REGION Network 14: data move
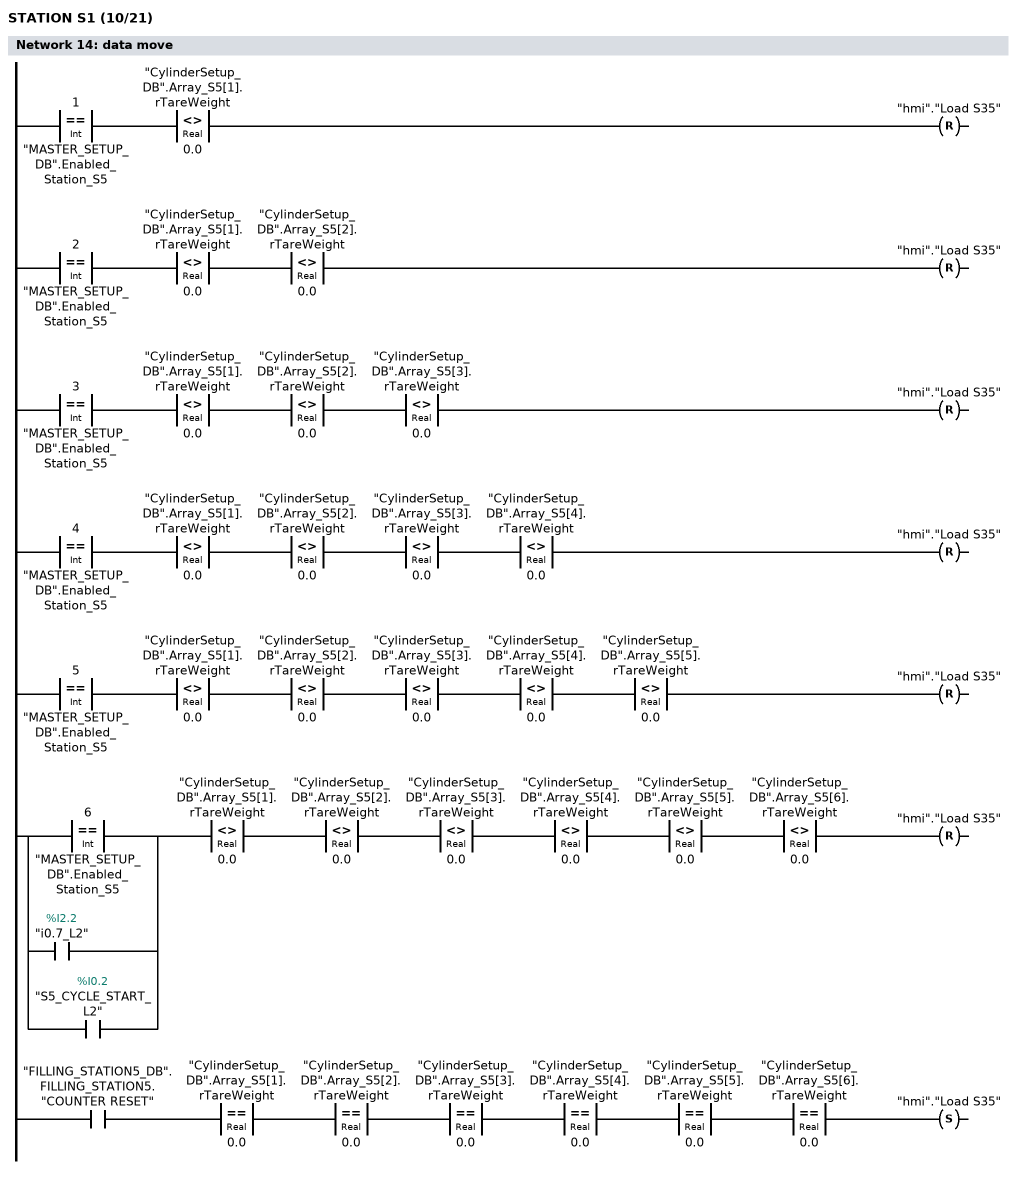
   RUNG wire#powerrail
      { S7_Templates := "SrcType := Int" } EQ_Contact(in1 := 1, in2 := "MASTER_SETUP_DB".Enabled_Station_S5)
      { S7_Templates := "SrcType := Real" } NE_Contact(in1 := "CylinderSetup_DB".Array_S5[1].rTareWeight, in2 := 0.0)
      R_Coil( "hmi"."Load S35" )
   END_RUNG
   RUNG wire#powerrail
      { S7_Templates := "SrcType := Int" } EQ_Contact(in1 := 2, in2 := "MASTER_SETUP_DB".Enabled_Station_S5)
      { S7_Templates := "SrcType := Real" } NE_Contact(in1 := "CylinderSetup_DB".Array_S5[1].rTareWeight, in2 := 0.0)
      { S7_Templates := "SrcType := Real" } NE_Contact(in1 := "CylinderSetup_DB".Array_S5[2].rTareWeight, in2 := 0.0)
      R_Coil( "hmi"."Load S35" )
   END_RUNG
   RUNG wire#powerrail
      { S7_Templates := "SrcType := Int" } EQ_Contact(in1 := 3, in2 := "MASTER_SETUP_DB".Enabled_Station_S5)
      { S7_Templates := "SrcType := Real" } NE_Contact(in1 := "CylinderSetup_DB".Array_S5[1].rTareWeight, in2 := 0.0)
      { S7_Templates := "SrcType := Real" } NE_Contact(in1 := "CylinderSetup_DB".Array_S5[2].rTareWeight, in2 := 0.0)
      { S7_Templates := "SrcType := Real" } NE_Contact(in1 := "CylinderSetup_DB".Array_S5[3].rTareWeight, in2 := 0.0)
      R_Coil( "hmi"."Load S35" )
   END_RUNG
   RUNG wire#powerrail
      { S7_Templates := "SrcType := Int" } EQ_Contact(in1 := 4, in2 := "MASTER_SETUP_DB".Enabled_Station_S5)
      { S7_Templates := "SrcType := Real" } NE_Contact(in1 := "CylinderSetup_DB".Array_S5[1].rTareWeight, in2 := 0.0)
      { S7_Templates := "SrcType := Real" } NE_Contact(in1 := "CylinderSetup_DB".Array_S5[2].rTareWeight, in2 := 0.0)
      { S7_Templates := "SrcType := Real" } NE_Contact(in1 := "CylinderSetup_DB".Array_S5[3].rTareWeight, in2 := 0.0)
      { S7_Templates := "SrcType := Real" } NE_Contact(in1 := "CylinderSetup_DB".Array_S5[4].rTareWeight, in2 := 0.0)
      R_Coil( "hmi"."Load S35" )
   END_RUNG
   RUNG wire#powerrail
      { S7_Templates := "SrcType := Int" } EQ_Contact(in1 := 5, in2 := "MASTER_SETUP_DB".Enabled_Station_S5)
      { S7_Templates := "SrcType := Real" } NE_Contact(in1 := "CylinderSetup_DB".Array_S5[1].rTareWeight, in2 := 0.0)
      { S7_Templates := "SrcType := Real" } NE_Contact(in1 := "CylinderSetup_DB".Array_S5[2].rTareWeight, in2 := 0.0)
      { S7_Templates := "SrcType := Real" } NE_Contact(in1 := "CylinderSetup_DB".Array_S5[3].rTareWeight, in2 := 0.0)
      { S7_Templates := "SrcType := Real" } NE_Contact(in1 := "CylinderSetup_DB".Array_S5[4].rTareWeight, in2 := 0.0)
      { S7_Templates := "SrcType := Real" } NE_Contact(in1 := "CylinderSetup_DB".Array_S5[5].rTareWeight, in2 := 0.0)
      R_Coil( "hmi"."Load S35" )
   END_RUNG
   RUNG wire#powerrail
      { S7_Templates := "SrcType := Int" } EQ_Contact(in1 := 6, in2 := "MASTER_SETUP_DB".Enabled_Station_S5)
      wire#w1
      { S7_Templates := "SrcType := Real" } NE_Contact(in1 := "CylinderSetup_DB".Array_S5[1].rTareWeight, in2 := 0.0)
      { S7_Templates := "SrcType := Real" } NE_Contact(in1 := "CylinderSetup_DB".Array_S5[2].rTareWeight, in2 := 0.0)
      { S7_Templates := "SrcType := Real" } NE_Contact(in1 := "CylinderSetup_DB".Array_S5[3].rTareWeight, in2 := 0.0)
      { S7_Templates := "SrcType := Real" } NE_Contact(in1 := "CylinderSetup_DB".Array_S5[4].rTareWeight, in2 := 0.0)
      { S7_Templates := "SrcType := Real" } NE_Contact(in1 := "CylinderSetup_DB".Array_S5[5].rTareWeight, in2 := 0.0)
      { S7_Templates := "SrcType := Real" } NE_Contact(in1 := "CylinderSetup_DB".Array_S5[6].rTareWeight, in2 := 0.0)
      R_Coil( "hmi"."Load S35" )
   END_RUNG
   RUNG wire#powerrail
      Contact( "i0.7_L2" )
   END_RUNG wire#w1
   RUNG wire#powerrail
      Contact( "S5_CYCLE_START_L2" )
   END_RUNG wire#w1
   RUNG wire#powerrail
      Contact( "FILLING_STATION5_DB".FILLING_STATION5."COUNTER RESET" )
      { S7_Templates := "SrcType := Real" } EQ_Contact(in1 := "CylinderSetup_DB".Array_S5[1].rTareWeight, in2 := 0.0)
      { S7_Templates := "SrcType := Real" } EQ_Contact(in1 := "CylinderSetup_DB".Array_S5[2].rTareWeight, in2 := 0.0)
      { S7_Templates := "SrcType := Real" } EQ_Contact(in1 := "CylinderSetup_DB".Array_S5[3].rTareWeight, in2 := 0.0)
      { S7_Templates := "SrcType := Real" } EQ_Contact(in1 := "CylinderSetup_DB".Array_S5[4].rTareWeight, in2 := 0.0)
      { S7_Templates := "SrcType := Real" } EQ_Contact(in1 := "CylinderSetup_DB".Array_S5[5].rTareWeight, in2 := 0.0)
      { S7_Templates := "SrcType := Real" } EQ_Contact(in1 := "CylinderSetup_DB".Array_S5[6].rTareWeight, in2 := 0.0)
      S_Coil( "hmi"."Load S35" )
   END_RUNG
   // the same network as SCL:
   IF (1 = "MASTER_SETUP_DB".Enabled_Station_S5) AND ("CylinderSetup_DB".Array_S5[1].rTareWeight <> 0.0) THEN
       "hmi"."Load S35" := FALSE;
   END_IF;
   IF (2 = "MASTER_SETUP_DB".Enabled_Station_S5) AND ("CylinderSetup_DB".Array_S5[1].rTareWeight <> 0.0) AND ("CylinderSetup_DB".Array_S5[2].rTareWeight <> 0.0) THEN
       "hmi"."Load S35" := FALSE;
   END_IF;
   IF (3 = "MASTER_SETUP_DB".Enabled_Station_S5) AND ("CylinderSetup_DB".Array_S5[1].rTareWeight <> 0.0) AND ("CylinderSetup_DB".Array_S5[2].rTareWeight <> 0.0) AND ("CylinderSetup_DB".Array_S5[3].rTareWeight <> 0.0) THEN
       "hmi"."Load S35" := FALSE;
   END_IF;
   IF (4 = "MASTER_SETUP_DB".Enabled_Station_S5) AND ("CylinderSetup_DB".Array_S5[1].rTareWeight <> 0.0) AND ("CylinderSetup_DB".Array_S5[2].rTareWeight <> 0.0) AND ("CylinderSetup_DB".Array_S5[3].rTareWeight <> 0.0) AND ("CylinderSetup_DB".Array_S5[4].rTareWeight <> 0.0) THEN
       "hmi"."Load S35" := FALSE;
   END_IF;
   IF (5 = "MASTER_SETUP_DB".Enabled_Station_S5) AND ("CylinderSetup_DB".Array_S5[1].rTareWeight <> 0.0) AND ("CylinderSetup_DB".Array_S5[2].rTareWeight <> 0.0) AND ("CylinderSetup_DB".Array_S5[3].rTareWeight <> 0.0) AND ("CylinderSetup_DB".Array_S5[4].rTareWeight <> 0.0) AND ("CylinderSetup_DB".Array_S5[5].rTareWeight <> 0.0) THEN
       "hmi"."Load S35" := FALSE;
   END_IF;
   IF ((6 = "MASTER_SETUP_DB".Enabled_Station_S5) OR "i0.7_L2" OR "S5_CYCLE_START_L2") AND ("CylinderSetup_DB".Array_S5[1].rTareWeight <> 0.0) AND ("CylinderSetup_DB".Array_S5[2].rTareWeight <> 0.0) AND ("CylinderSetup_DB".Array_S5[3].rTareWeight <> 0.0) AND ("CylinderSetup_DB".Array_S5[4].rTareWeight <> 0.0) AND ("CylinderSetup_DB".Array_S5[5].rTareWeight <> 0.0) AND ("CylinderSetup_DB".Array_S5[6].rTareWeight <> 0.0) THEN
       "hmi"."Load S35" := FALSE;
   END_IF;
   IF "FILLING_STATION5_DB".FILLING_STATION5."COUNTER RESET" AND ("CylinderSetup_DB".Array_S5[1].rTareWeight = 0.0) AND ("CylinderSetup_DB".Array_S5[2].rTareWeight = 0.0) AND ("CylinderSetup_DB".Array_S5[3].rTareWeight = 0.0) AND ("CylinderSetup_DB".Array_S5[4].rTareWeight = 0.0) AND ("CylinderSetup_DB".Array_S5[5].rTareWeight = 0.0) AND ("CylinderSetup_DB".Array_S5[6].rTareWeight = 0.0) THEN
       "hmi"."Load S35" := TRUE;
   END_IF;
END_REGION

REGION Network 15: S5_TO_S7 exit
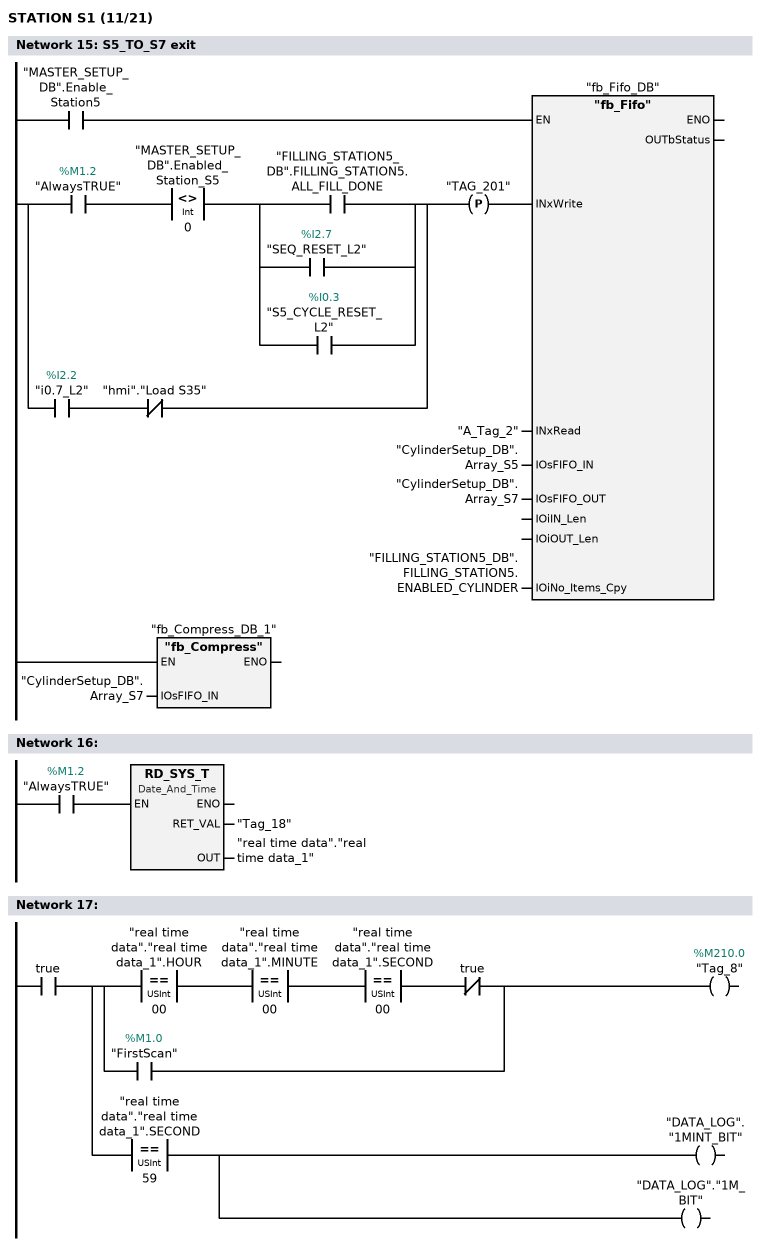
   RUNG wire#powerrail
      Contact( "MASTER_SETUP_DB".Enable_Station5 )
      "fb_Fifo_DB"(INxWrite := wire#w3, INxRead := "A_Tag_2", IOsFIFO_IN := "CylinderSetup_DB".Array_S5, IOsFIFO_OUT := "CylinderSetup_DB".Array_S7, IOiIN_Len :=, IOiOUT_Len :=, IOiNo_Items_Cpy := "FILLING_STATION5_DB".FILLING_STATION5.ENABLED_CYLINDER, OUTbStatus =>)
   END_RUNG
   RUNG wire#powerrail
      Contact( "AlwaysTRUE" )
      { S7_Templates := "SrcType := Int" } NE_Contact(in1 := "MASTER_SETUP_DB".Enabled_Station_S5, in2 := 0)
      wire#w1
      Contact( "FILLING_STATION5_DB".FILLING_STATION5.ALL_FILL_DONE )
      wire#w2
      P_Trig( "TAG_201" )
   END_RUNG wire#w3
   RUNG wire#w1
      Contact( "SEQ_RESET_L2" )
   END_RUNG wire#w2
   RUNG wire#w1
      Contact( "S5_CYCLE_RESET_L2" )
   END_RUNG wire#w2
   RUNG wire#powerrail
      Contact( "i0.7_L2" )
      I_Contact( "hmi"."Load S35" )
   END_RUNG wire#w2
   RUNG wire#powerrail
      "fb_Compress_DB_1"(IOsFIFO_IN := "CylinderSetup_DB".Array_S7)
   END_RUNG
   // the same network as SCL:
   #_w1 := ("AlwaysTRUE" AND ("MASTER_SETUP_DB".Enabled_Station_S5 <> 0) AND ("FILLING_STATION5_DB".FILLING_STATION5.ALL_FILL_DONE OR "SEQ_RESET_L2" OR "S5_CYCLE_RESET_L2")) OR ("i0.7_L2" AND NOT "hmi"."Load S35");
   #_w2 := #_w1 AND NOT "TAG_201";   // rising edge
   "TAG_201" := #_w1;
   IF "MASTER_SETUP_DB".Enable_Station5 THEN
       "fb_Fifo_DB"(INxWrite := #_w2,   // "fb_Fifo"
                    INxRead := "A_Tag_2",
                    IOsFIFO_IN := "CylinderSetup_DB".Array_S5,
                    IOsFIFO_OUT := "CylinderSetup_DB".Array_S7,
                    IOiNo_Items_Cpy := "FILLING_STATION5_DB".FILLING_STATION5.ENABLED_CYLINDER);
   END_IF;
   "fb_Compress_DB_1"(IOsFIFO_IN := "CylinderSetup_DB".Array_S7);   // "fb_Compress"
END_REGION

REGION Network 16
   RUNG wire#powerrail
      Contact( "AlwaysTRUE" )
      { S7_Templates := "date_type := Date_And_Time" } RD_SYS_T(RET_VAL => "Tag_18", OUT => "real time data"."real time data_1")
   END_RUNG
   // the same network as SCL:
   IF "AlwaysTRUE" THEN "Tag_18" := RD_SYS_T(OUT => "real time data"."real time data_1"); END_IF;
END_REGION

REGION Network 17
   RUNG wire#powerrail
      Contact( true )
      wire#w1
      { S7_Templates := "SrcType := USInt" } EQ_Contact(in1 := "real time data"."real time data_1".HOUR, in2 := 00)
      { S7_Templates := "SrcType := USInt" } EQ_Contact(in1 := "real time data"."real time data_1".MINUTE, in2 := 00)
      { S7_Templates := "SrcType := USInt" } EQ_Contact(in1 := "real time data"."real time data_1".SECOND, in2 := 00)
      I_Contact( true )
      wire#w2
      Coil( "Tag_8" )
   END_RUNG
   RUNG wire#w1
      Contact( "FirstScan" )
   END_RUNG wire#w2
   RUNG wire#w1
      { S7_Templates := "SrcType := USInt" } EQ_Contact(in1 := "real time data"."real time data_1".SECOND, in2 := 59)
      wire#w3
      Coil( "DATA_LOG"."1MINT_BIT" )
   END_RUNG
   RUNG wire#w3
      Coil( "DATA_LOG"."1M_BIT" )
   END_RUNG
   // the same network as SCL:
   "Tag_8" := true AND ((("real time data"."real time data_1".HOUR = 00) AND ("real time data"."real time data_1".MINUTE = 00) AND ("real time data"."real time data_1".SECOND = 00) AND NOT true) OR "FirstScan");
   "DATA_LOG"."1MINT_BIT" := true AND ("real time data"."real time data_1".SECOND = 59);
   "DATA_LOG"."1M_BIT" := "DATA_LOG"."1MINT_BIT";
END_REGION

REGION Network 18 (SCL): S4 S6 FIFO DATA SKIP
   #idx2 := 0;
   #idx3 := 0;

   IF "AlwaysTRUE" THEN
       FOR #idx2 := 1 TO "MASTER_SETUP_DB".S4_Total_Station DO

           IF "MASTER_SETUP_DB".S4_Enabled_Station[#idx2]  THEN
               #idx3 := #idx3 + 1;
               "hmi_dummy_array".S4_PrefillingDummyData[#idx2] := "CylinderSetup_DB".Array_S6[#idx3];

             ELSIF
                #idx2 > "MASTER_SETUP_DB".S4_Total_Station OR #idx3 >"MASTER_SETUP_DB".S4_Total_Station THEN
                   EXIT;
               END_IF;
           END_FOR;


   END_IF;
END_REGION

REGION Network 19 (SCL)
   #idx4 := 0;
   #idx6 := 0;

   IF "AlwaysTRUE" THEN
       FOR #idx4 := 1 TO "MASTER_SETUP_DB".S5_Total_Station DO

           IF "MASTER_SETUP_DB".S5_Enabled_Station[#idx4] THEN
               #idx6 := #idx6 + 1;
               "hmi_dummy_array".S5_PrefillingdummyData[#idx4] := "CylinderSetup_DB".Array_S5[#idx6];

           ELSIF
               #idx4 > "MASTER_SETUP_DB".S5_Total_Station OR #idx6 > "MASTER_SETUP_DB".S5_Total_Station THEN
               EXIT;
           END_IF;
       END_FOR;


   END_IF;
END_REGION

REGION Network 20
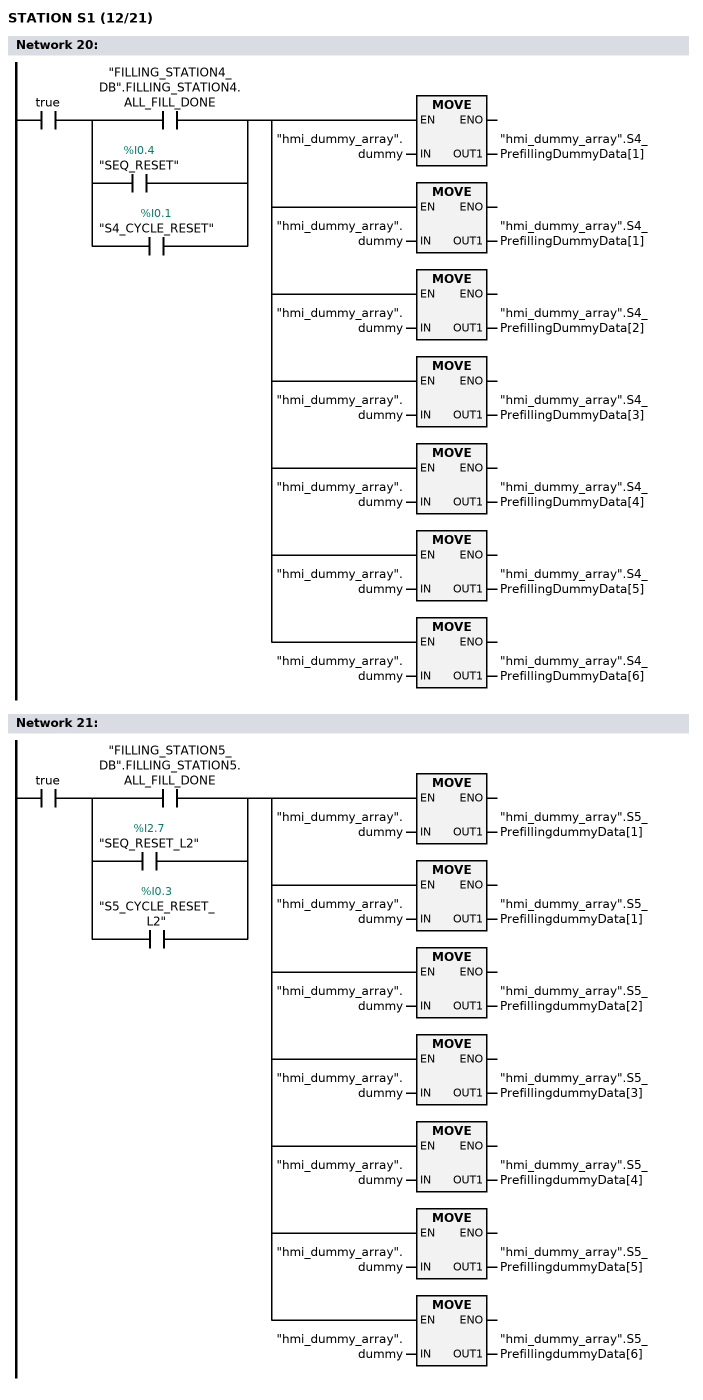
   RUNG wire#powerrail
      Contact( true )
      wire#w1
      Contact( "FILLING_STATION4_DB".FILLING_STATION4.ALL_FILL_DONE )
      wire#w2
      Move(in := "hmi_dummy_array".dummy, out1 => "hmi_dummy_array".S4_PrefillingDummyData[1])
   END_RUNG
   RUNG wire#w1
      Contact( "SEQ_RESET" )
   END_RUNG wire#w2
   RUNG wire#w1
      Contact( "S4_CYCLE_RESET" )
   END_RUNG wire#w2
   RUNG wire#w2
      Move(in := "hmi_dummy_array".dummy, out1 => "hmi_dummy_array".S4_PrefillingDummyData[1])
   END_RUNG
   RUNG wire#w2
      Move(in := "hmi_dummy_array".dummy, out1 => "hmi_dummy_array".S4_PrefillingDummyData[2])
   END_RUNG
   RUNG wire#w2
      Move(in := "hmi_dummy_array".dummy, out1 => "hmi_dummy_array".S4_PrefillingDummyData[3])
   END_RUNG
   RUNG wire#w2
      Move(in := "hmi_dummy_array".dummy, out1 => "hmi_dummy_array".S4_PrefillingDummyData[4])
   END_RUNG
   RUNG wire#w2
      Move(in := "hmi_dummy_array".dummy, out1 => "hmi_dummy_array".S4_PrefillingDummyData[5])
   END_RUNG
   RUNG wire#w2
      Move(in := "hmi_dummy_array".dummy, out1 => "hmi_dummy_array".S4_PrefillingDummyData[6])
   END_RUNG
   // the same network as SCL:
   IF true AND ("FILLING_STATION4_DB".FILLING_STATION4.ALL_FILL_DONE OR "SEQ_RESET" OR "S4_CYCLE_RESET") THEN
       "hmi_dummy_array".S4_PrefillingDummyData[1] := "hmi_dummy_array".dummy;
       "hmi_dummy_array".S4_PrefillingDummyData[1] := "hmi_dummy_array".dummy;
       "hmi_dummy_array".S4_PrefillingDummyData[2] := "hmi_dummy_array".dummy;
       "hmi_dummy_array".S4_PrefillingDummyData[3] := "hmi_dummy_array".dummy;
       "hmi_dummy_array".S4_PrefillingDummyData[4] := "hmi_dummy_array".dummy;
       "hmi_dummy_array".S4_PrefillingDummyData[5] := "hmi_dummy_array".dummy;
       "hmi_dummy_array".S4_PrefillingDummyData[6] := "hmi_dummy_array".dummy;
   END_IF;
END_REGION

REGION Network 21
   RUNG wire#powerrail
      Contact( true )
      wire#w1
      Contact( "FILLING_STATION5_DB".FILLING_STATION5.ALL_FILL_DONE )
      wire#w2
      Move(in := "hmi_dummy_array".dummy, out1 => "hmi_dummy_array".S5_PrefillingdummyData[1])
   END_RUNG
   RUNG wire#w1
      Contact( "SEQ_RESET_L2" )
   END_RUNG wire#w2
   RUNG wire#w1
      Contact( "S5_CYCLE_RESET_L2" )
   END_RUNG wire#w2
   RUNG wire#w2
      Move(in := "hmi_dummy_array".dummy, out1 => "hmi_dummy_array".S5_PrefillingdummyData[1])
   END_RUNG
   RUNG wire#w2
      Move(in := "hmi_dummy_array".dummy, out1 => "hmi_dummy_array".S5_PrefillingdummyData[2])
   END_RUNG
   RUNG wire#w2
      Move(in := "hmi_dummy_array".dummy, out1 => "hmi_dummy_array".S5_PrefillingdummyData[3])
   END_RUNG
   RUNG wire#w2
      Move(in := "hmi_dummy_array".dummy, out1 => "hmi_dummy_array".S5_PrefillingdummyData[4])
   END_RUNG
   RUNG wire#w2
      Move(in := "hmi_dummy_array".dummy, out1 => "hmi_dummy_array".S5_PrefillingdummyData[5])
   END_RUNG
   RUNG wire#w2
      Move(in := "hmi_dummy_array".dummy, out1 => "hmi_dummy_array".S5_PrefillingdummyData[6])
   END_RUNG
   // the same network as SCL:
   IF true AND ("FILLING_STATION5_DB".FILLING_STATION5.ALL_FILL_DONE OR "SEQ_RESET_L2" OR "S5_CYCLE_RESET_L2") THEN
       "hmi_dummy_array".S5_PrefillingdummyData[1] := "hmi_dummy_array".dummy;
       "hmi_dummy_array".S5_PrefillingdummyData[1] := "hmi_dummy_array".dummy;
       "hmi_dummy_array".S5_PrefillingdummyData[2] := "hmi_dummy_array".dummy;
       "hmi_dummy_array".S5_PrefillingdummyData[3] := "hmi_dummy_array".dummy;
       "hmi_dummy_array".S5_PrefillingdummyData[4] := "hmi_dummy_array".dummy;
       "hmi_dummy_array".S5_PrefillingdummyData[5] := "hmi_dummy_array".dummy;
       "hmi_dummy_array".S5_PrefillingdummyData[6] := "hmi_dummy_array".dummy;
   END_IF;
END_REGION

REGION Network 22
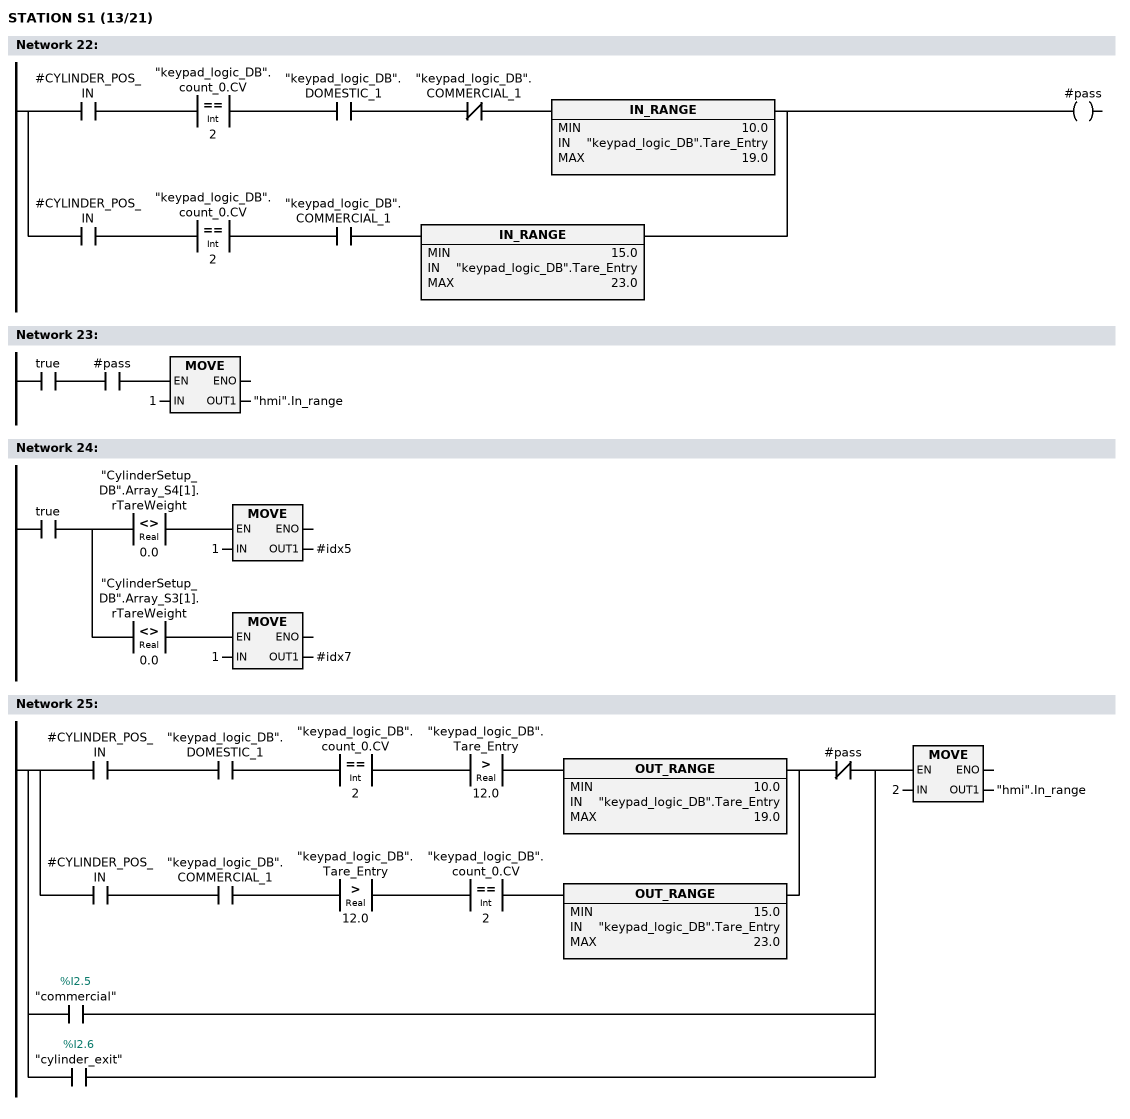
   RUNG wire#powerrail
      Contact( #CYLINDER_POS_IN )
      { S7_Templates := "SrcType := Int" } EQ_Contact(in1 := "keypad_logic_DB".count_0.CV, in2 := 2)
      Contact( "keypad_logic_DB".DOMESTIC_1 )
      I_Contact( "keypad_logic_DB".COMMERCIAL_1 )
      { S7_Templates := "SrcType := Real" } InRange(min := 10.0, in := "keypad_logic_DB".Tare_Entry, max := 19.0)
      wire#w1
      Coil( #pass )
   END_RUNG
   RUNG wire#powerrail
      Contact( #CYLINDER_POS_IN )
      { S7_Templates := "SrcType := Int" } EQ_Contact(in1 := "keypad_logic_DB".count_0.CV, in2 := 2)
      Contact( "keypad_logic_DB".COMMERCIAL_1 )
      { S7_Templates := "SrcType := Real" } InRange(min := 15.0, in := "keypad_logic_DB".Tare_Entry, max := 23.0)
   END_RUNG wire#w1
   // the same network as SCL:
   #pass := (#CYLINDER_POS_IN AND ("keypad_logic_DB".count_0.CV = 2) AND "keypad_logic_DB".DOMESTIC_1 AND NOT "keypad_logic_DB".COMMERCIAL_1 AND (10.0 <= "keypad_logic_DB".Tare_Entry) AND ("keypad_logic_DB".Tare_Entry <= 19.0)) OR (#CYLINDER_POS_IN AND ("keypad_logic_DB".count_0.CV = 2) AND "keypad_logic_DB".COMMERCIAL_1 AND (15.0 <= "keypad_logic_DB".Tare_Entry) AND ("keypad_logic_DB".Tare_Entry <= 23.0));
END_REGION

REGION Network 23
   RUNG wire#powerrail
      Contact( true )
      Contact( #pass )
      Move(in := 1, out1 => "hmi".In_range)
   END_RUNG
   // the same network as SCL:
   IF true AND #pass THEN "hmi".In_range := 1; END_IF;
END_REGION

REGION Network 24
   RUNG wire#powerrail
      Contact( true )
      wire#w1
      { S7_Templates := "SrcType := Real" } NE_Contact(in1 := "CylinderSetup_DB".Array_S4[1].rTareWeight, in2 := 0.0)
      Move(in := 1, out1 => #idx5)
   END_RUNG
   RUNG wire#w1
      { S7_Templates := "SrcType := Real" } NE_Contact(in1 := "CylinderSetup_DB".Array_S3[1].rTareWeight, in2 := 0.0)
      Move(in := 1, out1 => #idx7)
   END_RUNG
   // the same network as SCL:
   IF true AND ("CylinderSetup_DB".Array_S4[1].rTareWeight <> 0.0) THEN #idx5 := 1; END_IF;
   IF true AND ("CylinderSetup_DB".Array_S3[1].rTareWeight <> 0.0) THEN #idx7 := 1; END_IF;
END_REGION

REGION Network 25
   IF (((#CYLINDER_POS_IN AND "keypad_logic_DB".DOMESTIC_1 AND ("keypad_logic_DB".count_0.CV = 2) AND ("keypad_logic_DB".Tare_Entry > 12.0) AND (("keypad_logic_DB".Tare_Entry < 10.0) OR ("keypad_logic_DB".Tare_Entry > 19.0))) OR (#CYLINDER_POS_IN AND "keypad_logic_DB".COMMERCIAL_1 AND ("keypad_logic_DB".Tare_Entry > 12.0) AND ("keypad_logic_DB".count_0.CV = 2) AND (("keypad_logic_DB".Tare_Entry < 15.0) OR ("keypad_logic_DB".Tare_Entry > 23.0)))) AND NOT #pass) OR "commercial" OR "cylinder_exit" THEN
       "hmi".In_range := 2;
   END_IF;
END_REGION

REGION Network 26
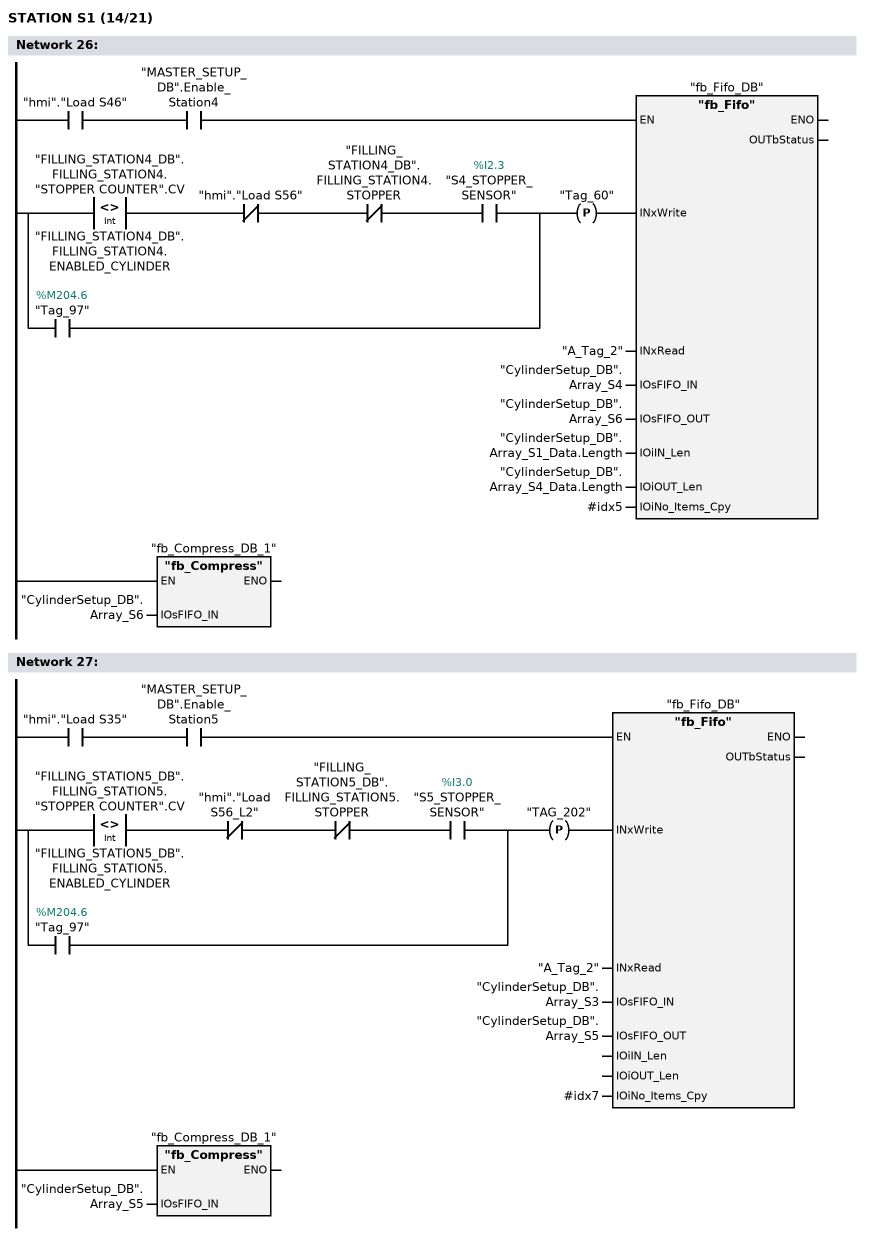
   RUNG wire#powerrail
      Contact( "hmi"."Load S46" )
      Contact( "MASTER_SETUP_DB".Enable_Station4 )
      "fb_Fifo_DB"(INxWrite := wire#w2, INxRead := "A_Tag_2", IOsFIFO_IN := "CylinderSetup_DB".Array_S4, IOsFIFO_OUT := "CylinderSetup_DB".Array_S6, IOiIN_Len := "CylinderSetup_DB".Array_S1_Data.Length, IOiOUT_Len := "CylinderSetup_DB".Array_S4_Data.Length, IOiNo_Items_Cpy := #idx5, OUTbStatus =>)
   END_RUNG
   RUNG wire#powerrail
      { S7_Templates := "SrcType := Int" } NE_Contact(in1 := "FILLING_STATION4_DB".FILLING_STATION4."STOPPER COUNTER".CV, in2 := "FILLING_STATION4_DB".FILLING_STATION4.ENABLED_CYLINDER)
      I_Contact( "hmi"."Load S56" )
      I_Contact( "FILLING_STATION4_DB".FILLING_STATION4.STOPPER )
      Contact( "S4_STOPPER_SENSOR" )
      wire#w1
      P_Trig( "Tag_60" )
   END_RUNG wire#w2
   RUNG wire#powerrail
      Contact( "Tag_97" )
   END_RUNG wire#w1
   RUNG wire#powerrail
      "fb_Compress_DB_1"(IOsFIFO_IN := "CylinderSetup_DB".Array_S6)
   END_RUNG
   // the same network as SCL:
   #_w1 := (("FILLING_STATION4_DB".FILLING_STATION4."STOPPER COUNTER".CV <> "FILLING_STATION4_DB".FILLING_STATION4.ENABLED_CYLINDER) AND NOT "hmi"."Load S56" AND NOT "FILLING_STATION4_DB".FILLING_STATION4.STOPPER AND "S4_STOPPER_SENSOR") OR "Tag_97";
   #_w2 := #_w1 AND NOT "Tag_60";   // rising edge
   "Tag_60" := #_w1;
   IF "hmi"."Load S46" AND "MASTER_SETUP_DB".Enable_Station4 THEN
       "fb_Fifo_DB"(INxWrite := #_w2,   // "fb_Fifo"
                    INxRead := "A_Tag_2",
                    IOsFIFO_IN := "CylinderSetup_DB".Array_S4,
                    IOsFIFO_OUT := "CylinderSetup_DB".Array_S6,
                    IOiIN_Len := "CylinderSetup_DB".Array_S1_Data.Length,
                    IOiOUT_Len := "CylinderSetup_DB".Array_S4_Data.Length,
                    IOiNo_Items_Cpy := #idx5);
   END_IF;
   "fb_Compress_DB_1"(IOsFIFO_IN := "CylinderSetup_DB".Array_S6);   // "fb_Compress"
END_REGION

REGION Network 27
   RUNG wire#powerrail
      Contact( "hmi"."Load S35" )
      Contact( "MASTER_SETUP_DB".Enable_Station5 )
      "fb_Fifo_DB"(INxWrite := wire#w2, INxRead := "A_Tag_2", IOsFIFO_IN := "CylinderSetup_DB".Array_S3, IOsFIFO_OUT := "CylinderSetup_DB".Array_S5, IOiIN_Len :=, IOiOUT_Len :=, IOiNo_Items_Cpy := #idx7, OUTbStatus =>)
   END_RUNG
   RUNG wire#powerrail
      { S7_Templates := "SrcType := Int" } NE_Contact(in1 := "FILLING_STATION5_DB".FILLING_STATION5."STOPPER COUNTER".CV, in2 := "FILLING_STATION5_DB".FILLING_STATION5.ENABLED_CYLINDER)
      I_Contact( "hmi"."Load S56_L2" )
      I_Contact( "FILLING_STATION5_DB".FILLING_STATION5.STOPPER )
      Contact( "S5_STOPPER_SENSOR" )
      wire#w1
      P_Trig( "TAG_202" )
   END_RUNG wire#w2
   RUNG wire#powerrail
      Contact( "Tag_97" )
   END_RUNG wire#w1
   RUNG wire#powerrail
      "fb_Compress_DB_1"(IOsFIFO_IN := "CylinderSetup_DB".Array_S5)
   END_RUNG
   // the same network as SCL:
   #_w1 := (("FILLING_STATION5_DB".FILLING_STATION5."STOPPER COUNTER".CV <> "FILLING_STATION5_DB".FILLING_STATION5.ENABLED_CYLINDER) AND NOT "hmi"."Load S56_L2" AND NOT "FILLING_STATION5_DB".FILLING_STATION5.STOPPER AND "S5_STOPPER_SENSOR") OR "Tag_97";
   #_w2 := #_w1 AND NOT "TAG_202";   // rising edge
   "TAG_202" := #_w1;
   IF "hmi"."Load S35" AND "MASTER_SETUP_DB".Enable_Station5 THEN
       "fb_Fifo_DB"(INxWrite := #_w2,   // "fb_Fifo"
                    INxRead := "A_Tag_2",
                    IOsFIFO_IN := "CylinderSetup_DB".Array_S3,
                    IOsFIFO_OUT := "CylinderSetup_DB".Array_S5,
                    IOiNo_Items_Cpy := #idx7);
   END_IF;
   "fb_Compress_DB_1"(IOsFIFO_IN := "CylinderSetup_DB".Array_S5);   // "fb_Compress"
END_REGION

REGION Network 28
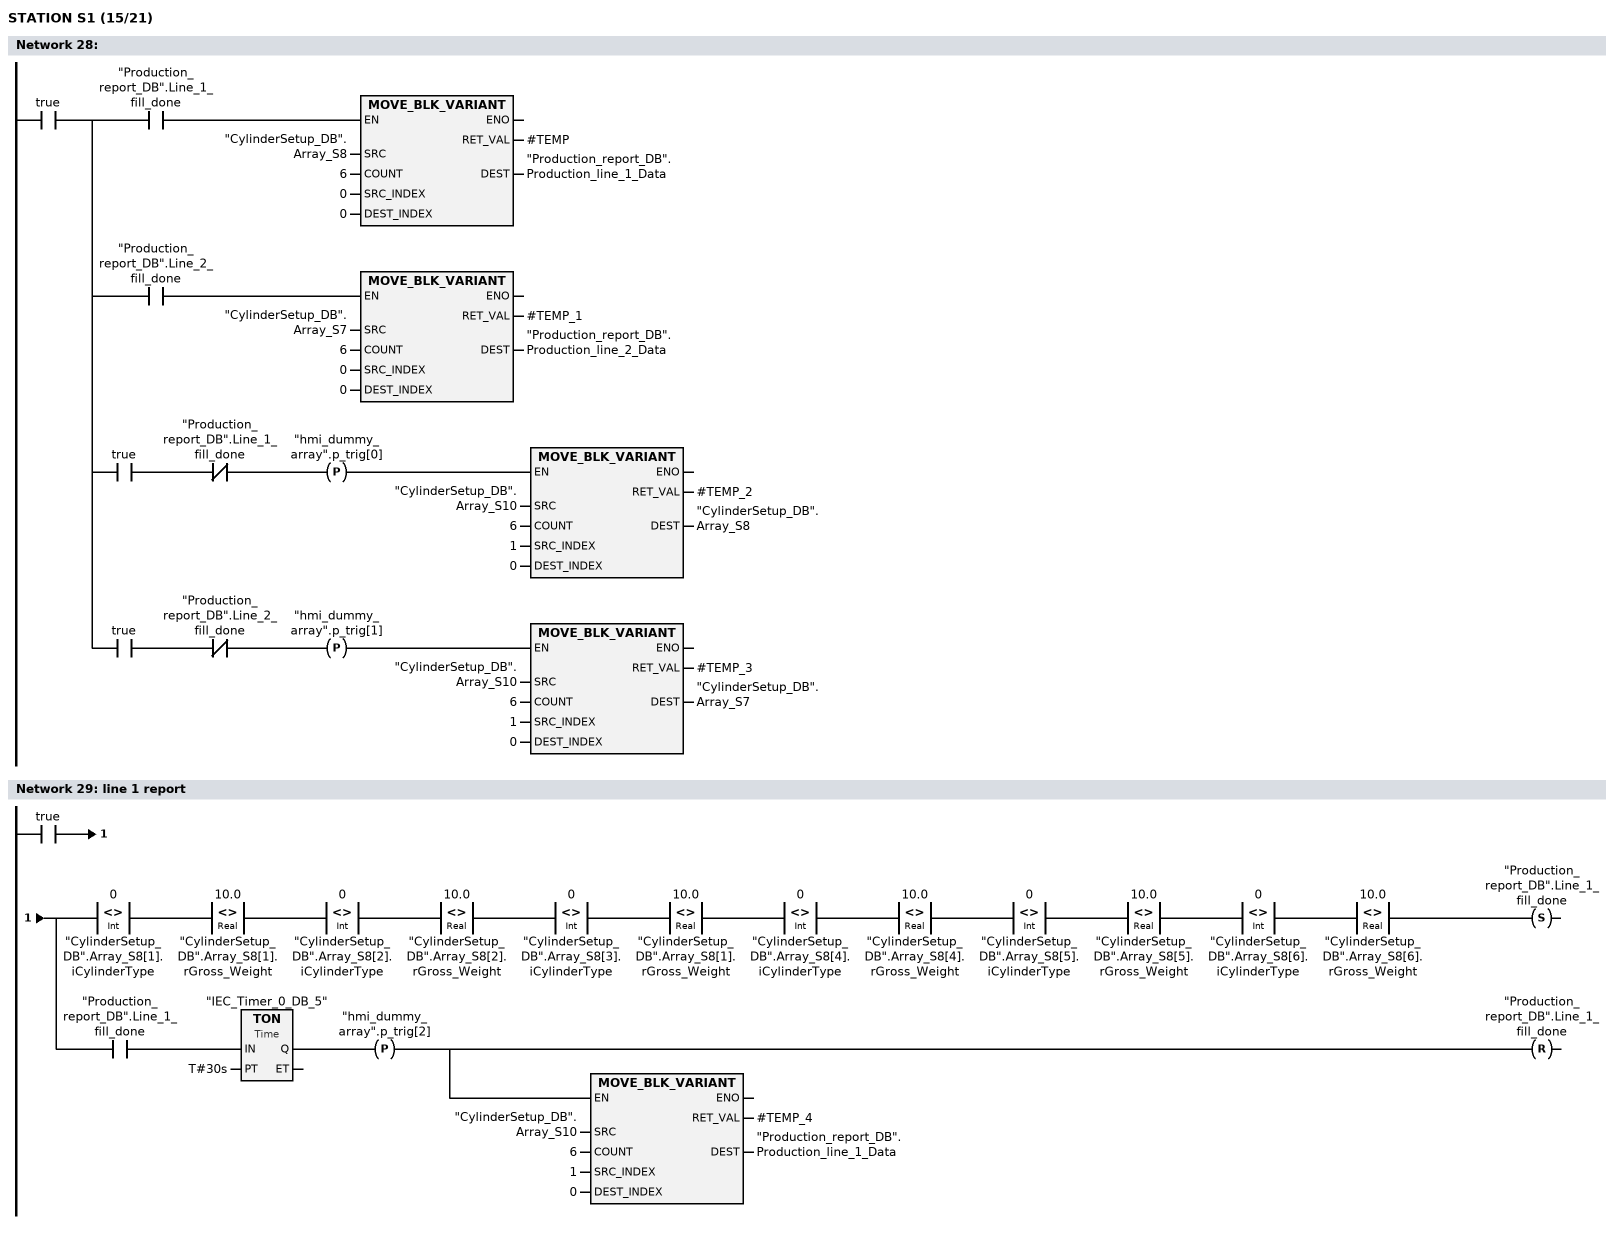
   RUNG wire#powerrail
      Contact( true )
      wire#w1
      Contact( "Production_report_DB".Line_1_fill_done )
      MOVE_BLK_VARIANT(SRC := "CylinderSetup_DB".Array_S8, COUNT := 6, SRC_INDEX := 0, DEST_INDEX := 0, Ret_Val => #TEMP, DEST => "Production_report_DB".Production_line_1_Data)
   END_RUNG
   RUNG wire#w1
      Contact( "Production_report_DB".Line_2_fill_done )
      MOVE_BLK_VARIANT(SRC := "CylinderSetup_DB".Array_S7, COUNT := 6, SRC_INDEX := 0, DEST_INDEX := 0, Ret_Val => #TEMP_1, DEST => "Production_report_DB".Production_line_2_Data)
   END_RUNG
   RUNG wire#w1
      Contact( true )
      I_Contact( "Production_report_DB".Line_1_fill_done )
      P_Trig( "hmi_dummy_array".p_trig[0] )
      MOVE_BLK_VARIANT(SRC := "CylinderSetup_DB".Array_S10, COUNT := 6, SRC_INDEX := 1, DEST_INDEX := 0, Ret_Val => #TEMP_2, DEST => "CylinderSetup_DB".Array_S8)
   END_RUNG
   RUNG wire#w1
      Contact( true )
      I_Contact( "Production_report_DB".Line_2_fill_done )
      P_Trig( "hmi_dummy_array".p_trig[1] )
      MOVE_BLK_VARIANT(SRC := "CylinderSetup_DB".Array_S10, COUNT := 6, SRC_INDEX := 1, DEST_INDEX := 0, Ret_Val => #TEMP_3, DEST => "CylinderSetup_DB".Array_S7)
   END_RUNG
   // the same network as SCL:
   IF true AND "Production_report_DB".Line_1_fill_done THEN
       #TEMP := MOVE_BLK_VARIANT(SRC := "CylinderSetup_DB".Array_S8,
                               COUNT := 6,
                               SRC_INDEX := 0,
                               DEST_INDEX := 0,
                               DEST => "Production_report_DB".Production_line_1_Data);
   END_IF;
   IF true AND "Production_report_DB".Line_2_fill_done THEN
       #TEMP_1 := MOVE_BLK_VARIANT(SRC := "CylinderSetup_DB".Array_S7,
                               COUNT := 6,
                               SRC_INDEX := 0,
                               DEST_INDEX := 0,
                               DEST => "Production_report_DB".Production_line_2_Data);
   END_IF;
   #_w1 := true AND true AND NOT "Production_report_DB".Line_1_fill_done;
   #_w2 := #_w1 AND NOT "hmi_dummy_array".p_trig[0];   // rising edge
   "hmi_dummy_array".p_trig[0] := #_w1;
   IF #_w2 THEN
       #TEMP_2 := MOVE_BLK_VARIANT(SRC := "CylinderSetup_DB".Array_S10,
                               COUNT := 6,
                               SRC_INDEX := 1,
                               DEST_INDEX := 0,
                               DEST => "CylinderSetup_DB".Array_S8);
   END_IF;
   #_w3 := true AND true AND NOT "Production_report_DB".Line_2_fill_done;
   #_w4 := #_w3 AND NOT "hmi_dummy_array".p_trig[1];   // rising edge
   "hmi_dummy_array".p_trig[1] := #_w3;
   IF #_w4 THEN
       #TEMP_3 := MOVE_BLK_VARIANT(SRC := "CylinderSetup_DB".Array_S10,
                               COUNT := 6,
                               SRC_INDEX := 1,
                               DEST_INDEX := 0,
                               DEST => "CylinderSetup_DB".Array_S7);
   END_IF;
END_REGION

REGION Network 29: line 1 report
   RUNG wire#powerrail
      Contact( true )
      wire#w1
      { S7_Templates := "SrcType := Int" } NE_Contact(in1 := 0, in2 := "CylinderSetup_DB".Array_S8[1].iCylinderType)
      { S7_Templates := "SrcType := Real" } NE_Contact(in1 := 10.0, in2 := "CylinderSetup_DB".Array_S8[1].rGross_Weight)
      { S7_Templates := "SrcType := Int" } NE_Contact(in1 := 0, in2 := "CylinderSetup_DB".Array_S8[2].iCylinderType)
      { S7_Templates := "SrcType := Real" } NE_Contact(in1 := 10.0, in2 := "CylinderSetup_DB".Array_S8[2].rGross_Weight)
      { S7_Templates := "SrcType := Int" } NE_Contact(in1 := 0, in2 := "CylinderSetup_DB".Array_S8[3].iCylinderType)
      { S7_Templates := "SrcType := Real" } NE_Contact(in1 := 10.0, in2 := "CylinderSetup_DB".Array_S8[1].rGross_Weight)
      { S7_Templates := "SrcType := Int" } NE_Contact(in1 := 0, in2 := "CylinderSetup_DB".Array_S8[4].iCylinderType)
      { S7_Templates := "SrcType := Real" } NE_Contact(in1 := 10.0, in2 := "CylinderSetup_DB".Array_S8[4].rGross_Weight)
      { S7_Templates := "SrcType := Int" } NE_Contact(in1 := 0, in2 := "CylinderSetup_DB".Array_S8[5].iCylinderType)
      { S7_Templates := "SrcType := Real" } NE_Contact(in1 := 10.0, in2 := "CylinderSetup_DB".Array_S8[5].rGross_Weight)
      { S7_Templates := "SrcType := Int" } NE_Contact(in1 := 0, in2 := "CylinderSetup_DB".Array_S8[6].iCylinderType)
      { S7_Templates := "SrcType := Real" } NE_Contact(in1 := 10.0, in2 := "CylinderSetup_DB".Array_S8[6].rGross_Weight)
      S_Coil( "Production_report_DB".Line_1_fill_done )
   END_RUNG
   RUNG wire#w1
      Contact( "Production_report_DB".Line_1_fill_done )
      { S7_Templates := "time_type := Time" } "IEC_Timer_0_DB_5".TON(pt := T#30s, et =>)
      P_Trig( "hmi_dummy_array".p_trig[2] )
      wire#w2
      R_Coil( "Production_report_DB".Line_1_fill_done )
   END_RUNG
   RUNG wire#w2
      MOVE_BLK_VARIANT(SRC := "CylinderSetup_DB".Array_S10, COUNT := 6, SRC_INDEX := 1, DEST_INDEX := 0, Ret_Val => #TEMP_4, DEST => "Production_report_DB".Production_line_1_Data)
   END_RUNG
   // the same network as SCL:
   IF true AND (0 <> "CylinderSetup_DB".Array_S8[1].iCylinderType) AND (10.0 <> "CylinderSetup_DB".Array_S8[1].rGross_Weight) AND (0 <> "CylinderSetup_DB".Array_S8[2].iCylinderType) AND (10.0 <> "CylinderSetup_DB".Array_S8[2].rGross_Weight) AND (0 <> "CylinderSetup_DB".Array_S8[3].iCylinderType) AND (10.0 <> "CylinderSetup_DB".Array_S8[1].rGross_Weight) AND (0 <> "CylinderSetup_DB".Array_S8[4].iCylinderType) AND (10.0 <> "CylinderSetup_DB".Array_S8[4].rGross_Weight) AND (0 <> "CylinderSetup_DB".Array_S8[5].iCylinderType) AND (10.0 <> "CylinderSetup_DB".Array_S8[5].rGross_Weight) AND (0 <> "CylinderSetup_DB".Array_S8[6].iCylinderType) AND (10.0 <> "CylinderSetup_DB".Array_S8[6].rGross_Weight) THEN
       "Production_report_DB".Line_1_fill_done := TRUE;
   END_IF;
   "IEC_Timer_0_DB_5".TON(IN := true AND "Production_report_DB".Line_1_fill_done, PT := T#30s);
   #_w1 := "IEC_Timer_0_DB_5".Q AND NOT "hmi_dummy_array".p_trig[2];   // rising edge
   "hmi_dummy_array".p_trig[2] := "IEC_Timer_0_DB_5".Q;
   IF #_w1 THEN
       "Production_report_DB".Line_1_fill_done := FALSE;
       #TEMP_4 := MOVE_BLK_VARIANT(SRC := "CylinderSetup_DB".Array_S10,
                               COUNT := 6,
                               SRC_INDEX := 1,
                               DEST_INDEX := 0,
                               DEST => "Production_report_DB".Production_line_1_Data);
   END_IF;
END_REGION

REGION Network 30: line 2 report
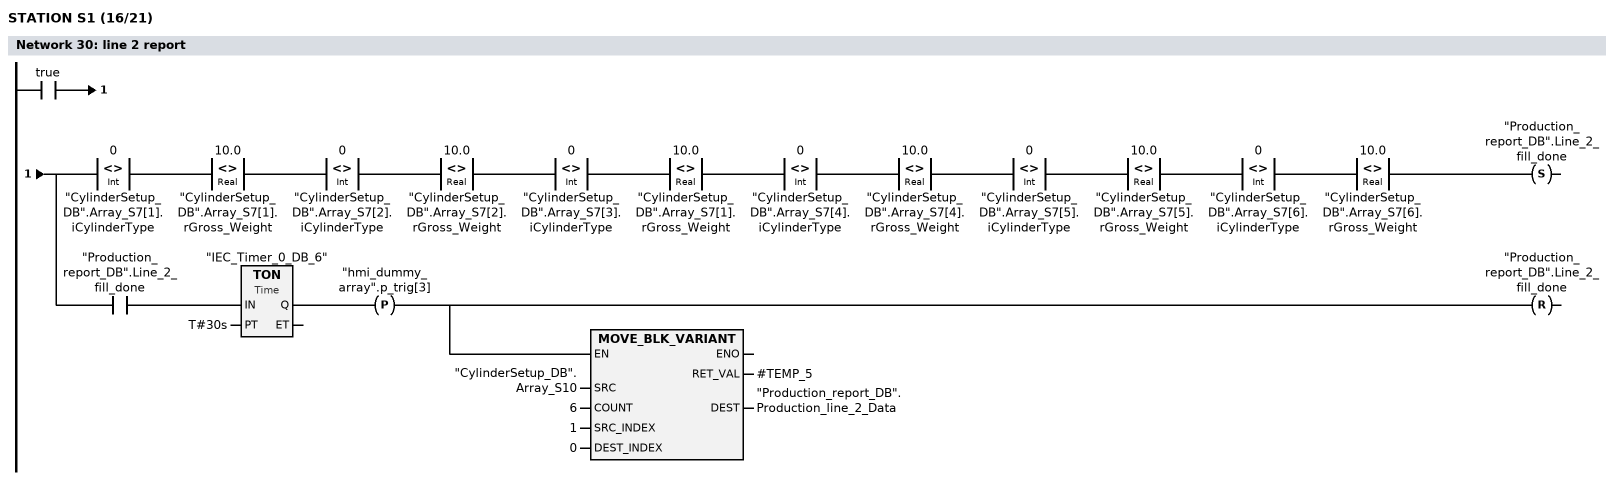
   RUNG wire#powerrail
      Contact( true )
      wire#w1
      { S7_Templates := "SrcType := Int" } NE_Contact(in1 := 0, in2 := "CylinderSetup_DB".Array_S7[1].iCylinderType)
      { S7_Templates := "SrcType := Real" } NE_Contact(in1 := 10.0, in2 := "CylinderSetup_DB".Array_S7[1].rGross_Weight)
      { S7_Templates := "SrcType := Int" } NE_Contact(in1 := 0, in2 := "CylinderSetup_DB".Array_S7[2].iCylinderType)
      { S7_Templates := "SrcType := Real" } NE_Contact(in1 := 10.0, in2 := "CylinderSetup_DB".Array_S7[2].rGross_Weight)
      { S7_Templates := "SrcType := Int" } NE_Contact(in1 := 0, in2 := "CylinderSetup_DB".Array_S7[3].iCylinderType)
      { S7_Templates := "SrcType := Real" } NE_Contact(in1 := 10.0, in2 := "CylinderSetup_DB".Array_S7[1].rGross_Weight)
      { S7_Templates := "SrcType := Int" } NE_Contact(in1 := 0, in2 := "CylinderSetup_DB".Array_S7[4].iCylinderType)
      { S7_Templates := "SrcType := Real" } NE_Contact(in1 := 10.0, in2 := "CylinderSetup_DB".Array_S7[4].rGross_Weight)
      { S7_Templates := "SrcType := Int" } NE_Contact(in1 := 0, in2 := "CylinderSetup_DB".Array_S7[5].iCylinderType)
      { S7_Templates := "SrcType := Real" } NE_Contact(in1 := 10.0, in2 := "CylinderSetup_DB".Array_S7[5].rGross_Weight)
      { S7_Templates := "SrcType := Int" } NE_Contact(in1 := 0, in2 := "CylinderSetup_DB".Array_S7[6].iCylinderType)
      { S7_Templates := "SrcType := Real" } NE_Contact(in1 := 10.0, in2 := "CylinderSetup_DB".Array_S7[6].rGross_Weight)
      S_Coil( "Production_report_DB".Line_2_fill_done )
   END_RUNG
   RUNG wire#w1
      Contact( "Production_report_DB".Line_2_fill_done )
      { S7_Templates := "time_type := Time" } "IEC_Timer_0_DB_6".TON(pt := T#30s, et =>)
      P_Trig( "hmi_dummy_array".p_trig[3] )
      wire#w2
      R_Coil( "Production_report_DB".Line_2_fill_done )
   END_RUNG
   RUNG wire#w2
      MOVE_BLK_VARIANT(SRC := "CylinderSetup_DB".Array_S10, COUNT := 6, SRC_INDEX := 1, DEST_INDEX := 0, Ret_Val => #TEMP_5, DEST => "Production_report_DB".Production_line_2_Data)
   END_RUNG
   // the same network as SCL:
   IF true AND (0 <> "CylinderSetup_DB".Array_S7[1].iCylinderType) AND (10.0 <> "CylinderSetup_DB".Array_S7[1].rGross_Weight) AND (0 <> "CylinderSetup_DB".Array_S7[2].iCylinderType) AND (10.0 <> "CylinderSetup_DB".Array_S7[2].rGross_Weight) AND (0 <> "CylinderSetup_DB".Array_S7[3].iCylinderType) AND (10.0 <> "CylinderSetup_DB".Array_S7[1].rGross_Weight) AND (0 <> "CylinderSetup_DB".Array_S7[4].iCylinderType) AND (10.0 <> "CylinderSetup_DB".Array_S7[4].rGross_Weight) AND (0 <> "CylinderSetup_DB".Array_S7[5].iCylinderType) AND (10.0 <> "CylinderSetup_DB".Array_S7[5].rGross_Weight) AND (0 <> "CylinderSetup_DB".Array_S7[6].iCylinderType) AND (10.0 <> "CylinderSetup_DB".Array_S7[6].rGross_Weight) THEN
       "Production_report_DB".Line_2_fill_done := TRUE;
   END_IF;
   "IEC_Timer_0_DB_6".TON(IN := true AND "Production_report_DB".Line_2_fill_done, PT := T#30s);
   #_w1 := "IEC_Timer_0_DB_6".Q AND NOT "hmi_dummy_array".p_trig[3];   // rising edge
   "hmi_dummy_array".p_trig[3] := "IEC_Timer_0_DB_6".Q;
   IF #_w1 THEN
       "Production_report_DB".Line_2_fill_done := FALSE;
       #TEMP_5 := MOVE_BLK_VARIANT(SRC := "CylinderSetup_DB".Array_S10,
                               COUNT := 6,
                               SRC_INDEX := 1,
                               DEST_INDEX := 0,
                               DEST => "Production_report_DB".Production_line_2_Data);
   END_IF;
END_REGION

REGION Network 31
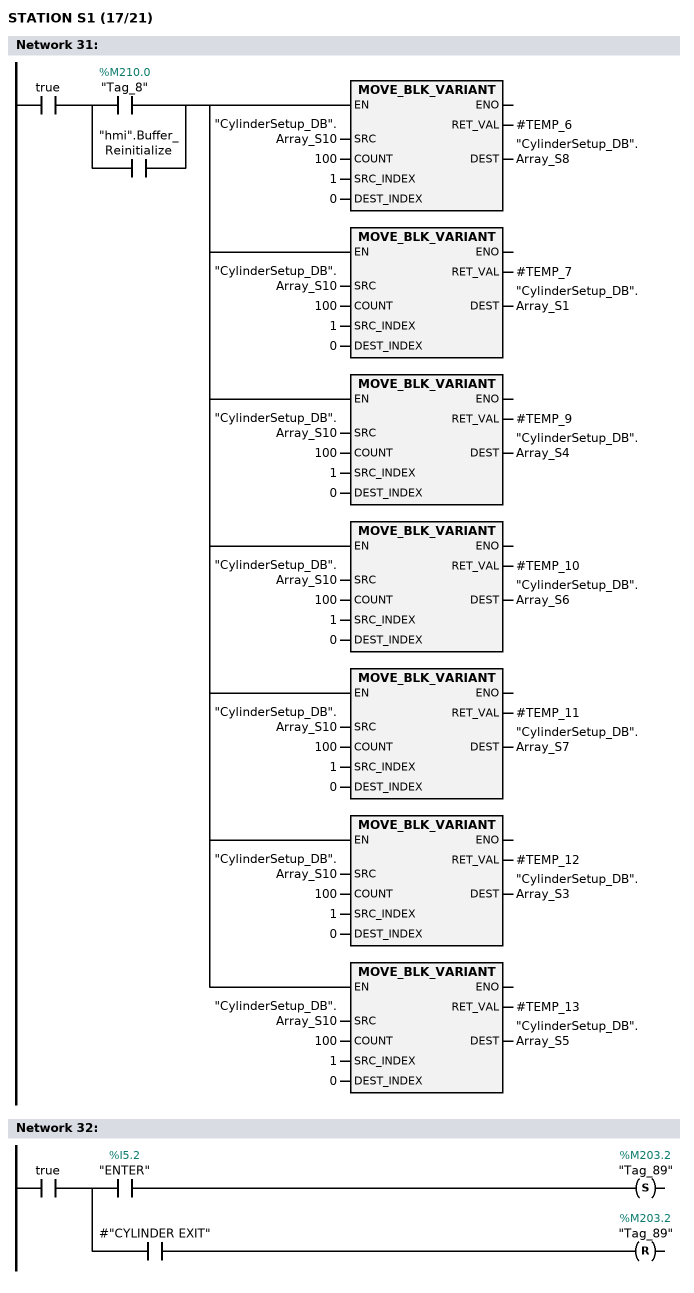
   RUNG wire#powerrail
      Contact( true )
      wire#w1
      Contact( "Tag_8" )
      wire#w2
      MOVE_BLK_VARIANT(SRC := "CylinderSetup_DB".Array_S10, COUNT := 100, SRC_INDEX := 1, DEST_INDEX := 0, Ret_Val => #TEMP_6, DEST => "CylinderSetup_DB".Array_S8)
   END_RUNG
   RUNG wire#w1
      Contact( "hmi".Buffer_Reinitialize )
   END_RUNG wire#w2
   RUNG wire#w2
      MOVE_BLK_VARIANT(SRC := "CylinderSetup_DB".Array_S10, COUNT := 100, SRC_INDEX := 1, DEST_INDEX := 0, Ret_Val => #TEMP_7, DEST => "CylinderSetup_DB".Array_S1)
   END_RUNG
   RUNG wire#w2
      MOVE_BLK_VARIANT(SRC := "CylinderSetup_DB".Array_S10, COUNT := 100, SRC_INDEX := 1, DEST_INDEX := 0, Ret_Val => #TEMP_9, DEST => "CylinderSetup_DB".Array_S4)
   END_RUNG
   RUNG wire#w2
      MOVE_BLK_VARIANT(SRC := "CylinderSetup_DB".Array_S10, COUNT := 100, SRC_INDEX := 1, DEST_INDEX := 0, Ret_Val => #TEMP_10, DEST => "CylinderSetup_DB".Array_S6)
   END_RUNG
   RUNG wire#w2
      MOVE_BLK_VARIANT(SRC := "CylinderSetup_DB".Array_S10, COUNT := 100, SRC_INDEX := 1, DEST_INDEX := 0, Ret_Val => #TEMP_11, DEST => "CylinderSetup_DB".Array_S7)
   END_RUNG
   RUNG wire#w2
      MOVE_BLK_VARIANT(SRC := "CylinderSetup_DB".Array_S10, COUNT := 100, SRC_INDEX := 1, DEST_INDEX := 0, Ret_Val => #TEMP_12, DEST => "CylinderSetup_DB".Array_S3)
   END_RUNG
   RUNG wire#w2
      MOVE_BLK_VARIANT(SRC := "CylinderSetup_DB".Array_S10, COUNT := 100, SRC_INDEX := 1, DEST_INDEX := 0, Ret_Val => #TEMP_13, DEST => "CylinderSetup_DB".Array_S5)
   END_RUNG
   // the same network as SCL:
   #_w1 := true AND ("Tag_8" OR "hmi".Buffer_Reinitialize);
   IF #_w1 THEN
       #TEMP_6 := MOVE_BLK_VARIANT(SRC := "CylinderSetup_DB".Array_S10,
                               COUNT := 100,
                               SRC_INDEX := 1,
                               DEST_INDEX := 0,
                               DEST => "CylinderSetup_DB".Array_S8);
       #TEMP_7 := MOVE_BLK_VARIANT(SRC := "CylinderSetup_DB".Array_S10,
                               COUNT := 100,
                               SRC_INDEX := 1,
                               DEST_INDEX := 0,
                               DEST => "CylinderSetup_DB".Array_S1);
       #TEMP_9 := MOVE_BLK_VARIANT(SRC := "CylinderSetup_DB".Array_S10,
                               COUNT := 100,
                               SRC_INDEX := 1,
                               DEST_INDEX := 0,
                               DEST => "CylinderSetup_DB".Array_S4);
       #TEMP_10 := MOVE_BLK_VARIANT(SRC := "CylinderSetup_DB".Array_S10,
                               COUNT := 100,
                               SRC_INDEX := 1,
                               DEST_INDEX := 0,
                               DEST => "CylinderSetup_DB".Array_S6);
       #TEMP_11 := MOVE_BLK_VARIANT(SRC := "CylinderSetup_DB".Array_S10,
                               COUNT := 100,
                               SRC_INDEX := 1,
                               DEST_INDEX := 0,
                               DEST => "CylinderSetup_DB".Array_S7);
       #TEMP_12 := MOVE_BLK_VARIANT(SRC := "CylinderSetup_DB".Array_S10,
                               COUNT := 100,
                               SRC_INDEX := 1,
                               DEST_INDEX := 0,
                               DEST => "CylinderSetup_DB".Array_S3);
       #TEMP_13 := MOVE_BLK_VARIANT(SRC := "CylinderSetup_DB".Array_S10,
                               COUNT := 100,
                               SRC_INDEX := 1,
                               DEST_INDEX := 0,
                               DEST => "CylinderSetup_DB".Array_S5);
   END_IF;
END_REGION

REGION Network 32
   RUNG wire#powerrail
      Contact( true )
      wire#w1
      Contact( "ENTER" )
      S_Coil( "Tag_89" )
   END_RUNG
   RUNG wire#w1
      Contact( #"CYLINDER EXIT" )
      R_Coil( "Tag_89" )
   END_RUNG
   // the same network as SCL:
   IF true AND "ENTER" THEN "Tag_89" := TRUE; END_IF;
   IF true AND #"CYLINDER EXIT" THEN "Tag_89" := FALSE; END_IF;
END_REGION

REGION Network 33
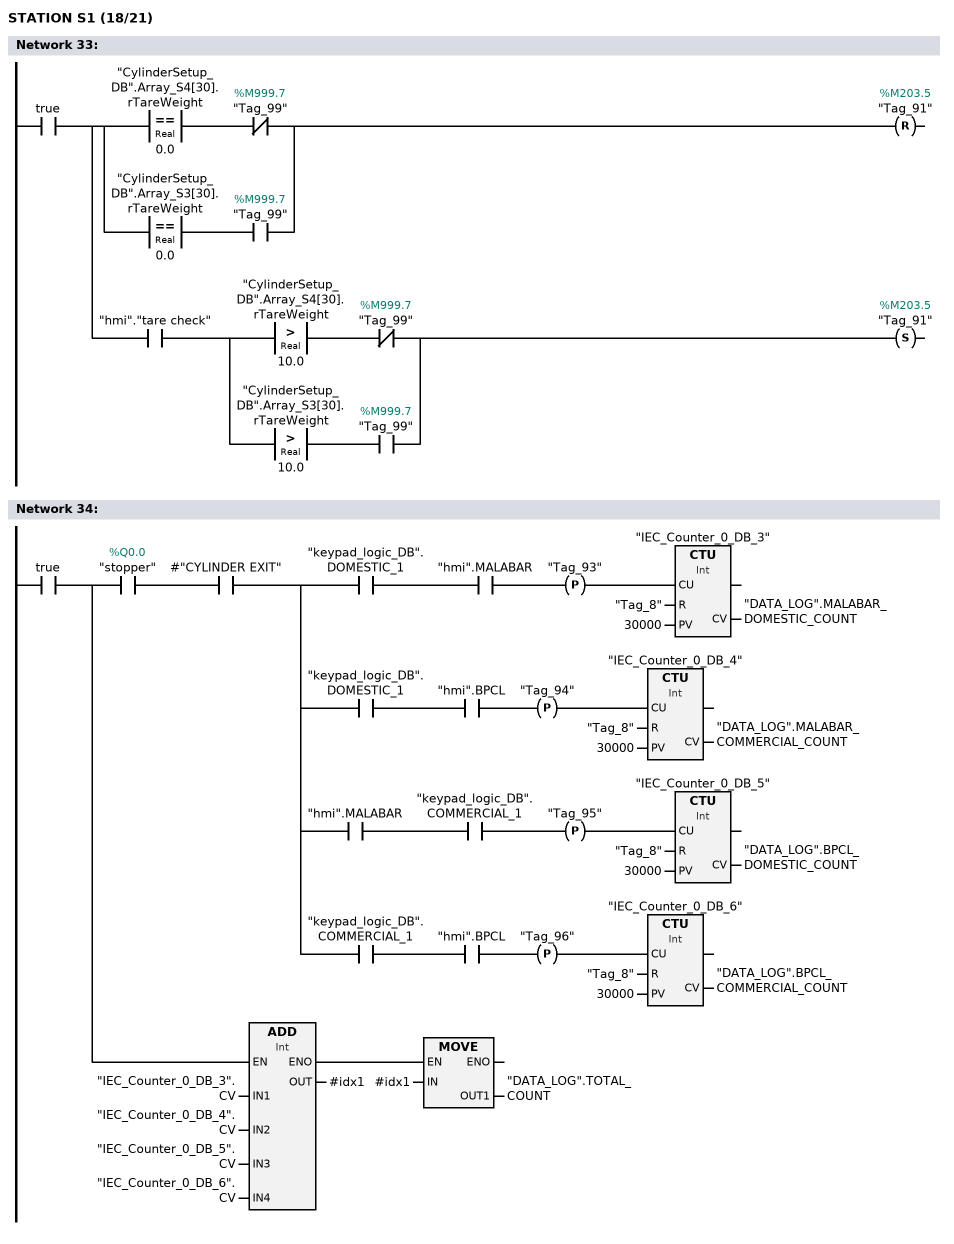
   RUNG wire#powerrail
      Contact( true )
      wire#w1
      { S7_Templates := "SrcType := Real" } EQ_Contact(in1 := "CylinderSetup_DB".Array_S4[30].rTareWeight, in2 := 0.0)
      I_Contact( "Tag_99" )
      wire#w2
      R_Coil( "Tag_91" )
   END_RUNG
   RUNG wire#w1
      { S7_Templates := "SrcType := Real" } EQ_Contact(in1 := "CylinderSetup_DB".Array_S3[30].rTareWeight, in2 := 0.0)
      Contact( "Tag_99" )
   END_RUNG wire#w2
   RUNG wire#w1
      Contact( "hmi"."tare check" )
      wire#w3
      { S7_Templates := "SrcType := Real" } GT_Contact(in1 := "CylinderSetup_DB".Array_S4[30].rTareWeight, in2 := 10.0)
      I_Contact( "Tag_99" )
      wire#w4
      S_Coil( "Tag_91" )
   END_RUNG
   RUNG wire#w3
      { S7_Templates := "SrcType := Real" } GT_Contact(in1 := "CylinderSetup_DB".Array_S3[30].rTareWeight, in2 := 10.0)
      Contact( "Tag_99" )
   END_RUNG wire#w4
   // the same network as SCL:
   IF true AND ((("CylinderSetup_DB".Array_S4[30].rTareWeight = 0.0) AND NOT "Tag_99") OR (("CylinderSetup_DB".Array_S3[30].rTareWeight = 0.0) AND "Tag_99")) THEN
       "Tag_91" := FALSE;
   END_IF;
   IF true AND "hmi"."tare check" AND ((("CylinderSetup_DB".Array_S4[30].rTareWeight > 10.0) AND NOT "Tag_99") OR (("CylinderSetup_DB".Array_S3[30].rTareWeight > 10.0) AND "Tag_99")) THEN
       "Tag_91" := TRUE;
   END_IF;
END_REGION

REGION Network 34
   RUNG wire#powerrail
      Contact( true )
      wire#w1
      Contact( "stopper" )
      Contact( #"CYLINDER EXIT" )
      wire#w2
      Contact( "keypad_logic_DB".DOMESTIC_1 )
      Contact( "hmi".MALABAR )
      P_Trig( "Tag_93" )
      { S7_Templates := "value_type := Int" } "IEC_Counter_0_DB_3".CTU(r := "Tag_8", pv := 30000, cv => "DATA_LOG".MALABAR_DOMESTIC_COUNT)
   END_RUNG
   RUNG wire#w2
      Contact( "keypad_logic_DB".DOMESTIC_1 )
      Contact( "hmi".BPCL )
      P_Trig( "Tag_94" )
      { S7_Templates := "value_type := Int" } "IEC_Counter_0_DB_4".CTU(r := "Tag_8", pv := 30000, cv => "DATA_LOG".MALABAR_COMMERCIAL_COUNT)
   END_RUNG
   RUNG wire#w2
      Contact( "hmi".MALABAR )
      Contact( "keypad_logic_DB".COMMERCIAL_1 )
      P_Trig( "Tag_95" )
      { S7_Templates := "value_type := Int" } "IEC_Counter_0_DB_5".CTU(r := "Tag_8", pv := 30000, cv => "DATA_LOG".BPCL_DOMESTIC_COUNT)
   END_RUNG
   RUNG wire#w2
      Contact( "keypad_logic_DB".COMMERCIAL_1 )
      Contact( "hmi".BPCL )
      P_Trig( "Tag_96" )
      { S7_Templates := "value_type := Int" } "IEC_Counter_0_DB_6".CTU(r := "Tag_8", pv := 30000, cv => "DATA_LOG".BPCL_COMMERCIAL_COUNT)
   END_RUNG
   RUNG wire#w1
      { S7_Templates := "SrcType := Int" } Add(in1 := "IEC_Counter_0_DB_3".CV, in2 := "IEC_Counter_0_DB_4".CV, in3 := "IEC_Counter_0_DB_5".CV, in4 := "IEC_Counter_0_DB_6".CV, out => #idx1)
      Move(in := #idx1, out1 => "DATA_LOG".TOTAL_COUNT)
   END_RUNG
   // the same network as SCL:
   #_w1 := true AND "stopper" AND #"CYLINDER EXIT";
   #_w2 := #_w1 AND "keypad_logic_DB".DOMESTIC_1 AND "hmi".MALABAR;
   #_w3 := #_w2 AND NOT "Tag_93";   // rising edge
   "Tag_93" := #_w2;
   "IEC_Counter_0_DB_3".CTU(CU := #_w3, R := "Tag_8", PV := 30000, CV => "DATA_LOG".MALABAR_DOMESTIC_COUNT);
   #_w4 := #_w1 AND "keypad_logic_DB".DOMESTIC_1 AND "hmi".BPCL;
   #_w5 := #_w4 AND NOT "Tag_94";   // rising edge
   "Tag_94" := #_w4;
   "IEC_Counter_0_DB_4".CTU(CU := #_w5, R := "Tag_8", PV := 30000, CV => "DATA_LOG".MALABAR_COMMERCIAL_COUNT);
   #_w6 := #_w1 AND "hmi".MALABAR AND "keypad_logic_DB".COMMERCIAL_1;
   #_w7 := #_w6 AND NOT "Tag_95";   // rising edge
   "Tag_95" := #_w6;
   "IEC_Counter_0_DB_5".CTU(CU := #_w7, R := "Tag_8", PV := 30000, CV => "DATA_LOG".BPCL_DOMESTIC_COUNT);
   #_w8 := #_w1 AND "keypad_logic_DB".COMMERCIAL_1 AND "hmi".BPCL;
   #_w9 := #_w8 AND NOT "Tag_96";   // rising edge
   "Tag_96" := #_w8;
   "IEC_Counter_0_DB_6".CTU(CU := #_w9, R := "Tag_8", PV := 30000, CV => "DATA_LOG".BPCL_COMMERCIAL_COUNT);
   IF true THEN
       #idx1 := "IEC_Counter_0_DB_3".CV + "IEC_Counter_0_DB_4".CV + "IEC_Counter_0_DB_5".CV + "IEC_Counter_0_DB_6".CV;
       "DATA_LOG".TOTAL_COUNT := #idx1;
   END_IF;
END_REGION

REGION Network 35: L1 TOTAL NET WT
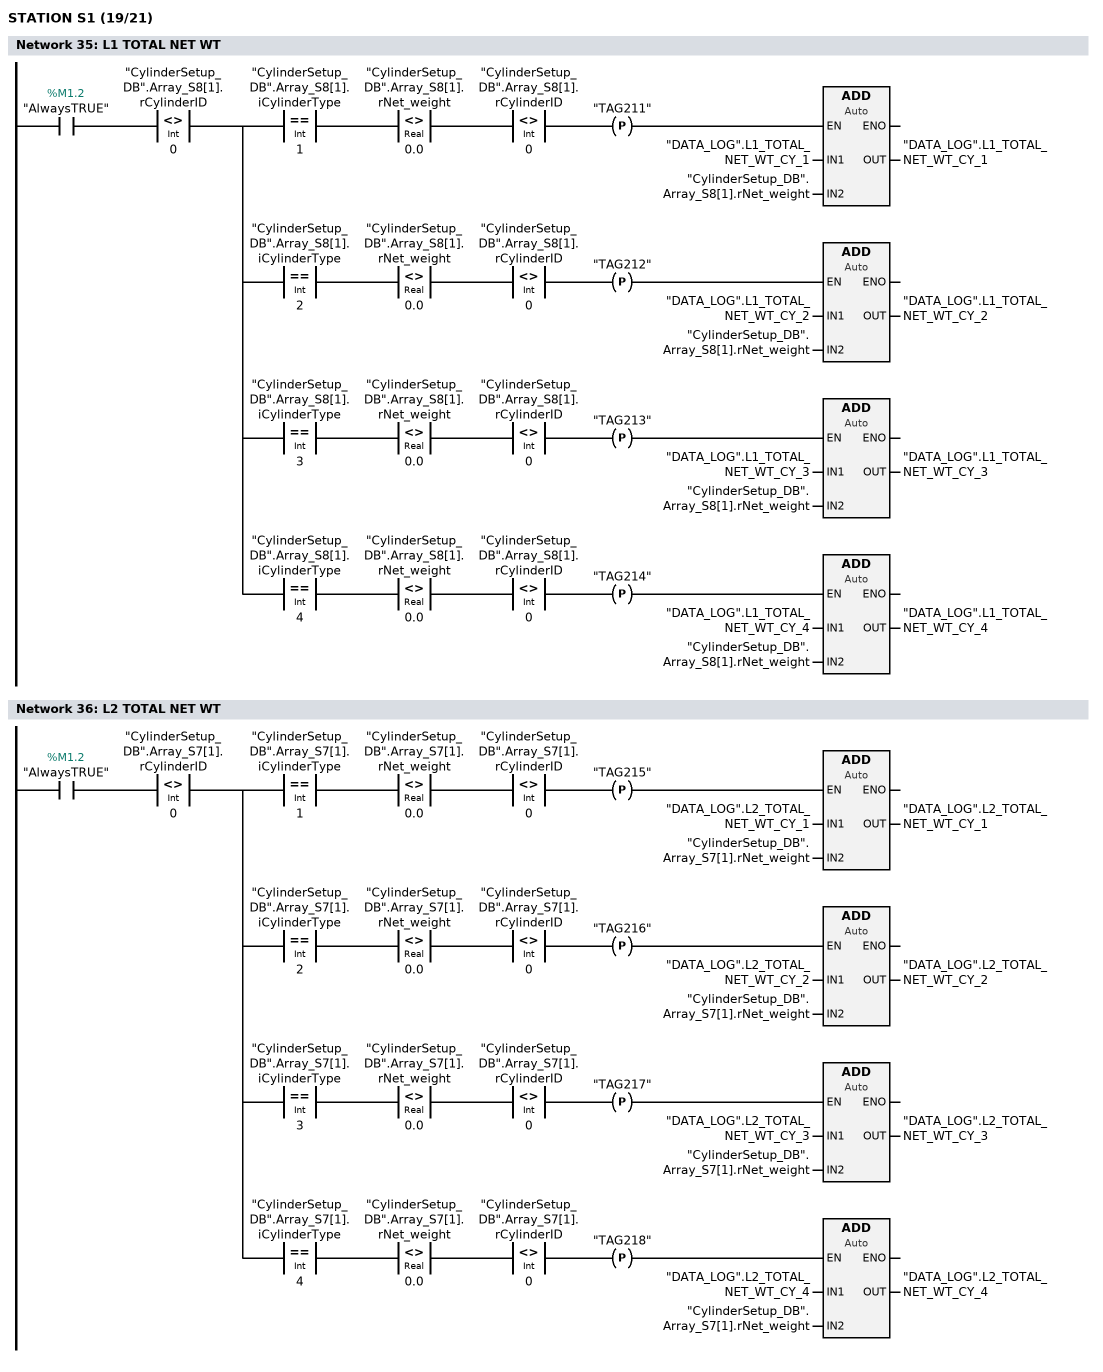
   RUNG wire#powerrail
      Contact( "AlwaysTRUE" )
      { S7_Templates := "SrcType := Int" } NE_Contact(in1 := "CylinderSetup_DB".Array_S8[1].rCylinderID, in2 := 0)
      wire#w1
      { S7_Templates := "SrcType := Int" } EQ_Contact(in1 := "CylinderSetup_DB".Array_S8[1].iCylinderType, in2 := 1)
      { S7_Templates := "SrcType := Real" } NE_Contact(in1 := "CylinderSetup_DB".Array_S8[1].rNet_weight, in2 := 0.0)
      { S7_Templates := "SrcType := Int" } NE_Contact(in1 := "CylinderSetup_DB".Array_S8[1].rCylinderID, in2 := 0)
      P_Trig( "TAG211" )
      Add(in1 := "DATA_LOG".L1_TOTAL_NET_WT_CY_1, in2 := "CylinderSetup_DB".Array_S8[1].rNet_weight, out => "DATA_LOG".L1_TOTAL_NET_WT_CY_1)
   END_RUNG
   RUNG wire#w1
      { S7_Templates := "SrcType := Int" } EQ_Contact(in1 := "CylinderSetup_DB".Array_S8[1].iCylinderType, in2 := 2)
      { S7_Templates := "SrcType := Real" } NE_Contact(in1 := "CylinderSetup_DB".Array_S8[1].rNet_weight, in2 := 0.0)
      { S7_Templates := "SrcType := Int" } NE_Contact(in1 := "CylinderSetup_DB".Array_S8[1].rCylinderID, in2 := 0)
      P_Trig( "TAG212" )
      Add(in1 := "DATA_LOG".L1_TOTAL_NET_WT_CY_2, in2 := "CylinderSetup_DB".Array_S8[1].rNet_weight, out => "DATA_LOG".L1_TOTAL_NET_WT_CY_2)
   END_RUNG
   RUNG wire#w1
      { S7_Templates := "SrcType := Int" } EQ_Contact(in1 := "CylinderSetup_DB".Array_S8[1].iCylinderType, in2 := 3)
      { S7_Templates := "SrcType := Real" } NE_Contact(in1 := "CylinderSetup_DB".Array_S8[1].rNet_weight, in2 := 0.0)
      { S7_Templates := "SrcType := Int" } NE_Contact(in1 := "CylinderSetup_DB".Array_S8[1].rCylinderID, in2 := 0)
      P_Trig( "TAG213" )
      Add(in1 := "DATA_LOG".L1_TOTAL_NET_WT_CY_3, in2 := "CylinderSetup_DB".Array_S8[1].rNet_weight, out => "DATA_LOG".L1_TOTAL_NET_WT_CY_3)
   END_RUNG
   RUNG wire#w1
      { S7_Templates := "SrcType := Int" } EQ_Contact(in1 := "CylinderSetup_DB".Array_S8[1].iCylinderType, in2 := 4)
      { S7_Templates := "SrcType := Real" } NE_Contact(in1 := "CylinderSetup_DB".Array_S8[1].rNet_weight, in2 := 0.0)
      { S7_Templates := "SrcType := Int" } NE_Contact(in1 := "CylinderSetup_DB".Array_S8[1].rCylinderID, in2 := 0)
      P_Trig( "TAG214" )
      Add(in1 := "DATA_LOG".L1_TOTAL_NET_WT_CY_4, in2 := "CylinderSetup_DB".Array_S8[1].rNet_weight, out => "DATA_LOG".L1_TOTAL_NET_WT_CY_4)
   END_RUNG
   // the same network as SCL:
   #_w1 := "AlwaysTRUE" AND ("CylinderSetup_DB".Array_S8[1].rCylinderID <> 0);
   #_w2 := #_w1 AND ("CylinderSetup_DB".Array_S8[1].iCylinderType = 1) AND ("CylinderSetup_DB".Array_S8[1].rNet_weight <> 0.0) AND ("CylinderSetup_DB".Array_S8[1].rCylinderID <> 0);
   #_w3 := #_w2 AND NOT "TAG211";   // rising edge
   "TAG211" := #_w2;
   IF #_w3 THEN
       "DATA_LOG".L1_TOTAL_NET_WT_CY_1 := "DATA_LOG".L1_TOTAL_NET_WT_CY_1 + "CylinderSetup_DB".Array_S8[1].rNet_weight;
   END_IF;
   #_w4 := #_w1 AND ("CylinderSetup_DB".Array_S8[1].iCylinderType = 2) AND ("CylinderSetup_DB".Array_S8[1].rNet_weight <> 0.0) AND ("CylinderSetup_DB".Array_S8[1].rCylinderID <> 0);
   #_w5 := #_w4 AND NOT "TAG212";   // rising edge
   "TAG212" := #_w4;
   IF #_w5 THEN
       "DATA_LOG".L1_TOTAL_NET_WT_CY_2 := "DATA_LOG".L1_TOTAL_NET_WT_CY_2 + "CylinderSetup_DB".Array_S8[1].rNet_weight;
   END_IF;
   #_w6 := #_w1 AND ("CylinderSetup_DB".Array_S8[1].iCylinderType = 3) AND ("CylinderSetup_DB".Array_S8[1].rNet_weight <> 0.0) AND ("CylinderSetup_DB".Array_S8[1].rCylinderID <> 0);
   #_w7 := #_w6 AND NOT "TAG213";   // rising edge
   "TAG213" := #_w6;
   IF #_w7 THEN
       "DATA_LOG".L1_TOTAL_NET_WT_CY_3 := "DATA_LOG".L1_TOTAL_NET_WT_CY_3 + "CylinderSetup_DB".Array_S8[1].rNet_weight;
   END_IF;
   #_w8 := #_w1 AND ("CylinderSetup_DB".Array_S8[1].iCylinderType = 4) AND ("CylinderSetup_DB".Array_S8[1].rNet_weight <> 0.0) AND ("CylinderSetup_DB".Array_S8[1].rCylinderID <> 0);
   #_w9 := #_w8 AND NOT "TAG214";   // rising edge
   "TAG214" := #_w8;
   IF #_w9 THEN
       "DATA_LOG".L1_TOTAL_NET_WT_CY_4 := "DATA_LOG".L1_TOTAL_NET_WT_CY_4 + "CylinderSetup_DB".Array_S8[1].rNet_weight;
   END_IF;
END_REGION

REGION Network 36: L2 TOTAL NET WT
   RUNG wire#powerrail
      Contact( "AlwaysTRUE" )
      { S7_Templates := "SrcType := Int" } NE_Contact(in1 := "CylinderSetup_DB".Array_S7[1].rCylinderID, in2 := 0)
      wire#w1
      { S7_Templates := "SrcType := Int" } EQ_Contact(in1 := "CylinderSetup_DB".Array_S7[1].iCylinderType, in2 := 1)
      { S7_Templates := "SrcType := Real" } NE_Contact(in1 := "CylinderSetup_DB".Array_S7[1].rNet_weight, in2 := 0.0)
      { S7_Templates := "SrcType := Int" } NE_Contact(in1 := "CylinderSetup_DB".Array_S7[1].rCylinderID, in2 := 0)
      P_Trig( "TAG215" )
      Add(in1 := "DATA_LOG".L2_TOTAL_NET_WT_CY_1, in2 := "CylinderSetup_DB".Array_S7[1].rNet_weight, out => "DATA_LOG".L2_TOTAL_NET_WT_CY_1)
   END_RUNG
   RUNG wire#w1
      { S7_Templates := "SrcType := Int" } EQ_Contact(in1 := "CylinderSetup_DB".Array_S7[1].iCylinderType, in2 := 2)
      { S7_Templates := "SrcType := Real" } NE_Contact(in1 := "CylinderSetup_DB".Array_S7[1].rNet_weight, in2 := 0.0)
      { S7_Templates := "SrcType := Int" } NE_Contact(in1 := "CylinderSetup_DB".Array_S7[1].rCylinderID, in2 := 0)
      P_Trig( "TAG216" )
      Add(in1 := "DATA_LOG".L2_TOTAL_NET_WT_CY_2, in2 := "CylinderSetup_DB".Array_S7[1].rNet_weight, out => "DATA_LOG".L2_TOTAL_NET_WT_CY_2)
   END_RUNG
   RUNG wire#w1
      { S7_Templates := "SrcType := Int" } EQ_Contact(in1 := "CylinderSetup_DB".Array_S7[1].iCylinderType, in2 := 3)
      { S7_Templates := "SrcType := Real" } NE_Contact(in1 := "CylinderSetup_DB".Array_S7[1].rNet_weight, in2 := 0.0)
      { S7_Templates := "SrcType := Int" } NE_Contact(in1 := "CylinderSetup_DB".Array_S7[1].rCylinderID, in2 := 0)
      P_Trig( "TAG217" )
      Add(in1 := "DATA_LOG".L2_TOTAL_NET_WT_CY_3, in2 := "CylinderSetup_DB".Array_S7[1].rNet_weight, out => "DATA_LOG".L2_TOTAL_NET_WT_CY_3)
   END_RUNG
   RUNG wire#w1
      { S7_Templates := "SrcType := Int" } EQ_Contact(in1 := "CylinderSetup_DB".Array_S7[1].iCylinderType, in2 := 4)
      { S7_Templates := "SrcType := Real" } NE_Contact(in1 := "CylinderSetup_DB".Array_S7[1].rNet_weight, in2 := 0.0)
      { S7_Templates := "SrcType := Int" } NE_Contact(in1 := "CylinderSetup_DB".Array_S7[1].rCylinderID, in2 := 0)
      P_Trig( "TAG218" )
      Add(in1 := "DATA_LOG".L2_TOTAL_NET_WT_CY_4, in2 := "CylinderSetup_DB".Array_S7[1].rNet_weight, out => "DATA_LOG".L2_TOTAL_NET_WT_CY_4)
   END_RUNG
   // the same network as SCL:
   #_w1 := "AlwaysTRUE" AND ("CylinderSetup_DB".Array_S7[1].rCylinderID <> 0);
   #_w2 := #_w1 AND ("CylinderSetup_DB".Array_S7[1].iCylinderType = 1) AND ("CylinderSetup_DB".Array_S7[1].rNet_weight <> 0.0) AND ("CylinderSetup_DB".Array_S7[1].rCylinderID <> 0);
   #_w3 := #_w2 AND NOT "TAG215";   // rising edge
   "TAG215" := #_w2;
   IF #_w3 THEN
       "DATA_LOG".L2_TOTAL_NET_WT_CY_1 := "DATA_LOG".L2_TOTAL_NET_WT_CY_1 + "CylinderSetup_DB".Array_S7[1].rNet_weight;
   END_IF;
   #_w4 := #_w1 AND ("CylinderSetup_DB".Array_S7[1].iCylinderType = 2) AND ("CylinderSetup_DB".Array_S7[1].rNet_weight <> 0.0) AND ("CylinderSetup_DB".Array_S7[1].rCylinderID <> 0);
   #_w5 := #_w4 AND NOT "TAG216";   // rising edge
   "TAG216" := #_w4;
   IF #_w5 THEN
       "DATA_LOG".L2_TOTAL_NET_WT_CY_2 := "DATA_LOG".L2_TOTAL_NET_WT_CY_2 + "CylinderSetup_DB".Array_S7[1].rNet_weight;
   END_IF;
   #_w6 := #_w1 AND ("CylinderSetup_DB".Array_S7[1].iCylinderType = 3) AND ("CylinderSetup_DB".Array_S7[1].rNet_weight <> 0.0) AND ("CylinderSetup_DB".Array_S7[1].rCylinderID <> 0);
   #_w7 := #_w6 AND NOT "TAG217";   // rising edge
   "TAG217" := #_w6;
   IF #_w7 THEN
       "DATA_LOG".L2_TOTAL_NET_WT_CY_3 := "DATA_LOG".L2_TOTAL_NET_WT_CY_3 + "CylinderSetup_DB".Array_S7[1].rNet_weight;
   END_IF;
   #_w8 := #_w1 AND ("CylinderSetup_DB".Array_S7[1].iCylinderType = 4) AND ("CylinderSetup_DB".Array_S7[1].rNet_weight <> 0.0) AND ("CylinderSetup_DB".Array_S7[1].rCylinderID <> 0);
   #_w9 := #_w8 AND NOT "TAG218";   // rising edge
   "TAG218" := #_w8;
   IF #_w9 THEN
       "DATA_LOG".L2_TOTAL_NET_WT_CY_4 := "DATA_LOG".L2_TOTAL_NET_WT_CY_4 + "CylinderSetup_DB".Array_S7[1].rNet_weight;
   END_IF;
END_REGION

REGION Network 37
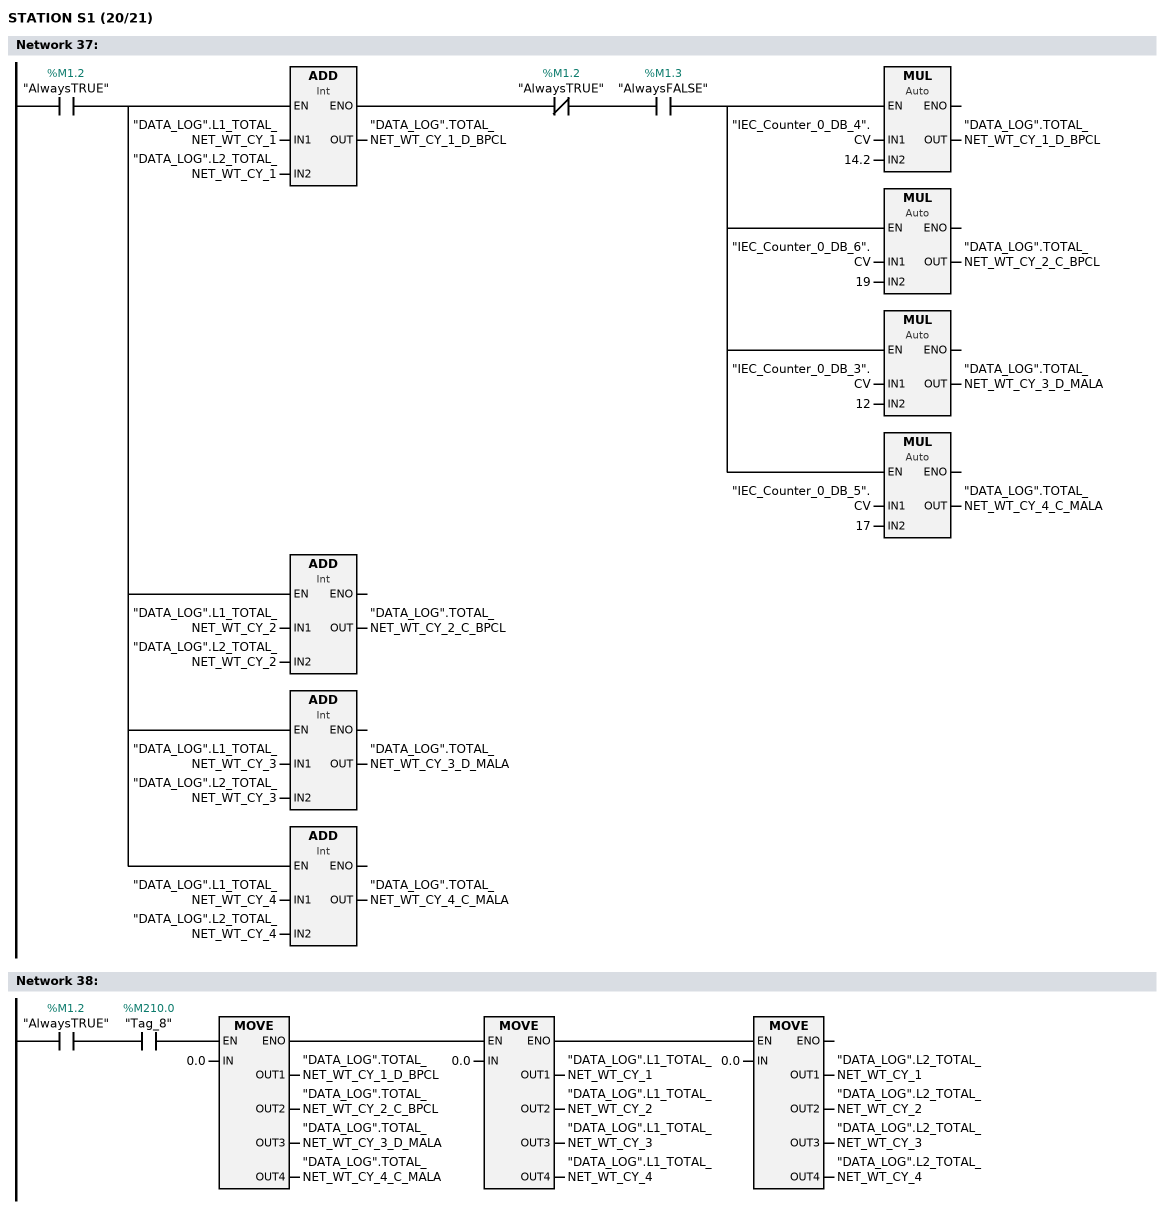
   RUNG wire#powerrail
      Contact( "AlwaysTRUE" )
      wire#w1
      { S7_Templates := "SrcType := Int" } Add(in1 := "DATA_LOG".L1_TOTAL_NET_WT_CY_1, in2 := "DATA_LOG".L2_TOTAL_NET_WT_CY_1, out => "DATA_LOG".TOTAL_NET_WT_CY_1_D_BPCL)
      I_Contact( "AlwaysTRUE" )
      Contact( "AlwaysFALSE" )
      wire#w2
      Mul(in1 := "IEC_Counter_0_DB_4".CV, in2 := 14.2, out => "DATA_LOG".TOTAL_NET_WT_CY_1_D_BPCL)
   END_RUNG
   RUNG wire#w2
      Mul(in1 := "IEC_Counter_0_DB_6".CV, in2 := 19, out => "DATA_LOG".TOTAL_NET_WT_CY_2_C_BPCL)
   END_RUNG
   RUNG wire#w2
      Mul(in1 := "IEC_Counter_0_DB_3".CV, in2 := 12, out => "DATA_LOG".TOTAL_NET_WT_CY_3_D_MALA)
   END_RUNG
   RUNG wire#w2
      Mul(in1 := "IEC_Counter_0_DB_5".CV, in2 := 17, out => "DATA_LOG".TOTAL_NET_WT_CY_4_C_MALA)
   END_RUNG
   RUNG wire#w1
      { S7_Templates := "SrcType := Int" } Add(in1 := "DATA_LOG".L1_TOTAL_NET_WT_CY_2, in2 := "DATA_LOG".L2_TOTAL_NET_WT_CY_2, out => "DATA_LOG".TOTAL_NET_WT_CY_2_C_BPCL)
   END_RUNG
   RUNG wire#w1
      { S7_Templates := "SrcType := Int" } Add(in1 := "DATA_LOG".L1_TOTAL_NET_WT_CY_3, in2 := "DATA_LOG".L2_TOTAL_NET_WT_CY_3, out => "DATA_LOG".TOTAL_NET_WT_CY_3_D_MALA)
   END_RUNG
   RUNG wire#w1
      { S7_Templates := "SrcType := Int" } Add(in1 := "DATA_LOG".L1_TOTAL_NET_WT_CY_4, in2 := "DATA_LOG".L2_TOTAL_NET_WT_CY_4, out => "DATA_LOG".TOTAL_NET_WT_CY_4_C_MALA)
   END_RUNG
   // the same network as SCL:
   IF "AlwaysTRUE" THEN
       "DATA_LOG".TOTAL_NET_WT_CY_1_D_BPCL := "DATA_LOG".L1_TOTAL_NET_WT_CY_1 + "DATA_LOG".L2_TOTAL_NET_WT_CY_1;
   END_IF;
   IF "AlwaysTRUE" AND NOT "AlwaysTRUE" AND "AlwaysFALSE" THEN
       "DATA_LOG".TOTAL_NET_WT_CY_1_D_BPCL := "IEC_Counter_0_DB_4".CV * 14.2;
       "DATA_LOG".TOTAL_NET_WT_CY_2_C_BPCL := "IEC_Counter_0_DB_6".CV * 19;
       "DATA_LOG".TOTAL_NET_WT_CY_3_D_MALA := "IEC_Counter_0_DB_3".CV * 12;
       "DATA_LOG".TOTAL_NET_WT_CY_4_C_MALA := "IEC_Counter_0_DB_5".CV * 17;
   END_IF;
   IF "AlwaysTRUE" THEN
       "DATA_LOG".TOTAL_NET_WT_CY_2_C_BPCL := "DATA_LOG".L1_TOTAL_NET_WT_CY_2 + "DATA_LOG".L2_TOTAL_NET_WT_CY_2;
       "DATA_LOG".TOTAL_NET_WT_CY_3_D_MALA := "DATA_LOG".L1_TOTAL_NET_WT_CY_3 + "DATA_LOG".L2_TOTAL_NET_WT_CY_3;
       "DATA_LOG".TOTAL_NET_WT_CY_4_C_MALA := "DATA_LOG".L1_TOTAL_NET_WT_CY_4 + "DATA_LOG".L2_TOTAL_NET_WT_CY_4;
   END_IF;
END_REGION

REGION Network 38
   RUNG wire#powerrail
      Contact( "AlwaysTRUE" )
      Contact( "Tag_8" )
      Move(in := 0.0, out1 => "DATA_LOG".TOTAL_NET_WT_CY_1_D_BPCL, out2 => "DATA_LOG".TOTAL_NET_WT_CY_2_C_BPCL, out3 => "DATA_LOG".TOTAL_NET_WT_CY_3_D_MALA, out4 => "DATA_LOG".TOTAL_NET_WT_CY_4_C_MALA)
      Move(in := 0.0, out1 => "DATA_LOG".L1_TOTAL_NET_WT_CY_1, out2 => "DATA_LOG".L1_TOTAL_NET_WT_CY_2, out3 => "DATA_LOG".L1_TOTAL_NET_WT_CY_3, out4 => "DATA_LOG".L1_TOTAL_NET_WT_CY_4)
      Move(in := 0.0, out1 => "DATA_LOG".L2_TOTAL_NET_WT_CY_1, out2 => "DATA_LOG".L2_TOTAL_NET_WT_CY_2, out3 => "DATA_LOG".L2_TOTAL_NET_WT_CY_3, out4 => "DATA_LOG".L2_TOTAL_NET_WT_CY_4)
   END_RUNG
   // the same network as SCL:
   IF "AlwaysTRUE" AND "Tag_8" THEN
       "DATA_LOG".TOTAL_NET_WT_CY_1_D_BPCL := 0.0;
       "DATA_LOG".TOTAL_NET_WT_CY_2_C_BPCL := 0.0;
       "DATA_LOG".TOTAL_NET_WT_CY_3_D_MALA := 0.0;
       "DATA_LOG".TOTAL_NET_WT_CY_4_C_MALA := 0.0;
       "DATA_LOG".L1_TOTAL_NET_WT_CY_1 := 0.0;
       "DATA_LOG".L1_TOTAL_NET_WT_CY_2 := 0.0;
       "DATA_LOG".L1_TOTAL_NET_WT_CY_3 := 0.0;
       "DATA_LOG".L1_TOTAL_NET_WT_CY_4 := 0.0;
       "DATA_LOG".L2_TOTAL_NET_WT_CY_1 := 0.0;
       "DATA_LOG".L2_TOTAL_NET_WT_CY_2 := 0.0;
       "DATA_LOG".L2_TOTAL_NET_WT_CY_3 := 0.0;
       "DATA_LOG".L2_TOTAL_NET_WT_CY_4 := 0.0;
   END_IF;
END_REGION

REGION Network 39: filled CYL data to check scale data
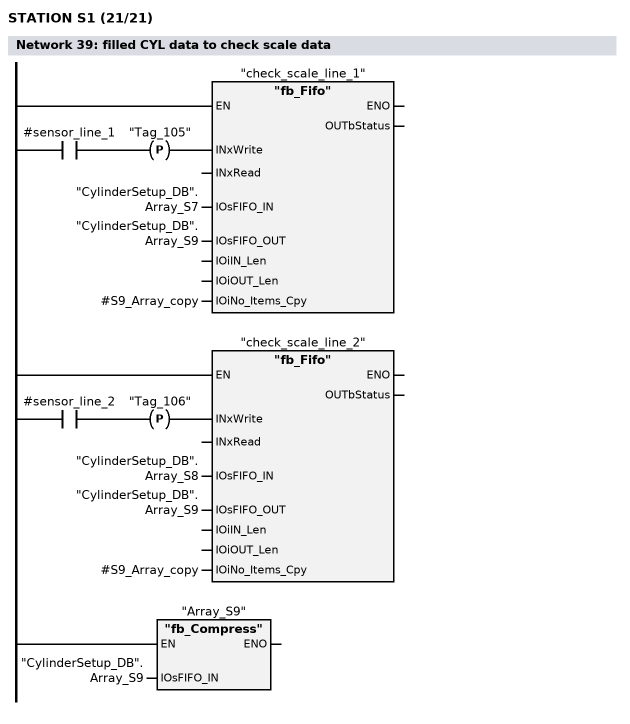
   RUNG wire#powerrail
      "check_scale_line_1"(INxWrite := wire#w1, INxRead :=, IOsFIFO_IN := "CylinderSetup_DB".Array_S7, IOsFIFO_OUT := "CylinderSetup_DB".Array_S9, IOiIN_Len :=, IOiOUT_Len :=, IOiNo_Items_Cpy := #S9_Array_copy, OUTbStatus =>)
   END_RUNG
   RUNG wire#powerrail
      Contact( #sensor_line_1 )
      P_Trig( "Tag_105" )
   END_RUNG wire#w1
   RUNG wire#powerrail
      "check_scale_line_2"(INxWrite := wire#w2, INxRead :=, IOsFIFO_IN := "CylinderSetup_DB".Array_S8, IOsFIFO_OUT := "CylinderSetup_DB".Array_S9, IOiIN_Len :=, IOiOUT_Len :=, IOiNo_Items_Cpy := #S9_Array_copy, OUTbStatus =>)
   END_RUNG
   RUNG wire#powerrail
      Contact( #sensor_line_2 )
      P_Trig( "Tag_106" )
   END_RUNG wire#w2
   RUNG wire#powerrail
      "Array_S9"(IOsFIFO_IN := "CylinderSetup_DB".Array_S9)
   END_RUNG
   // the same network as SCL:
   #_w1 := #sensor_line_1 AND NOT "Tag_105";   // rising edge
   "Tag_105" := #sensor_line_1;
   "check_scale_line_1"(INxWrite := #_w1,   // "fb_Fifo"
                        IOsFIFO_IN := "CylinderSetup_DB".Array_S7,
                        IOsFIFO_OUT := "CylinderSetup_DB".Array_S9,
                        IOiNo_Items_Cpy := #S9_Array_copy);
   #_w2 := #sensor_line_2 AND NOT "Tag_106";   // rising edge
   "Tag_106" := #sensor_line_2;
   "check_scale_line_2"(INxWrite := #_w2,   // "fb_Fifo"
                        IOsFIFO_IN := "CylinderSetup_DB".Array_S8,
                        IOsFIFO_OUT := "CylinderSetup_DB".Array_S9,
                        IOiNo_Items_Cpy := #S9_Array_copy);
   "Array_S9"(IOsFIFO_IN := "CylinderSetup_DB".Array_S9);   // "fb_Compress"
END_REGION
END_FUNCTION

FUNCTION_BLOCK "fb_Compress"
{ S7_Optimized_Access := 'TRUE' }
VERSION : 0.1
   VAR_IN_OUT 
      IOsFIFO_IN : Array[1..50] of "uCylinderData";
   END_VAR

   VAR 
      sEmpty { S7_SetPoint := 'False'} : "uCylinderData";
      idx1 { S7_SetPoint := 'True'} : Int;
   END_VAR


BEGIN
	FOR #idx1 := 1 TO 50 - 1 DO
	    IF #idx1 <= 0 THEN
	        EXIT;
	    END_IF;
	    // Shift down FiFo by one
	    IF #IOsFIFO_IN[#idx1].rCylinderID = 0.0 AND
	        #IOsFIFO_IN[#idx1 + 1].rCylinderID <> 0.0 THEN
	        #IOsFIFO_IN[#idx1] := #IOsFIFO_IN[#idx1 + 1];
	        #IOsFIFO_IN[#idx1 + 1] := #sEmpty;
	    END_IF;
	END_FOR;
END_FUNCTION_BLOCK

FUNCTION_BLOCK "fb_Fifo"
{ S7_Optimized_Access := 'TRUE' }
VERSION : 0.1
   VAR_INPUT 
      INxWrite : Bool;
      INxRead : Bool;
   END_VAR

   VAR_OUTPUT 
      OUTbStatus : Byte;   // Status Ok - 1, Status Overflow at output - 2, Status Input Empty - 3
   END_VAR

   VAR_IN_OUT 
      IOsFIFO_IN : Array[1..50] of "uCylinderData";
      IOsFIFO_OUT : Array[1..50] of "uCylinderData";
      IOiIN_Len : Int;
      IOiOUT_Len : Int;
      IOiNo_Items_Cpy : Int;
   END_VAR

   VAR 
      idx1 { S7_SetPoint := 'True'} : Int;
      idx2 { S7_SetPoint := 'True'} : Int;
      idx3 { S7_SetPoint := 'True'} : Int;
      idx4 : Int;
      sEmpty { S7_SetPoint := 'False'} : "uCylinderData";
   END_VAR


BEGIN
	//Initialization
	#IOiIN_Len := 0;
	#IOiOUT_Len := 0;
	
	
	//Check Input FIFO Lengeth
	FOR #idx1 := 1 TO 50 DO
	    IF #IOsFIFO_IN[#idx1].rCylinderID <> 0.0 THEN
	        #IOiIN_Len := #IOiIN_Len + 1;
	    END_IF;
	END_FOR;
	
	//Check Output FIFO Lengeth
	FOR #idx2 := 1 TO 50 DO
	    IF #IOsFIFO_OUT[#idx2].rCylinderID <> 0.0 THEN
	        #IOiOUT_Len := #IOiOUT_Len + 1;
	    END_IF;
	END_FOR;
	
	
	//Write data into output FIFO from input FIFO
	IF #INxWrite THEN
	    #OUTbStatus := 0; //Initialise status
	    IF #IOiIN_Len <> 0 AND #IOiOUT_Len <= 49 THEN
	        //Copy Data into output FIFO
	        WHILE #IOiNo_Items_Cpy <> 0 DO
	            #IOsFIFO_OUT[49] := #IOsFIFO_IN[1]; //Copy Data into output FIFO
	            #IOsFIFO_IN[1] := #sEmpty; //Delete Copied data in input FIFO
	            //Compress Input FIFO
	            FOR #idx4 := 1 TO 50 - 1 DO
	                IF #idx4 <= 0 THEN
	                    EXIT;
	                END_IF;
	                // Shift down FiFo by one
	                IF #IOsFIFO_OUT[#idx4].rCylinderID = 0.0 AND
	                    #IOsFIFO_OUT[#idx4 + 1].rCylinderID <> 0.0 THEN
	                    #IOsFIFO_OUT[#idx4] := #IOsFIFO_OUT[#idx4 + 1];
	                    #IOsFIFO_OUT[#idx4 + 1] := #sEmpty;
	                END_IF;
	            END_FOR;
	            //Compress Output FIFO
	            FOR #idx3 := 1 TO 50 - 1 DO
	                IF #idx3 <= 0 THEN
	                    EXIT;
	                END_IF;
	                // Shift down FiFo by one
	                IF #IOsFIFO_IN[#idx3].rCylinderID = 0.0 AND
	                    #IOsFIFO_IN[#idx3 + 1].rCylinderID <> 0.0 THEN
	                    #IOsFIFO_IN[#idx3] := #IOsFIFO_IN[#idx3 + 1];
	                    #IOsFIFO_IN[#idx3 + 1] := #sEmpty;
	                END_IF;
	            END_FOR;
	            #IOiNo_Items_Cpy := #IOiNo_Items_Cpy - 1; //Move to Next Item in the FIFO
	        END_WHILE;
	        #OUTbStatus := 1;
	    ELSIF #IOiIN_Len = 0 THEN
	        #OUTbStatus := 3;
	    ELSIF #IOiOUT_Len > 49 THEN
	        #OUTbStatus := 2;
	    END_IF;
	END_IF;
	
	
	
	
	
	
	
	
END_FUNCTION_BLOCK

FUNCTION "MODTCP_STN4_FC" : Void   // FC100, LAD
{ S7_Optimized_Access := 'TRUE' }
VERSION : 0.1
// stored: AutoNumber false, IsIECCheckEnabled false, SetENOAutomatically false, UDAEnableTagReadback false
BEGIN

REGION Network 2: Call Filling Line-1 Station-1
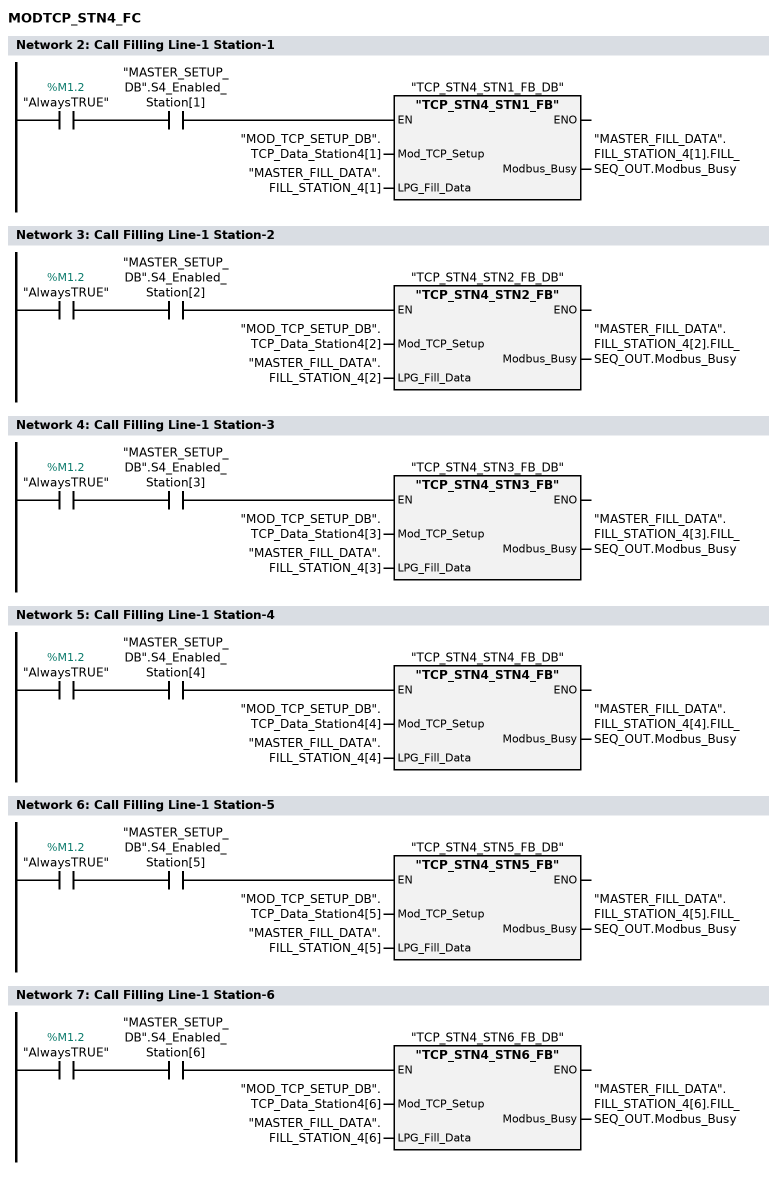
   RUNG wire#powerrail
      Contact( "AlwaysTRUE" )
      Contact( "MASTER_SETUP_DB".S4_Enabled_Station[1] )
      "TCP_STN4_STN1_FB_DB"(Mod_TCP_Setup := "MOD_TCP_SETUP_DB".TCP_Data_Station4[1], LPG_Fill_Data := "MASTER_FILL_DATA".FILL_STATION_4[1], Modbus_Busy => "MASTER_FILL_DATA".FILL_STATION_4[1].FILL_SEQ_OUT.Modbus_Busy)
   END_RUNG
   // the same network as SCL:
   IF "AlwaysTRUE" AND "MASTER_SETUP_DB".S4_Enabled_Station[1] THEN
       "TCP_STN4_STN1_FB_DB"(Mod_TCP_Setup := "MOD_TCP_SETUP_DB".TCP_Data_Station4[1],   // "TCP_STN4_STN1_FB"
                             LPG_Fill_Data := "MASTER_FILL_DATA".FILL_STATION_4[1],
                             Modbus_Busy => "MASTER_FILL_DATA".FILL_STATION_4[1].FILL_SEQ_OUT.Modbus_Busy);
   END_IF;
END_REGION

REGION Network 3: Call Filling Line-1 Station-2
   RUNG wire#powerrail
      Contact( "AlwaysTRUE" )
      Contact( "MASTER_SETUP_DB".S4_Enabled_Station[2] )
      "TCP_STN4_STN2_FB_DB"(Mod_TCP_Setup := "MOD_TCP_SETUP_DB".TCP_Data_Station4[2], LPG_Fill_Data := "MASTER_FILL_DATA".FILL_STATION_4[2], Modbus_Busy => "MASTER_FILL_DATA".FILL_STATION_4[2].FILL_SEQ_OUT.Modbus_Busy)
   END_RUNG
   // the same network as SCL:
   IF "AlwaysTRUE" AND "MASTER_SETUP_DB".S4_Enabled_Station[2] THEN
       "TCP_STN4_STN2_FB_DB"(Mod_TCP_Setup := "MOD_TCP_SETUP_DB".TCP_Data_Station4[2],   // "TCP_STN4_STN2_FB"
                             LPG_Fill_Data := "MASTER_FILL_DATA".FILL_STATION_4[2],
                             Modbus_Busy => "MASTER_FILL_DATA".FILL_STATION_4[2].FILL_SEQ_OUT.Modbus_Busy);
   END_IF;
END_REGION

REGION Network 4: Call Filling Line-1 Station-3
   RUNG wire#powerrail
      Contact( "AlwaysTRUE" )
      Contact( "MASTER_SETUP_DB".S4_Enabled_Station[3] )
      "TCP_STN4_STN3_FB_DB"(Mod_TCP_Setup := "MOD_TCP_SETUP_DB".TCP_Data_Station4[3], LPG_Fill_Data := "MASTER_FILL_DATA".FILL_STATION_4[3], Modbus_Busy => "MASTER_FILL_DATA".FILL_STATION_4[3].FILL_SEQ_OUT.Modbus_Busy)
   END_RUNG
   // the same network as SCL:
   IF "AlwaysTRUE" AND "MASTER_SETUP_DB".S4_Enabled_Station[3] THEN
       "TCP_STN4_STN3_FB_DB"(Mod_TCP_Setup := "MOD_TCP_SETUP_DB".TCP_Data_Station4[3],   // "TCP_STN4_STN3_FB"
                             LPG_Fill_Data := "MASTER_FILL_DATA".FILL_STATION_4[3],
                             Modbus_Busy => "MASTER_FILL_DATA".FILL_STATION_4[3].FILL_SEQ_OUT.Modbus_Busy);
   END_IF;
END_REGION

REGION Network 5: Call Filling Line-1 Station-4
   RUNG wire#powerrail
      Contact( "AlwaysTRUE" )
      Contact( "MASTER_SETUP_DB".S4_Enabled_Station[4] )
      "TCP_STN4_STN4_FB_DB"(Mod_TCP_Setup := "MOD_TCP_SETUP_DB".TCP_Data_Station4[4], LPG_Fill_Data := "MASTER_FILL_DATA".FILL_STATION_4[4], Modbus_Busy => "MASTER_FILL_DATA".FILL_STATION_4[4].FILL_SEQ_OUT.Modbus_Busy)
   END_RUNG
   // the same network as SCL:
   IF "AlwaysTRUE" AND "MASTER_SETUP_DB".S4_Enabled_Station[4] THEN
       "TCP_STN4_STN4_FB_DB"(Mod_TCP_Setup := "MOD_TCP_SETUP_DB".TCP_Data_Station4[4],   // "TCP_STN4_STN4_FB"
                             LPG_Fill_Data := "MASTER_FILL_DATA".FILL_STATION_4[4],
                             Modbus_Busy => "MASTER_FILL_DATA".FILL_STATION_4[4].FILL_SEQ_OUT.Modbus_Busy);
   END_IF;
END_REGION

REGION Network 6: Call Filling Line-1 Station-5
   RUNG wire#powerrail
      Contact( "AlwaysTRUE" )
      Contact( "MASTER_SETUP_DB".S4_Enabled_Station[5] )
      "TCP_STN4_STN5_FB_DB"(Mod_TCP_Setup := "MOD_TCP_SETUP_DB".TCP_Data_Station4[5], LPG_Fill_Data := "MASTER_FILL_DATA".FILL_STATION_4[5], Modbus_Busy => "MASTER_FILL_DATA".FILL_STATION_4[5].FILL_SEQ_OUT.Modbus_Busy)
   END_RUNG
   // the same network as SCL:
   IF "AlwaysTRUE" AND "MASTER_SETUP_DB".S4_Enabled_Station[5] THEN
       "TCP_STN4_STN5_FB_DB"(Mod_TCP_Setup := "MOD_TCP_SETUP_DB".TCP_Data_Station4[5],   // "TCP_STN4_STN5_FB"
                             LPG_Fill_Data := "MASTER_FILL_DATA".FILL_STATION_4[5],
                             Modbus_Busy => "MASTER_FILL_DATA".FILL_STATION_4[5].FILL_SEQ_OUT.Modbus_Busy);
   END_IF;
END_REGION

REGION Network 7: Call Filling Line-1 Station-6
   RUNG wire#powerrail
      Contact( "AlwaysTRUE" )
      Contact( "MASTER_SETUP_DB".S4_Enabled_Station[6] )
      "TCP_STN4_STN6_FB_DB"(Mod_TCP_Setup := "MOD_TCP_SETUP_DB".TCP_Data_Station4[6], LPG_Fill_Data := "MASTER_FILL_DATA".FILL_STATION_4[6], Modbus_Busy => "MASTER_FILL_DATA".FILL_STATION_4[6].FILL_SEQ_OUT.Modbus_Busy)
   END_RUNG
   // the same network as SCL:
   IF "AlwaysTRUE" AND "MASTER_SETUP_DB".S4_Enabled_Station[6] THEN
       "TCP_STN4_STN6_FB_DB"(Mod_TCP_Setup := "MOD_TCP_SETUP_DB".TCP_Data_Station4[6],   // "TCP_STN4_STN6_FB"
                             LPG_Fill_Data := "MASTER_FILL_DATA".FILL_STATION_4[6],
                             Modbus_Busy => "MASTER_FILL_DATA".FILL_STATION_4[6].FILL_SEQ_OUT.Modbus_Busy);
   END_IF;
END_REGION
END_FUNCTION

FUNCTION_BLOCK "TCP_STN4_STN1_FB"   // FB110, LAD
{ S7_Optimized_Access := 'TRUE' }
VERSION : 0.1
// stored: AutoNumber false, IsIECCheckEnabled false, IsRetainMemResEnabled false, MemoryReserve 100, SetENOAutomatically false, UDAEnableTagReadback false
   VAR_OUTPUT
      Modbus_Busy : Bool;
   END_VAR
   VAR_IN_OUT
      Mod_TCP_Setup : "Mod_TCP_Data";
      LPG_Fill_Data : "LPG_FILL_DATA";
   END_VAR
   VAR
      PStep_No : Struct
         MASTER_STEP_NO : "Master_Step_No";
      END_STRUCT;
      Write_Bit_Address : Int;
      TRIG : Array[1..100] of Bool;
      MOD_MASTER1_REQ : Array[1..10] of Bool;
      MOD_MASTER2_REQ : Array[1..10] of Bool;
      MOD_MASTER3_REQ : Array[1..10] of Bool;
      MOD_MASTER4_REQ : Array[1..10] of Bool;
      MOD_MASTER5_REQ : Array[1..10] of Bool;
      MOD_MASTER6_REQ : Array[1..10] of Bool;
      MAS_TRG_EXTN { S7_SetPoint := 'True'} : TOF_TIME;
      Tare_delay { S7_SetPoint := 'True'} : TON_TIME;
   END_VAR
   VAR_TEMP   // added for the SCL form of the ladder/FBD networks
      _w1 : Bool;
      _w2 : Bool;
      _w3 : Bool;
      _w4 : Bool;
   END_VAR
BEGIN

REGION Network 1: FILLING LINE-1 STATION-1
END_REGION

REGION Network 2: Write Master-1 Holding Register Request(Tare Weight Entry)
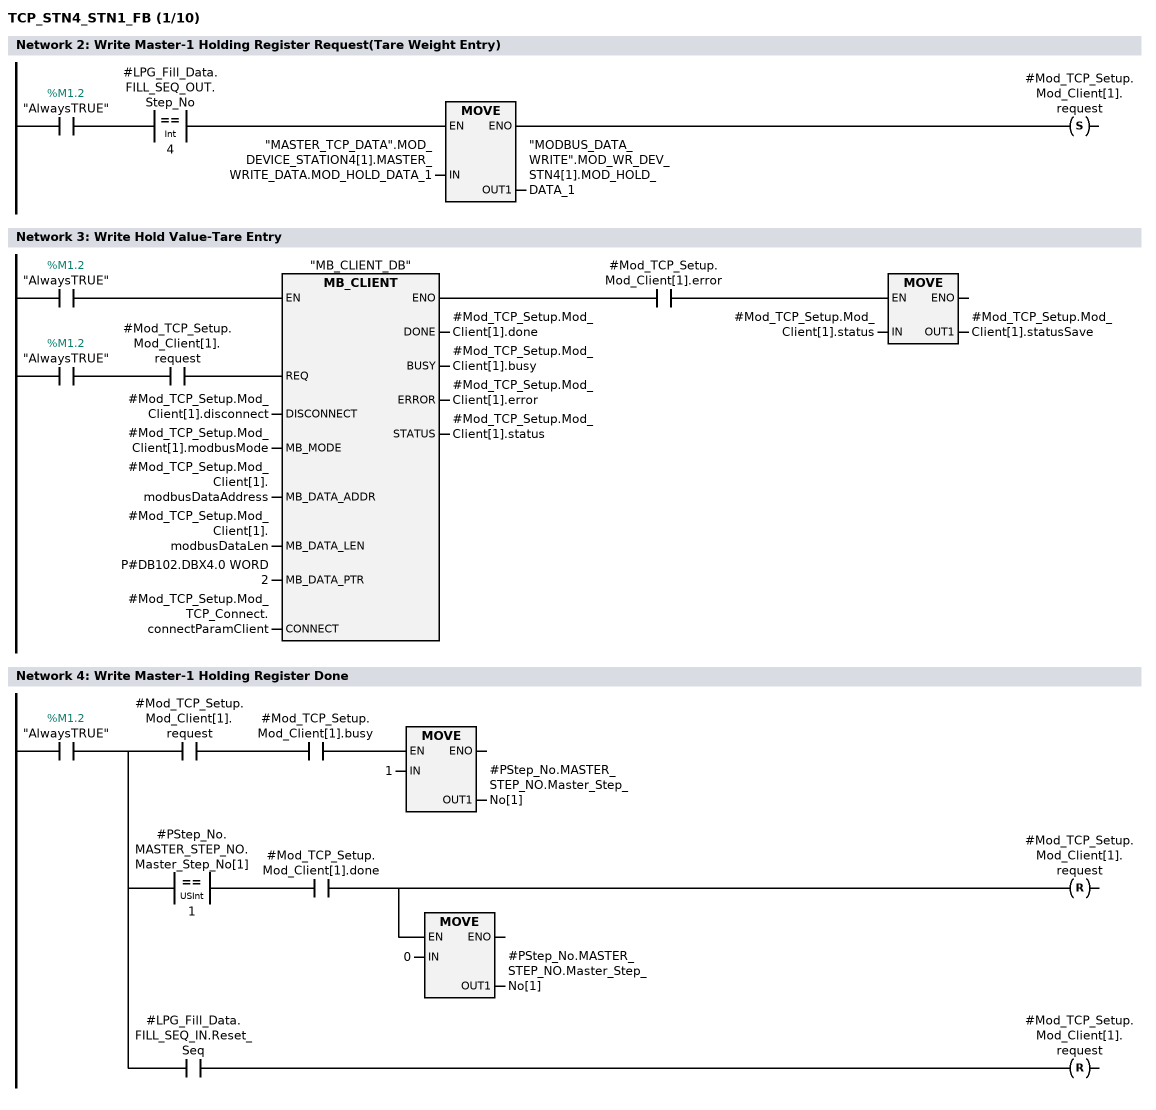
   RUNG wire#powerrail
      Contact( "AlwaysTRUE" )
      { S7_Templates := "SrcType := Int" } EQ_Contact(in1 := #LPG_Fill_Data.FILL_SEQ_OUT.Step_No, in2 := 4)
      Move(in := "MASTER_TCP_DATA".MOD_DEVICE_STATION4[1].MASTER_WRITE_DATA.MOD_HOLD_DATA_1, out1 => "MODBUS_DATA_WRITE".MOD_WR_DEV_STN4[1].MOD_HOLD_DATA_1)
      S_Coil( #Mod_TCP_Setup.Mod_Client[1].request )
   END_RUNG
   // the same network as SCL:
   IF "AlwaysTRUE" AND (#LPG_Fill_Data.FILL_SEQ_OUT.Step_No = 4) THEN
       "MODBUS_DATA_WRITE".MOD_WR_DEV_STN4[1].MOD_HOLD_DATA_1 := "MASTER_TCP_DATA".MOD_DEVICE_STATION4[1].MASTER_WRITE_DATA.MOD_HOLD_DATA_1;
       #Mod_TCP_Setup.Mod_Client[1].request := TRUE;
   END_IF;
END_REGION

REGION Network 3: Write Hold Value-Tare Entry
   RUNG wire#powerrail
      Contact( "AlwaysTRUE" )
      "MB_CLIENT_DB".MB_CLIENT(REQ := wire#w1, DISCONNECT := #Mod_TCP_Setup.Mod_Client[1].disconnect, MB_MODE := #Mod_TCP_Setup.Mod_Client[1].modbusMode, MB_DATA_ADDR := #Mod_TCP_Setup.Mod_Client[1].modbusDataAddress, MB_DATA_LEN := #Mod_TCP_Setup.Mod_Client[1].modbusDataLen, MB_DATA_PTR := P#DB102.DBX4.0 WORD 2, CONNECT := #Mod_TCP_Setup.Mod_TCP_Connect.connectParamClient, DONE => #Mod_TCP_Setup.Mod_Client[1].done, BUSY => #Mod_TCP_Setup.Mod_Client[1].busy, ERROR => #Mod_TCP_Setup.Mod_Client[1].error, STATUS => #Mod_TCP_Setup.Mod_Client[1].status)
      Contact( #Mod_TCP_Setup.Mod_Client[1].error )
      Move(in := #Mod_TCP_Setup.Mod_Client[1].status, out1 => #Mod_TCP_Setup.Mod_Client[1].statusSave)
   END_RUNG
   RUNG wire#powerrail
      Contact( "AlwaysTRUE" )
      Contact( #Mod_TCP_Setup.Mod_Client[1].request )
   END_RUNG wire#w1
   // the same network as SCL:
   "MB_CLIENT_DB"(EN := "AlwaysTRUE",   // MB_CLIENT
                  REQ := "AlwaysTRUE" AND #Mod_TCP_Setup.Mod_Client[1].request,
                  DISCONNECT := #Mod_TCP_Setup.Mod_Client[1].disconnect,
                  MB_MODE := #Mod_TCP_Setup.Mod_Client[1].modbusMode,
                  MB_DATA_ADDR := #Mod_TCP_Setup.Mod_Client[1].modbusDataAddress,
                  MB_DATA_LEN := #Mod_TCP_Setup.Mod_Client[1].modbusDataLen,
                  MB_DATA_PTR := P#DB102.DBX4.0 WORD 2,
                  CONNECT := #Mod_TCP_Setup.Mod_TCP_Connect.connectParamClient,
                  DONE => #Mod_TCP_Setup.Mod_Client[1].done,
                  BUSY => #Mod_TCP_Setup.Mod_Client[1].busy,
                  ERROR => #Mod_TCP_Setup.Mod_Client[1].error,
                  STATUS => #Mod_TCP_Setup.Mod_Client[1].status,
                  ENO => #_w1);
   IF #_w1 AND #Mod_TCP_Setup.Mod_Client[1].error THEN
       #Mod_TCP_Setup.Mod_Client[1].statusSave := #Mod_TCP_Setup.Mod_Client[1].status;
   END_IF;
END_REGION

REGION Network 4: Write Master-1 Holding Register Done
   RUNG wire#powerrail
      Contact( "AlwaysTRUE" )
      wire#w1
      Contact( #Mod_TCP_Setup.Mod_Client[1].request )
      Contact( #Mod_TCP_Setup.Mod_Client[1].busy )
      Move(in := 1, out1 => #PStep_No.MASTER_STEP_NO.Master_Step_No[1])
   END_RUNG
   RUNG wire#w1
      { S7_Templates := "SrcType := USInt" } EQ_Contact(in1 := #PStep_No.MASTER_STEP_NO.Master_Step_No[1], in2 := 1)
      Contact( #Mod_TCP_Setup.Mod_Client[1].done )
      wire#w2
      R_Coil( #Mod_TCP_Setup.Mod_Client[1].request )
   END_RUNG
   RUNG wire#w2
      Move(in := 0, out1 => #PStep_No.MASTER_STEP_NO.Master_Step_No[1])
   END_RUNG
   RUNG wire#w1
      Contact( #LPG_Fill_Data.FILL_SEQ_IN.Reset_Seq )
      R_Coil( #Mod_TCP_Setup.Mod_Client[1].request )
   END_RUNG
   // the same network as SCL:
   IF "AlwaysTRUE" AND #Mod_TCP_Setup.Mod_Client[1].request AND #Mod_TCP_Setup.Mod_Client[1].busy THEN
       #PStep_No.MASTER_STEP_NO.Master_Step_No[1] := 1;
   END_IF;
   #_w1 := "AlwaysTRUE" AND (#PStep_No.MASTER_STEP_NO.Master_Step_No[1] = 1) AND #Mod_TCP_Setup.Mod_Client[1].done;
   IF #_w1 THEN
       #Mod_TCP_Setup.Mod_Client[1].request := FALSE;
       #PStep_No.MASTER_STEP_NO.Master_Step_No[1] := 0;
   END_IF;
   IF "AlwaysTRUE" AND #LPG_Fill_Data.FILL_SEQ_IN.Reset_Seq THEN
       #Mod_TCP_Setup.Mod_Client[1].request := FALSE;
   END_IF;
END_REGION

REGION Network 5: Modbus Master2 Read Request(Filled Data)
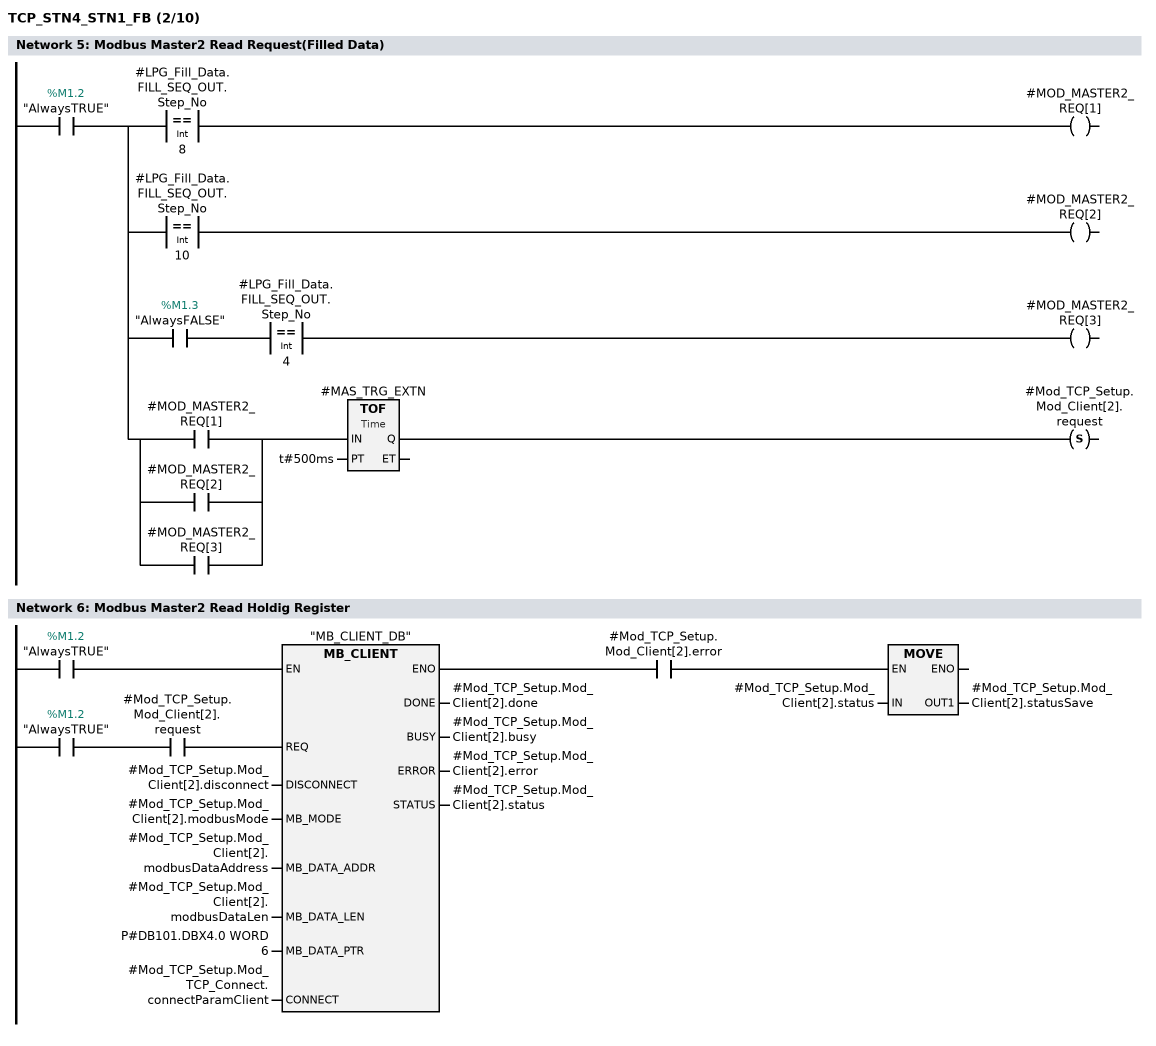
   RUNG wire#powerrail
      Contact( "AlwaysTRUE" )
      wire#w1
      { S7_Templates := "SrcType := Int" } EQ_Contact(in1 := #LPG_Fill_Data.FILL_SEQ_OUT.Step_No, in2 := 8)
      Coil( #MOD_MASTER2_REQ[1] )
   END_RUNG
   RUNG wire#w1
      { S7_Templates := "SrcType := Int" } EQ_Contact(in1 := #LPG_Fill_Data.FILL_SEQ_OUT.Step_No, in2 := 10)
      Coil( #MOD_MASTER2_REQ[2] )
   END_RUNG
   RUNG wire#w1
      Contact( "AlwaysFALSE" )
      { S7_Templates := "SrcType := Int" } EQ_Contact(in1 := #LPG_Fill_Data.FILL_SEQ_OUT.Step_No, in2 := 4)
      Coil( #MOD_MASTER2_REQ[3] )
   END_RUNG
   RUNG wire#w1
      Contact( #MOD_MASTER2_REQ[1] )
      wire#w2
      { S7_Templates := "time_type := Time" } #MAS_TRG_EXTN.TOF(pt := t#500ms, et =>)
      S_Coil( #Mod_TCP_Setup.Mod_Client[2].request )
   END_RUNG
   RUNG wire#w1
      Contact( #MOD_MASTER2_REQ[2] )
   END_RUNG wire#w2
   RUNG wire#w1
      Contact( #MOD_MASTER2_REQ[3] )
   END_RUNG wire#w2
   // the same network as SCL:
   #MOD_MASTER2_REQ[1] := "AlwaysTRUE" AND (#LPG_Fill_Data.FILL_SEQ_OUT.Step_No = 8);
   #MOD_MASTER2_REQ[2] := "AlwaysTRUE" AND (#LPG_Fill_Data.FILL_SEQ_OUT.Step_No = 10);
   #MOD_MASTER2_REQ[3] := "AlwaysTRUE" AND "AlwaysFALSE" AND (#LPG_Fill_Data.FILL_SEQ_OUT.Step_No = 4);
   #MAS_TRG_EXTN(IN := "AlwaysTRUE" AND (#MOD_MASTER2_REQ[1] OR #MOD_MASTER2_REQ[2] OR #MOD_MASTER2_REQ[3]),   // TOF
                 PT := t#500ms);
   IF #MAS_TRG_EXTN.Q THEN #Mod_TCP_Setup.Mod_Client[2].request := TRUE; END_IF;
END_REGION

REGION Network 6: Modbus Master2 Read Holdig Register
   RUNG wire#powerrail
      Contact( "AlwaysTRUE" )
      "MB_CLIENT_DB".MB_CLIENT(REQ := wire#w1, DISCONNECT := #Mod_TCP_Setup.Mod_Client[2].disconnect, MB_MODE := #Mod_TCP_Setup.Mod_Client[2].modbusMode, MB_DATA_ADDR := #Mod_TCP_Setup.Mod_Client[2].modbusDataAddress, MB_DATA_LEN := #Mod_TCP_Setup.Mod_Client[2].modbusDataLen, MB_DATA_PTR := P#DB101.DBX4.0 WORD 6, CONNECT := #Mod_TCP_Setup.Mod_TCP_Connect.connectParamClient, DONE => #Mod_TCP_Setup.Mod_Client[2].done, BUSY => #Mod_TCP_Setup.Mod_Client[2].busy, ERROR => #Mod_TCP_Setup.Mod_Client[2].error, STATUS => #Mod_TCP_Setup.Mod_Client[2].status)
      Contact( #Mod_TCP_Setup.Mod_Client[2].error )
      Move(in := #Mod_TCP_Setup.Mod_Client[2].status, out1 => #Mod_TCP_Setup.Mod_Client[2].statusSave)
   END_RUNG
   RUNG wire#powerrail
      Contact( "AlwaysTRUE" )
      Contact( #Mod_TCP_Setup.Mod_Client[2].request )
   END_RUNG wire#w1
   // the same network as SCL:
   "MB_CLIENT_DB"(EN := "AlwaysTRUE",   // MB_CLIENT
                  REQ := "AlwaysTRUE" AND #Mod_TCP_Setup.Mod_Client[2].request,
                  DISCONNECT := #Mod_TCP_Setup.Mod_Client[2].disconnect,
                  MB_MODE := #Mod_TCP_Setup.Mod_Client[2].modbusMode,
                  MB_DATA_ADDR := #Mod_TCP_Setup.Mod_Client[2].modbusDataAddress,
                  MB_DATA_LEN := #Mod_TCP_Setup.Mod_Client[2].modbusDataLen,
                  MB_DATA_PTR := P#DB101.DBX4.0 WORD 6,
                  CONNECT := #Mod_TCP_Setup.Mod_TCP_Connect.connectParamClient,
                  DONE => #Mod_TCP_Setup.Mod_Client[2].done,
                  BUSY => #Mod_TCP_Setup.Mod_Client[2].busy,
                  ERROR => #Mod_TCP_Setup.Mod_Client[2].error,
                  STATUS => #Mod_TCP_Setup.Mod_Client[2].status,
                  ENO => #_w1);
   IF #_w1 AND #Mod_TCP_Setup.Mod_Client[2].error THEN
       #Mod_TCP_Setup.Mod_Client[2].statusSave := #Mod_TCP_Setup.Mod_Client[2].status;
   END_IF;
END_REGION

REGION Network 7: Read Master-2 Holding Register Value
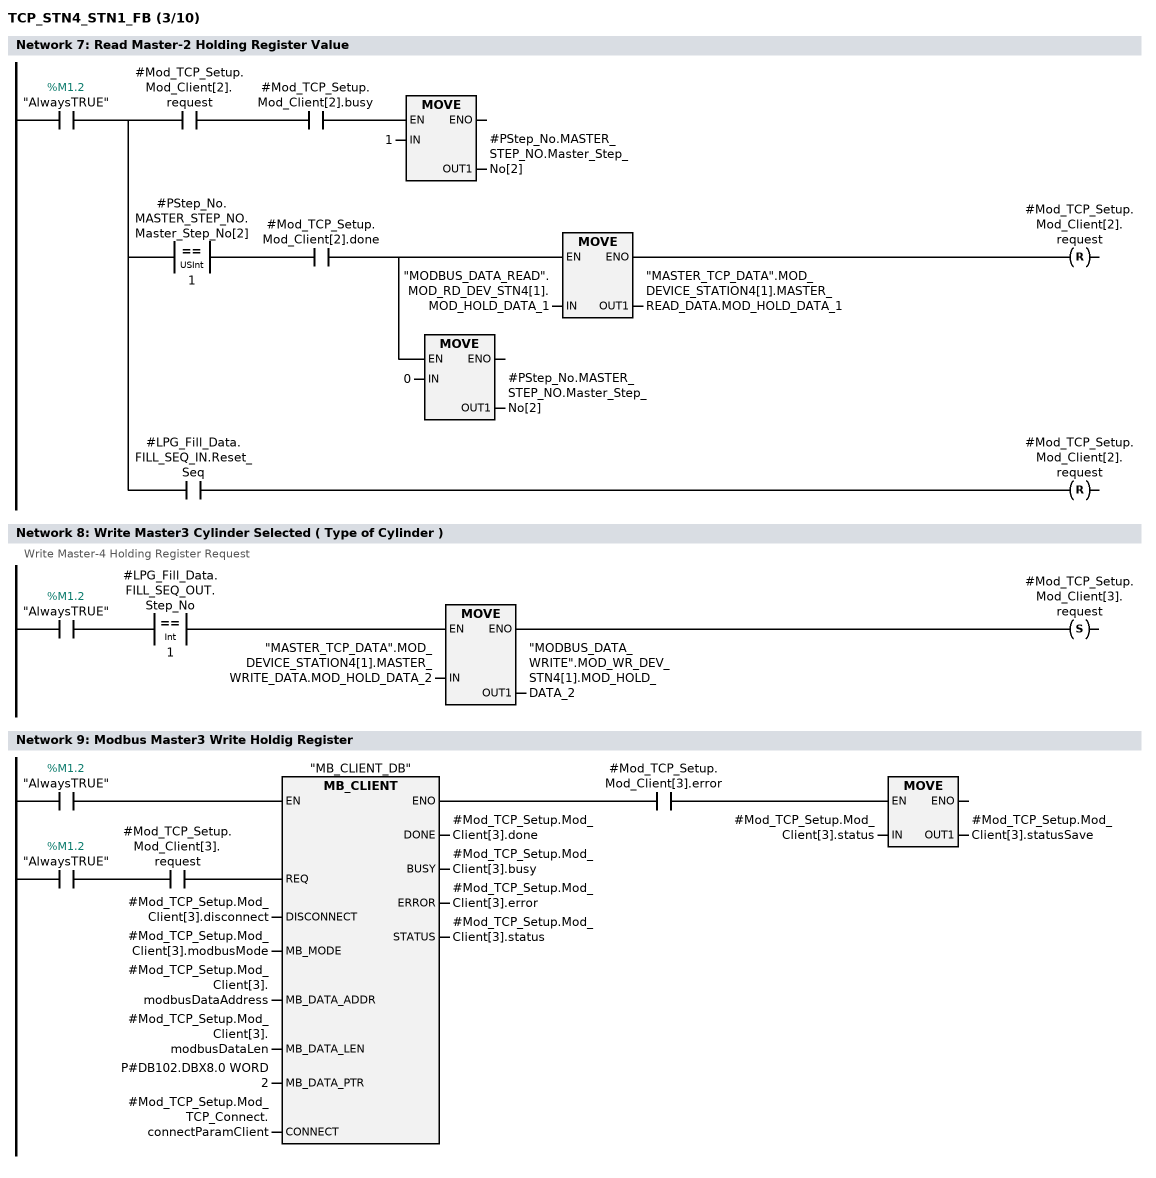
   RUNG wire#powerrail
      Contact( "AlwaysTRUE" )
      wire#w1
      Contact( #Mod_TCP_Setup.Mod_Client[2].request )
      Contact( #Mod_TCP_Setup.Mod_Client[2].busy )
      Move(in := 1, out1 => #PStep_No.MASTER_STEP_NO.Master_Step_No[2])
   END_RUNG
   RUNG wire#w1
      { S7_Templates := "SrcType := USInt" } EQ_Contact(in1 := #PStep_No.MASTER_STEP_NO.Master_Step_No[2], in2 := 1)
      Contact( #Mod_TCP_Setup.Mod_Client[2].done )
      wire#w2
      Move(in := "MODBUS_DATA_READ".MOD_RD_DEV_STN4[1].MOD_HOLD_DATA_1, out1 => "MASTER_TCP_DATA".MOD_DEVICE_STATION4[1].MASTER_READ_DATA.MOD_HOLD_DATA_1)
      R_Coil( #Mod_TCP_Setup.Mod_Client[2].request )
   END_RUNG
   RUNG wire#w2
      Move(in := 0, out1 => #PStep_No.MASTER_STEP_NO.Master_Step_No[2])
   END_RUNG
   RUNG wire#w1
      Contact( #LPG_Fill_Data.FILL_SEQ_IN.Reset_Seq )
      R_Coil( #Mod_TCP_Setup.Mod_Client[2].request )
   END_RUNG
   // the same network as SCL:
   IF "AlwaysTRUE" AND #Mod_TCP_Setup.Mod_Client[2].request AND #Mod_TCP_Setup.Mod_Client[2].busy THEN
       #PStep_No.MASTER_STEP_NO.Master_Step_No[2] := 1;
   END_IF;
   IF "AlwaysTRUE" AND (#PStep_No.MASTER_STEP_NO.Master_Step_No[2] = 1) AND #Mod_TCP_Setup.Mod_Client[2].done THEN
       "MASTER_TCP_DATA".MOD_DEVICE_STATION4[1].MASTER_READ_DATA.MOD_HOLD_DATA_1 := "MODBUS_DATA_READ".MOD_RD_DEV_STN4[1].MOD_HOLD_DATA_1;
   END_IF;
   #_w1 := "AlwaysTRUE" AND (#PStep_No.MASTER_STEP_NO.Master_Step_No[2] = 1) AND #Mod_TCP_Setup.Mod_Client[2].done;
   IF #_w1 THEN
       #Mod_TCP_Setup.Mod_Client[2].request := FALSE;
       #PStep_No.MASTER_STEP_NO.Master_Step_No[2] := 0;
   END_IF;
   IF "AlwaysTRUE" AND #LPG_Fill_Data.FILL_SEQ_IN.Reset_Seq THEN
       #Mod_TCP_Setup.Mod_Client[2].request := FALSE;
   END_IF;
END_REGION

REGION Network 8: Write Master3 Cylinder Selected ( Type of Cylinder )
   // Write Master-4 Holding Register Request
   RUNG wire#powerrail
      Contact( "AlwaysTRUE" )
      { S7_Templates := "SrcType := Int" } EQ_Contact(in1 := #LPG_Fill_Data.FILL_SEQ_OUT.Step_No, in2 := 1)
      Move(in := "MASTER_TCP_DATA".MOD_DEVICE_STATION4[1].MASTER_WRITE_DATA.MOD_HOLD_DATA_2, out1 => "MODBUS_DATA_WRITE".MOD_WR_DEV_STN4[1].MOD_HOLD_DATA_2)
      S_Coil( #Mod_TCP_Setup.Mod_Client[3].request )
   END_RUNG
   // the same network as SCL:
   IF "AlwaysTRUE" AND (#LPG_Fill_Data.FILL_SEQ_OUT.Step_No = 1) THEN
       "MODBUS_DATA_WRITE".MOD_WR_DEV_STN4[1].MOD_HOLD_DATA_2 := "MASTER_TCP_DATA".MOD_DEVICE_STATION4[1].MASTER_WRITE_DATA.MOD_HOLD_DATA_2;
       #Mod_TCP_Setup.Mod_Client[3].request := TRUE;
   END_IF;
END_REGION

REGION Network 9: Modbus Master3 Write Holdig Register
   RUNG wire#powerrail
      Contact( "AlwaysTRUE" )
      "MB_CLIENT_DB".MB_CLIENT(REQ := wire#w1, DISCONNECT := #Mod_TCP_Setup.Mod_Client[3].disconnect, MB_MODE := #Mod_TCP_Setup.Mod_Client[3].modbusMode, MB_DATA_ADDR := #Mod_TCP_Setup.Mod_Client[3].modbusDataAddress, MB_DATA_LEN := #Mod_TCP_Setup.Mod_Client[3].modbusDataLen, MB_DATA_PTR := P#DB102.DBX8.0 WORD 2, CONNECT := #Mod_TCP_Setup.Mod_TCP_Connect.connectParamClient, DONE => #Mod_TCP_Setup.Mod_Client[3].done, BUSY => #Mod_TCP_Setup.Mod_Client[3].busy, ERROR => #Mod_TCP_Setup.Mod_Client[3].error, STATUS => #Mod_TCP_Setup.Mod_Client[3].status)
      Contact( #Mod_TCP_Setup.Mod_Client[3].error )
      Move(in := #Mod_TCP_Setup.Mod_Client[3].status, out1 => #Mod_TCP_Setup.Mod_Client[3].statusSave)
   END_RUNG
   RUNG wire#powerrail
      Contact( "AlwaysTRUE" )
      Contact( #Mod_TCP_Setup.Mod_Client[3].request )
   END_RUNG wire#w1
   // the same network as SCL:
   "MB_CLIENT_DB"(EN := "AlwaysTRUE",   // MB_CLIENT
                  REQ := "AlwaysTRUE" AND #Mod_TCP_Setup.Mod_Client[3].request,
                  DISCONNECT := #Mod_TCP_Setup.Mod_Client[3].disconnect,
                  MB_MODE := #Mod_TCP_Setup.Mod_Client[3].modbusMode,
                  MB_DATA_ADDR := #Mod_TCP_Setup.Mod_Client[3].modbusDataAddress,
                  MB_DATA_LEN := #Mod_TCP_Setup.Mod_Client[3].modbusDataLen,
                  MB_DATA_PTR := P#DB102.DBX8.0 WORD 2,
                  CONNECT := #Mod_TCP_Setup.Mod_TCP_Connect.connectParamClient,
                  DONE => #Mod_TCP_Setup.Mod_Client[3].done,
                  BUSY => #Mod_TCP_Setup.Mod_Client[3].busy,
                  ERROR => #Mod_TCP_Setup.Mod_Client[3].error,
                  STATUS => #Mod_TCP_Setup.Mod_Client[3].status,
                  ENO => #_w1);
   IF #_w1 AND #Mod_TCP_Setup.Mod_Client[3].error THEN
       #Mod_TCP_Setup.Mod_Client[3].statusSave := #Mod_TCP_Setup.Mod_Client[3].status;
   END_IF;
END_REGION

REGION Network 10: Write Master-3 Holding Register Done
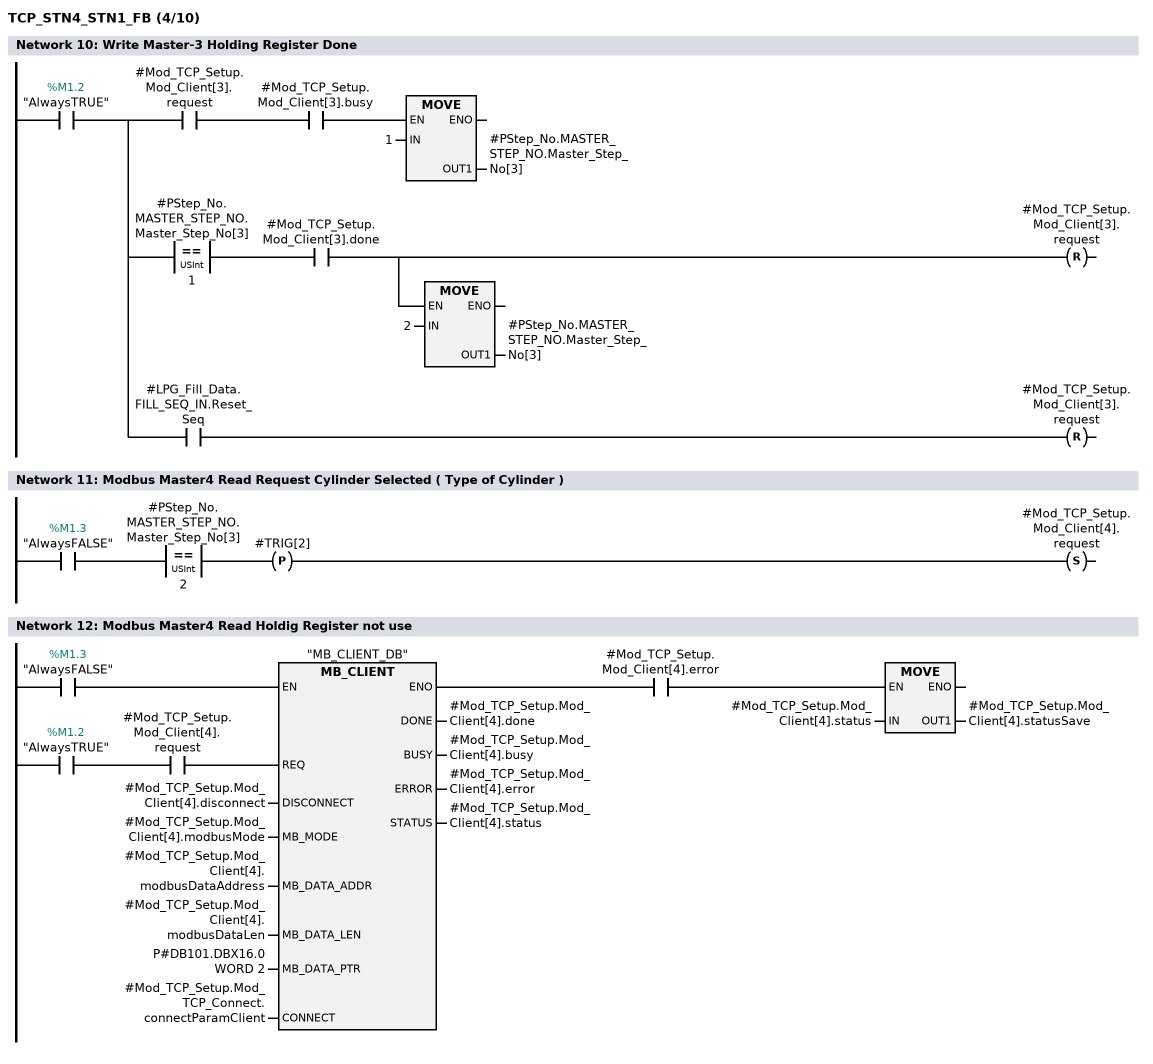
   RUNG wire#powerrail
      Contact( "AlwaysTRUE" )
      wire#w1
      Contact( #Mod_TCP_Setup.Mod_Client[3].request )
      Contact( #Mod_TCP_Setup.Mod_Client[3].busy )
      Move(in := 1, out1 => #PStep_No.MASTER_STEP_NO.Master_Step_No[3])
   END_RUNG
   RUNG wire#w1
      { S7_Templates := "SrcType := USInt" } EQ_Contact(in1 := #PStep_No.MASTER_STEP_NO.Master_Step_No[3], in2 := 1)
      Contact( #Mod_TCP_Setup.Mod_Client[3].done )
      wire#w2
      R_Coil( #Mod_TCP_Setup.Mod_Client[3].request )
   END_RUNG
   RUNG wire#w2
      Move(in := 2, out1 => #PStep_No.MASTER_STEP_NO.Master_Step_No[3])
   END_RUNG
   RUNG wire#w1
      Contact( #LPG_Fill_Data.FILL_SEQ_IN.Reset_Seq )
      R_Coil( #Mod_TCP_Setup.Mod_Client[3].request )
   END_RUNG
   // the same network as SCL:
   IF "AlwaysTRUE" AND #Mod_TCP_Setup.Mod_Client[3].request AND #Mod_TCP_Setup.Mod_Client[3].busy THEN
       #PStep_No.MASTER_STEP_NO.Master_Step_No[3] := 1;
   END_IF;
   #_w1 := "AlwaysTRUE" AND (#PStep_No.MASTER_STEP_NO.Master_Step_No[3] = 1) AND #Mod_TCP_Setup.Mod_Client[3].done;
   IF #_w1 THEN
       #Mod_TCP_Setup.Mod_Client[3].request := FALSE;
       #PStep_No.MASTER_STEP_NO.Master_Step_No[3] := 2;
   END_IF;
   IF "AlwaysTRUE" AND #LPG_Fill_Data.FILL_SEQ_IN.Reset_Seq THEN
       #Mod_TCP_Setup.Mod_Client[3].request := FALSE;
   END_IF;
END_REGION

REGION Network 11: Modbus Master4 Read Request Cylinder Selected ( Type of Cylinder )
   RUNG wire#powerrail
      Contact( "AlwaysFALSE" )
      { S7_Templates := "SrcType := USInt" } EQ_Contact(in1 := #PStep_No.MASTER_STEP_NO.Master_Step_No[3], in2 := 2)
      P_Trig( #TRIG[2] )
      S_Coil( #Mod_TCP_Setup.Mod_Client[4].request )
   END_RUNG
   // the same network as SCL:
   #_w1 := "AlwaysFALSE" AND (#PStep_No.MASTER_STEP_NO.Master_Step_No[3] = 2);
   #_w2 := #_w1 AND NOT #TRIG[2];   // rising edge
   #TRIG[2] := #_w1;
   IF #_w2 THEN #Mod_TCP_Setup.Mod_Client[4].request := TRUE; END_IF;
END_REGION

REGION Network 12: Modbus Master4 Read Holdig Register not use
   RUNG wire#powerrail
      Contact( "AlwaysFALSE" )
      "MB_CLIENT_DB".MB_CLIENT(REQ := wire#w1, DISCONNECT := #Mod_TCP_Setup.Mod_Client[4].disconnect, MB_MODE := #Mod_TCP_Setup.Mod_Client[4].modbusMode, MB_DATA_ADDR := #Mod_TCP_Setup.Mod_Client[4].modbusDataAddress, MB_DATA_LEN := #Mod_TCP_Setup.Mod_Client[4].modbusDataLen, MB_DATA_PTR := P#DB101.DBX16.0 WORD 2, CONNECT := #Mod_TCP_Setup.Mod_TCP_Connect.connectParamClient, DONE => #Mod_TCP_Setup.Mod_Client[4].done, BUSY => #Mod_TCP_Setup.Mod_Client[4].busy, ERROR => #Mod_TCP_Setup.Mod_Client[4].error, STATUS => #Mod_TCP_Setup.Mod_Client[4].status)
      Contact( #Mod_TCP_Setup.Mod_Client[4].error )
      Move(in := #Mod_TCP_Setup.Mod_Client[4].status, out1 => #Mod_TCP_Setup.Mod_Client[4].statusSave)
   END_RUNG
   RUNG wire#powerrail
      Contact( "AlwaysTRUE" )
      Contact( #Mod_TCP_Setup.Mod_Client[4].request )
   END_RUNG wire#w1
   // the same network as SCL:
   "MB_CLIENT_DB"(EN := "AlwaysFALSE",   // MB_CLIENT
                  REQ := "AlwaysTRUE" AND #Mod_TCP_Setup.Mod_Client[4].request,
                  DISCONNECT := #Mod_TCP_Setup.Mod_Client[4].disconnect,
                  MB_MODE := #Mod_TCP_Setup.Mod_Client[4].modbusMode,
                  MB_DATA_ADDR := #Mod_TCP_Setup.Mod_Client[4].modbusDataAddress,
                  MB_DATA_LEN := #Mod_TCP_Setup.Mod_Client[4].modbusDataLen,
                  MB_DATA_PTR := P#DB101.DBX16.0 WORD 2,
                  CONNECT := #Mod_TCP_Setup.Mod_TCP_Connect.connectParamClient,
                  DONE => #Mod_TCP_Setup.Mod_Client[4].done,
                  BUSY => #Mod_TCP_Setup.Mod_Client[4].busy,
                  ERROR => #Mod_TCP_Setup.Mod_Client[4].error,
                  STATUS => #Mod_TCP_Setup.Mod_Client[4].status,
                  ENO => #_w1);
   IF #_w1 AND #Mod_TCP_Setup.Mod_Client[4].error THEN
       #Mod_TCP_Setup.Mod_Client[4].statusSave := #Mod_TCP_Setup.Mod_Client[4].status;
   END_IF;
END_REGION

REGION Network 13: Read Master-4 Holding Register Value
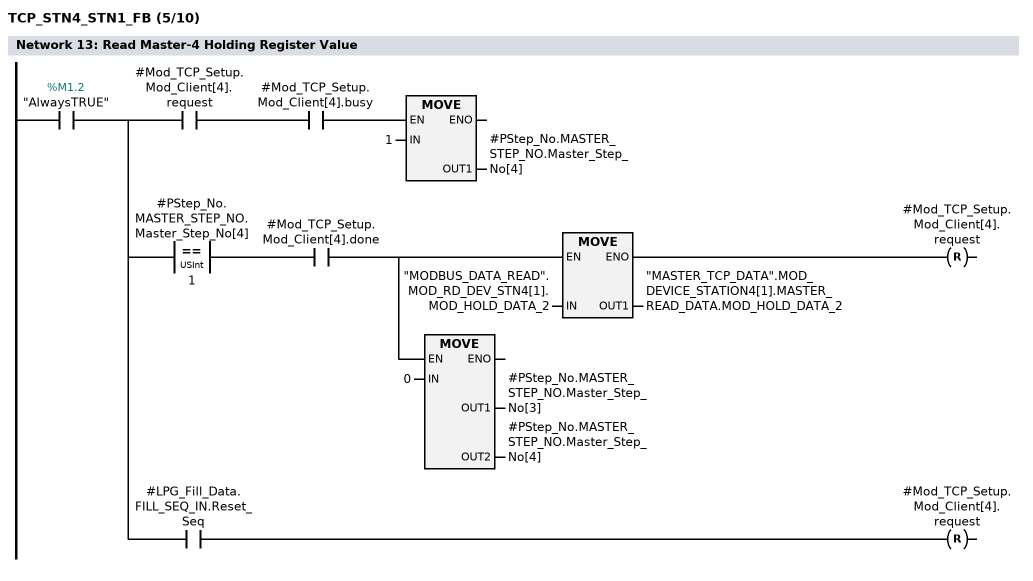
   RUNG wire#powerrail
      Contact( "AlwaysTRUE" )
      wire#w1
      Contact( #Mod_TCP_Setup.Mod_Client[4].request )
      Contact( #Mod_TCP_Setup.Mod_Client[4].busy )
      Move(in := 1, out1 => #PStep_No.MASTER_STEP_NO.Master_Step_No[4])
   END_RUNG
   RUNG wire#w1
      { S7_Templates := "SrcType := USInt" } EQ_Contact(in1 := #PStep_No.MASTER_STEP_NO.Master_Step_No[4], in2 := 1)
      Contact( #Mod_TCP_Setup.Mod_Client[4].done )
      wire#w2
      Move(in := "MODBUS_DATA_READ".MOD_RD_DEV_STN4[1].MOD_HOLD_DATA_2, out1 => "MASTER_TCP_DATA".MOD_DEVICE_STATION4[1].MASTER_READ_DATA.MOD_HOLD_DATA_2)
      R_Coil( #Mod_TCP_Setup.Mod_Client[4].request )
   END_RUNG
   RUNG wire#w2
      Move(in := 0, out1 => #PStep_No.MASTER_STEP_NO.Master_Step_No[3], out2 => #PStep_No.MASTER_STEP_NO.Master_Step_No[4])
   END_RUNG
   RUNG wire#w1
      Contact( #LPG_Fill_Data.FILL_SEQ_IN.Reset_Seq )
      R_Coil( #Mod_TCP_Setup.Mod_Client[4].request )
   END_RUNG
   // the same network as SCL:
   IF "AlwaysTRUE" AND #Mod_TCP_Setup.Mod_Client[4].request AND #Mod_TCP_Setup.Mod_Client[4].busy THEN
       #PStep_No.MASTER_STEP_NO.Master_Step_No[4] := 1;
   END_IF;
   IF "AlwaysTRUE" AND (#PStep_No.MASTER_STEP_NO.Master_Step_No[4] = 1) AND #Mod_TCP_Setup.Mod_Client[4].done THEN
       "MASTER_TCP_DATA".MOD_DEVICE_STATION4[1].MASTER_READ_DATA.MOD_HOLD_DATA_2 := "MODBUS_DATA_READ".MOD_RD_DEV_STN4[1].MOD_HOLD_DATA_2;
   END_IF;
   #_w1 := "AlwaysTRUE" AND (#PStep_No.MASTER_STEP_NO.Master_Step_No[4] = 1) AND #Mod_TCP_Setup.Mod_Client[4].done;
   IF #_w1 THEN
       #Mod_TCP_Setup.Mod_Client[4].request := FALSE;
       #PStep_No.MASTER_STEP_NO.Master_Step_No[3] := 0;
       #PStep_No.MASTER_STEP_NO.Master_Step_No[4] := 0;
   END_IF;
   IF "AlwaysTRUE" AND #LPG_Fill_Data.FILL_SEQ_IN.Reset_Seq THEN
       #Mod_TCP_Setup.Mod_Client[4].request := FALSE;
   END_IF;
END_REGION

REGION Network 14: Modbus Master5 Read Request(Coil Status)
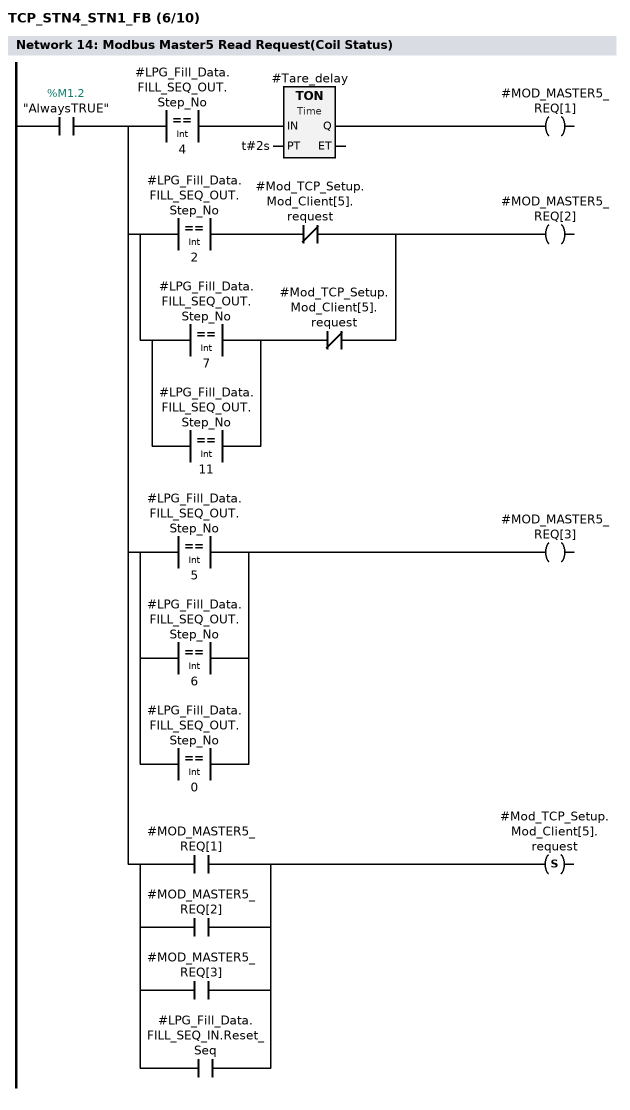
   RUNG wire#powerrail
      Contact( "AlwaysTRUE" )
      wire#w1
      { S7_Templates := "SrcType := Int" } EQ_Contact(in1 := #LPG_Fill_Data.FILL_SEQ_OUT.Step_No, in2 := 4)
      { S7_Templates := "time_type := Time" } #Tare_delay.TON(pt := t#2s, et =>)
      Coil( #MOD_MASTER5_REQ[1] )
   END_RUNG
   RUNG wire#w1
      { S7_Templates := "SrcType := Int" } EQ_Contact(in1 := #LPG_Fill_Data.FILL_SEQ_OUT.Step_No, in2 := 2)
      I_Contact( #Mod_TCP_Setup.Mod_Client[5].request )
      wire#w2
      Coil( #MOD_MASTER5_REQ[2] )
   END_RUNG
   RUNG wire#w1
      { S7_Templates := "SrcType := Int" } EQ_Contact(in1 := #LPG_Fill_Data.FILL_SEQ_OUT.Step_No, in2 := 7)
      wire#w3
      I_Contact( #Mod_TCP_Setup.Mod_Client[5].request )
   END_RUNG wire#w2
   RUNG wire#w1
      { S7_Templates := "SrcType := Int" } EQ_Contact(in1 := #LPG_Fill_Data.FILL_SEQ_OUT.Step_No, in2 := 11)
   END_RUNG wire#w3
   RUNG wire#w1
      { S7_Templates := "SrcType := Int" } EQ_Contact(in1 := #LPG_Fill_Data.FILL_SEQ_OUT.Step_No, in2 := 5)
      wire#w4
      Coil( #MOD_MASTER5_REQ[3] )
   END_RUNG
   RUNG wire#w1
      { S7_Templates := "SrcType := Int" } EQ_Contact(in1 := #LPG_Fill_Data.FILL_SEQ_OUT.Step_No, in2 := 6)
   END_RUNG wire#w4
   RUNG wire#w1
      { S7_Templates := "SrcType := Int" } EQ_Contact(in1 := #LPG_Fill_Data.FILL_SEQ_OUT.Step_No, in2 := 0)
   END_RUNG wire#w4
   RUNG wire#w1
      Contact( #MOD_MASTER5_REQ[1] )
      wire#w5
      S_Coil( #Mod_TCP_Setup.Mod_Client[5].request )
   END_RUNG
   RUNG wire#w1
      Contact( #MOD_MASTER5_REQ[2] )
   END_RUNG wire#w5
   RUNG wire#w1
      Contact( #MOD_MASTER5_REQ[3] )
   END_RUNG wire#w5
   RUNG wire#w1
      Contact( #LPG_Fill_Data.FILL_SEQ_IN.Reset_Seq )
   END_RUNG wire#w5
   // the same network as SCL:
   #Tare_delay(IN := "AlwaysTRUE" AND (#LPG_Fill_Data.FILL_SEQ_OUT.Step_No = 4), PT := t#2s);   // TON
   #MOD_MASTER5_REQ[1] := #Tare_delay.Q;
   #MOD_MASTER5_REQ[2] := "AlwaysTRUE" AND (((#LPG_Fill_Data.FILL_SEQ_OUT.Step_No = 2) AND NOT #Mod_TCP_Setup.Mod_Client[5].request) OR (((#LPG_Fill_Data.FILL_SEQ_OUT.Step_No = 7) OR (#LPG_Fill_Data.FILL_SEQ_OUT.Step_No = 11)) AND NOT #Mod_TCP_Setup.Mod_Client[5].request));
   #MOD_MASTER5_REQ[3] := "AlwaysTRUE" AND ((#LPG_Fill_Data.FILL_SEQ_OUT.Step_No = 5) OR (#LPG_Fill_Data.FILL_SEQ_OUT.Step_No = 6) OR (#LPG_Fill_Data.FILL_SEQ_OUT.Step_No = 0));
   IF "AlwaysTRUE" AND (#MOD_MASTER5_REQ[1] OR #MOD_MASTER5_REQ[2] OR #MOD_MASTER5_REQ[3] OR #LPG_Fill_Data.FILL_SEQ_IN.Reset_Seq) THEN
       #Mod_TCP_Setup.Mod_Client[5].request := TRUE;
   END_IF;
END_REGION

REGION Network 15: Modbus Master5 Read Coil Status
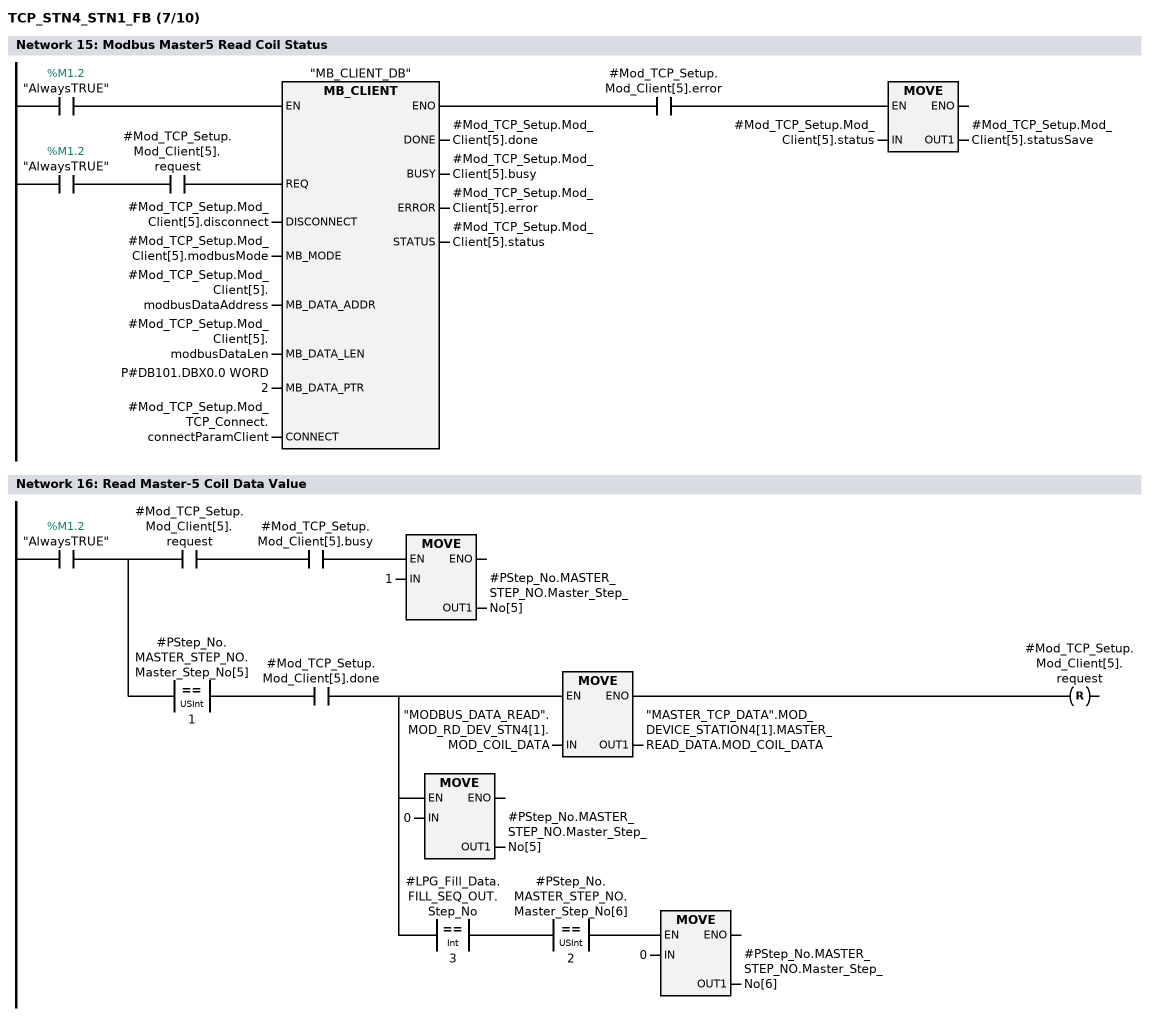
   RUNG wire#powerrail
      Contact( "AlwaysTRUE" )
      "MB_CLIENT_DB".MB_CLIENT(REQ := wire#w1, DISCONNECT := #Mod_TCP_Setup.Mod_Client[5].disconnect, MB_MODE := #Mod_TCP_Setup.Mod_Client[5].modbusMode, MB_DATA_ADDR := #Mod_TCP_Setup.Mod_Client[5].modbusDataAddress, MB_DATA_LEN := #Mod_TCP_Setup.Mod_Client[5].modbusDataLen, MB_DATA_PTR := P#DB101.DBX0.0 WORD 2, CONNECT := #Mod_TCP_Setup.Mod_TCP_Connect.connectParamClient, DONE => #Mod_TCP_Setup.Mod_Client[5].done, BUSY => #Mod_TCP_Setup.Mod_Client[5].busy, ERROR => #Mod_TCP_Setup.Mod_Client[5].error, STATUS => #Mod_TCP_Setup.Mod_Client[5].status)
      Contact( #Mod_TCP_Setup.Mod_Client[5].error )
      Move(in := #Mod_TCP_Setup.Mod_Client[5].status, out1 => #Mod_TCP_Setup.Mod_Client[5].statusSave)
   END_RUNG
   RUNG wire#powerrail
      Contact( "AlwaysTRUE" )
      Contact( #Mod_TCP_Setup.Mod_Client[5].request )
   END_RUNG wire#w1
   // the same network as SCL:
   "MB_CLIENT_DB"(EN := "AlwaysTRUE",   // MB_CLIENT
                  REQ := "AlwaysTRUE" AND #Mod_TCP_Setup.Mod_Client[5].request,
                  DISCONNECT := #Mod_TCP_Setup.Mod_Client[5].disconnect,
                  MB_MODE := #Mod_TCP_Setup.Mod_Client[5].modbusMode,
                  MB_DATA_ADDR := #Mod_TCP_Setup.Mod_Client[5].modbusDataAddress,
                  MB_DATA_LEN := #Mod_TCP_Setup.Mod_Client[5].modbusDataLen,
                  MB_DATA_PTR := P#DB101.DBX0.0 WORD 2,
                  CONNECT := #Mod_TCP_Setup.Mod_TCP_Connect.connectParamClient,
                  DONE => #Mod_TCP_Setup.Mod_Client[5].done,
                  BUSY => #Mod_TCP_Setup.Mod_Client[5].busy,
                  ERROR => #Mod_TCP_Setup.Mod_Client[5].error,
                  STATUS => #Mod_TCP_Setup.Mod_Client[5].status,
                  ENO => #_w1);
   IF #_w1 AND #Mod_TCP_Setup.Mod_Client[5].error THEN
       #Mod_TCP_Setup.Mod_Client[5].statusSave := #Mod_TCP_Setup.Mod_Client[5].status;
   END_IF;
END_REGION

REGION Network 16: Read Master-5 Coil Data Value
   RUNG wire#powerrail
      Contact( "AlwaysTRUE" )
      wire#w1
      Contact( #Mod_TCP_Setup.Mod_Client[5].request )
      Contact( #Mod_TCP_Setup.Mod_Client[5].busy )
      Move(in := 1, out1 => #PStep_No.MASTER_STEP_NO.Master_Step_No[5])
   END_RUNG
   RUNG wire#w1
      { S7_Templates := "SrcType := USInt" } EQ_Contact(in1 := #PStep_No.MASTER_STEP_NO.Master_Step_No[5], in2 := 1)
      Contact( #Mod_TCP_Setup.Mod_Client[5].done )
      wire#w2
      Move(in := "MODBUS_DATA_READ".MOD_RD_DEV_STN4[1].MOD_COIL_DATA, out1 => "MASTER_TCP_DATA".MOD_DEVICE_STATION4[1].MASTER_READ_DATA.MOD_COIL_DATA)
      R_Coil( #Mod_TCP_Setup.Mod_Client[5].request )
   END_RUNG
   RUNG wire#w2
      Move(in := 0, out1 => #PStep_No.MASTER_STEP_NO.Master_Step_No[5])
   END_RUNG
   RUNG wire#w2
      { S7_Templates := "SrcType := Int" } EQ_Contact(in1 := #LPG_Fill_Data.FILL_SEQ_OUT.Step_No, in2 := 3)
      { S7_Templates := "SrcType := USInt" } EQ_Contact(in1 := #PStep_No.MASTER_STEP_NO.Master_Step_No[6], in2 := 2)
      Move(in := 0, out1 => #PStep_No.MASTER_STEP_NO.Master_Step_No[6])
   END_RUNG
   // the same network as SCL:
   IF "AlwaysTRUE" AND #Mod_TCP_Setup.Mod_Client[5].request AND #Mod_TCP_Setup.Mod_Client[5].busy THEN
       #PStep_No.MASTER_STEP_NO.Master_Step_No[5] := 1;
   END_IF;
   #_w1 := "AlwaysTRUE" AND (#PStep_No.MASTER_STEP_NO.Master_Step_No[5] = 1) AND #Mod_TCP_Setup.Mod_Client[5].done;
   IF #_w1 THEN
       "MASTER_TCP_DATA".MOD_DEVICE_STATION4[1].MASTER_READ_DATA.MOD_COIL_DATA := "MODBUS_DATA_READ".MOD_RD_DEV_STN4[1].MOD_COIL_DATA;
       #Mod_TCP_Setup.Mod_Client[5].request := FALSE;
       #PStep_No.MASTER_STEP_NO.Master_Step_No[5] := 0;
   END_IF;
   IF #_w1 AND (#LPG_Fill_Data.FILL_SEQ_OUT.Step_No = 3) AND (#PStep_No.MASTER_STEP_NO.Master_Step_No[6] = 2) THEN
       #PStep_No.MASTER_STEP_NO.Master_Step_No[6] := 0;
   END_IF;
END_REGION

REGION Network 17: Write Coil Data
   // if multiple bit write not working
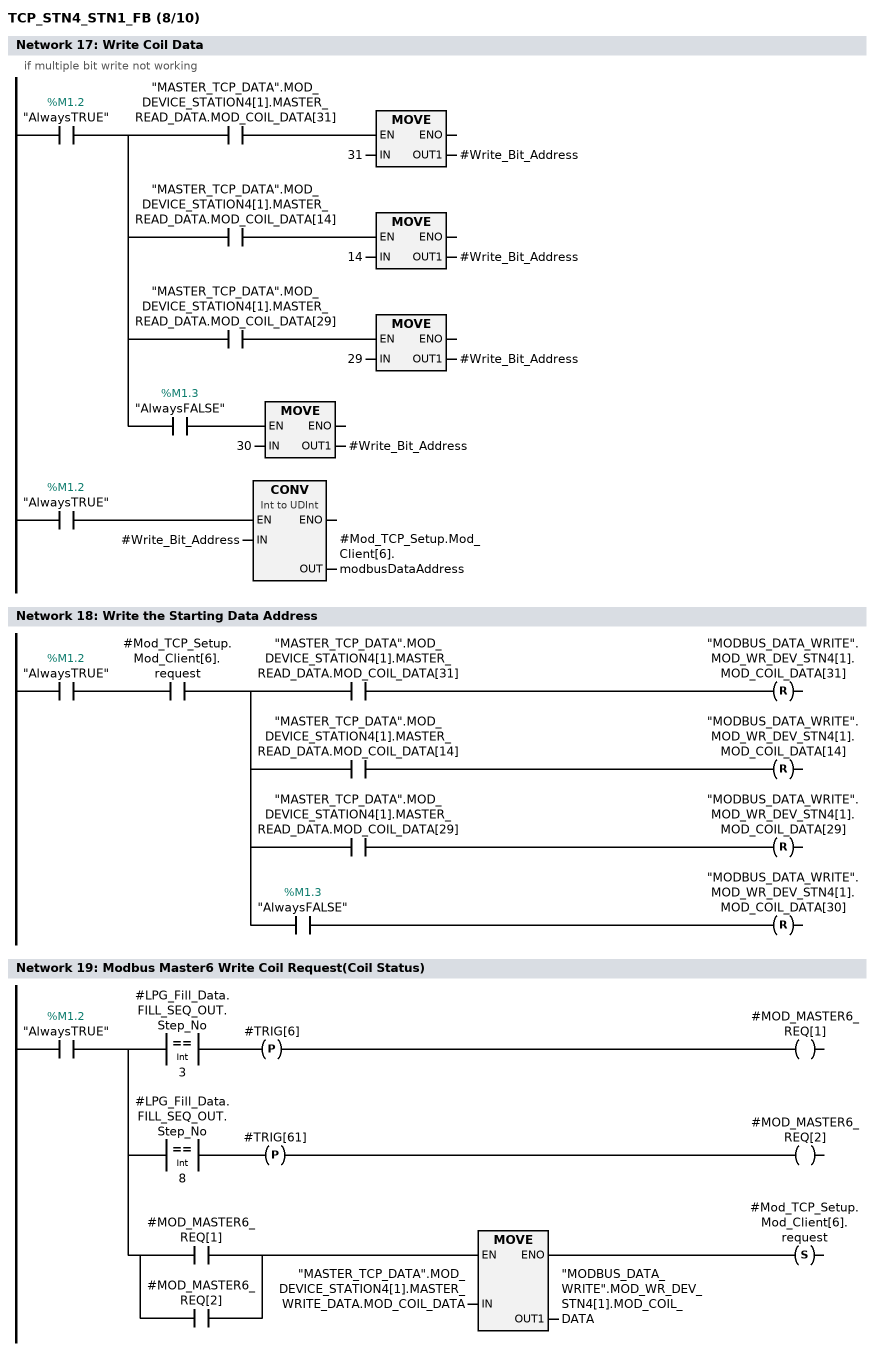
   RUNG wire#powerrail
      Contact( "AlwaysTRUE" )
      wire#w1
      Contact( "MASTER_TCP_DATA".MOD_DEVICE_STATION4[1].MASTER_READ_DATA.MOD_COIL_DATA[31] )
      Move(in := 31, out1 => #Write_Bit_Address)
   END_RUNG
   RUNG wire#w1
      Contact( "MASTER_TCP_DATA".MOD_DEVICE_STATION4[1].MASTER_READ_DATA.MOD_COIL_DATA[14] )
      Move(in := 14, out1 => #Write_Bit_Address)
   END_RUNG
   RUNG wire#w1
      Contact( "MASTER_TCP_DATA".MOD_DEVICE_STATION4[1].MASTER_READ_DATA.MOD_COIL_DATA[29] )
      Move(in := 29, out1 => #Write_Bit_Address)
   END_RUNG
   RUNG wire#w1
      Contact( "AlwaysFALSE" )
      Move(in := 30, out1 => #Write_Bit_Address)
   END_RUNG
   RUNG wire#powerrail
      Contact( "AlwaysTRUE" )
      { S7_Templates := "[SrcType := Int, DestType := UDInt]" } Convert(in := #Write_Bit_Address, out => #Mod_TCP_Setup.Mod_Client[6].modbusDataAddress)
   END_RUNG
   // the same network as SCL:
   IF "AlwaysTRUE" AND "MASTER_TCP_DATA".MOD_DEVICE_STATION4[1].MASTER_READ_DATA.MOD_COIL_DATA[31] THEN
       #Write_Bit_Address := 31;
   END_IF;
   IF "AlwaysTRUE" AND "MASTER_TCP_DATA".MOD_DEVICE_STATION4[1].MASTER_READ_DATA.MOD_COIL_DATA[14] THEN
       #Write_Bit_Address := 14;
   END_IF;
   IF "AlwaysTRUE" AND "MASTER_TCP_DATA".MOD_DEVICE_STATION4[1].MASTER_READ_DATA.MOD_COIL_DATA[29] THEN
       #Write_Bit_Address := 29;
   END_IF;
   IF "AlwaysTRUE" AND "AlwaysFALSE" THEN #Write_Bit_Address := 30; END_IF;
   IF "AlwaysTRUE" THEN
       #Mod_TCP_Setup.Mod_Client[6].modbusDataAddress := INT_TO_UDINT(#Write_Bit_Address);
   END_IF;
END_REGION

REGION Network 18: Write the Starting Data Address
   RUNG wire#powerrail
      Contact( "AlwaysTRUE" )
      Contact( #Mod_TCP_Setup.Mod_Client[6].request )
      wire#w1
      Contact( "MASTER_TCP_DATA".MOD_DEVICE_STATION4[1].MASTER_READ_DATA.MOD_COIL_DATA[31] )
      R_Coil( "MODBUS_DATA_WRITE".MOD_WR_DEV_STN4[1].MOD_COIL_DATA[31] )
   END_RUNG
   RUNG wire#w1
      Contact( "MASTER_TCP_DATA".MOD_DEVICE_STATION4[1].MASTER_READ_DATA.MOD_COIL_DATA[14] )
      R_Coil( "MODBUS_DATA_WRITE".MOD_WR_DEV_STN4[1].MOD_COIL_DATA[14] )
   END_RUNG
   RUNG wire#w1
      Contact( "MASTER_TCP_DATA".MOD_DEVICE_STATION4[1].MASTER_READ_DATA.MOD_COIL_DATA[29] )
      R_Coil( "MODBUS_DATA_WRITE".MOD_WR_DEV_STN4[1].MOD_COIL_DATA[29] )
   END_RUNG
   RUNG wire#w1
      Contact( "AlwaysFALSE" )
      R_Coil( "MODBUS_DATA_WRITE".MOD_WR_DEV_STN4[1].MOD_COIL_DATA[30] )
   END_RUNG
   // the same network as SCL:
   #_w1 := "AlwaysTRUE" AND #Mod_TCP_Setup.Mod_Client[6].request;
   IF #_w1 AND "MASTER_TCP_DATA".MOD_DEVICE_STATION4[1].MASTER_READ_DATA.MOD_COIL_DATA[31] THEN
       "MODBUS_DATA_WRITE".MOD_WR_DEV_STN4[1].MOD_COIL_DATA[31] := FALSE;
   END_IF;
   IF #_w1 AND "MASTER_TCP_DATA".MOD_DEVICE_STATION4[1].MASTER_READ_DATA.MOD_COIL_DATA[14] THEN
       "MODBUS_DATA_WRITE".MOD_WR_DEV_STN4[1].MOD_COIL_DATA[14] := FALSE;
   END_IF;
   IF #_w1 AND "MASTER_TCP_DATA".MOD_DEVICE_STATION4[1].MASTER_READ_DATA.MOD_COIL_DATA[29] THEN
       "MODBUS_DATA_WRITE".MOD_WR_DEV_STN4[1].MOD_COIL_DATA[29] := FALSE;
   END_IF;
   IF #_w1 AND "AlwaysFALSE" THEN "MODBUS_DATA_WRITE".MOD_WR_DEV_STN4[1].MOD_COIL_DATA[30] := FALSE; END_IF;
END_REGION

REGION Network 19: Modbus Master6 Write Coil Request(Coil Status)
   RUNG wire#powerrail
      Contact( "AlwaysTRUE" )
      wire#w1
      { S7_Templates := "SrcType := Int" } EQ_Contact(in1 := #LPG_Fill_Data.FILL_SEQ_OUT.Step_No, in2 := 3)
      P_Trig( #TRIG[6] )
      Coil( #MOD_MASTER6_REQ[1] )
   END_RUNG
   RUNG wire#w1
      { S7_Templates := "SrcType := Int" } EQ_Contact(in1 := #LPG_Fill_Data.FILL_SEQ_OUT.Step_No, in2 := 8)
      P_Trig( #TRIG[61] )
      Coil( #MOD_MASTER6_REQ[2] )
   END_RUNG
   RUNG wire#w1
      Contact( #MOD_MASTER6_REQ[1] )
      wire#w2
      Move(in := "MASTER_TCP_DATA".MOD_DEVICE_STATION4[1].MASTER_WRITE_DATA.MOD_COIL_DATA, out1 => "MODBUS_DATA_WRITE".MOD_WR_DEV_STN4[1].MOD_COIL_DATA)
      S_Coil( #Mod_TCP_Setup.Mod_Client[6].request )
   END_RUNG
   RUNG wire#w1
      Contact( #MOD_MASTER6_REQ[2] )
   END_RUNG wire#w2
   // the same network as SCL:
   #_w1 := "AlwaysTRUE" AND (#LPG_Fill_Data.FILL_SEQ_OUT.Step_No = 3);
   #_w2 := #_w1 AND NOT #TRIG[6];   // rising edge
   #TRIG[6] := #_w1;
   #MOD_MASTER6_REQ[1] := #_w2;
   #_w3 := "AlwaysTRUE" AND (#LPG_Fill_Data.FILL_SEQ_OUT.Step_No = 8);
   #_w4 := #_w3 AND NOT #TRIG[61];   // rising edge
   #TRIG[61] := #_w3;
   #MOD_MASTER6_REQ[2] := #_w4;
   IF "AlwaysTRUE" AND (#MOD_MASTER6_REQ[1] OR #MOD_MASTER6_REQ[2]) THEN
       "MODBUS_DATA_WRITE".MOD_WR_DEV_STN4[1].MOD_COIL_DATA := "MASTER_TCP_DATA".MOD_DEVICE_STATION4[1].MASTER_WRITE_DATA.MOD_COIL_DATA;
       #Mod_TCP_Setup.Mod_Client[6].request := TRUE;
   END_IF;
END_REGION

REGION Network 20: Modbus Master6 Write Coil Status
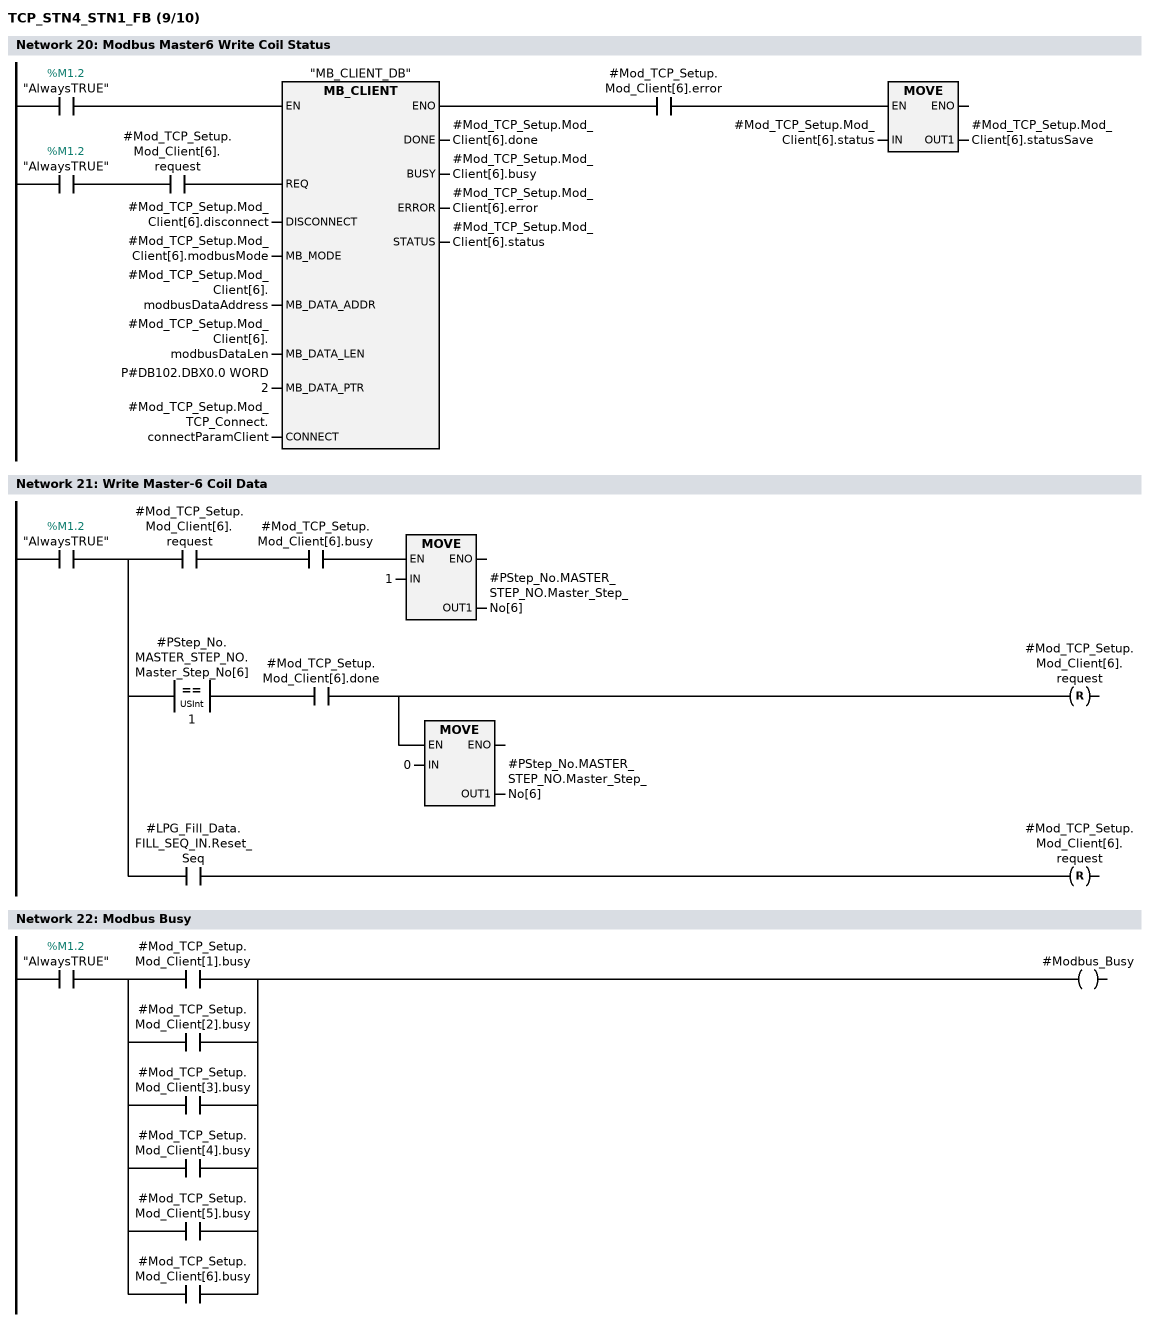
   RUNG wire#powerrail
      Contact( "AlwaysTRUE" )
      "MB_CLIENT_DB".MB_CLIENT(REQ := wire#w1, DISCONNECT := #Mod_TCP_Setup.Mod_Client[6].disconnect, MB_MODE := #Mod_TCP_Setup.Mod_Client[6].modbusMode, MB_DATA_ADDR := #Mod_TCP_Setup.Mod_Client[6].modbusDataAddress, MB_DATA_LEN := #Mod_TCP_Setup.Mod_Client[6].modbusDataLen, MB_DATA_PTR := P#DB102.DBX0.0 WORD 2, CONNECT := #Mod_TCP_Setup.Mod_TCP_Connect.connectParamClient, DONE => #Mod_TCP_Setup.Mod_Client[6].done, BUSY => #Mod_TCP_Setup.Mod_Client[6].busy, ERROR => #Mod_TCP_Setup.Mod_Client[6].error, STATUS => #Mod_TCP_Setup.Mod_Client[6].status)
      Contact( #Mod_TCP_Setup.Mod_Client[6].error )
      Move(in := #Mod_TCP_Setup.Mod_Client[6].status, out1 => #Mod_TCP_Setup.Mod_Client[6].statusSave)
   END_RUNG
   RUNG wire#powerrail
      Contact( "AlwaysTRUE" )
      Contact( #Mod_TCP_Setup.Mod_Client[6].request )
   END_RUNG wire#w1
   // the same network as SCL:
   "MB_CLIENT_DB"(EN := "AlwaysTRUE",   // MB_CLIENT
                  REQ := "AlwaysTRUE" AND #Mod_TCP_Setup.Mod_Client[6].request,
                  DISCONNECT := #Mod_TCP_Setup.Mod_Client[6].disconnect,
                  MB_MODE := #Mod_TCP_Setup.Mod_Client[6].modbusMode,
                  MB_DATA_ADDR := #Mod_TCP_Setup.Mod_Client[6].modbusDataAddress,
                  MB_DATA_LEN := #Mod_TCP_Setup.Mod_Client[6].modbusDataLen,
                  MB_DATA_PTR := P#DB102.DBX0.0 WORD 2,
                  CONNECT := #Mod_TCP_Setup.Mod_TCP_Connect.connectParamClient,
                  DONE => #Mod_TCP_Setup.Mod_Client[6].done,
                  BUSY => #Mod_TCP_Setup.Mod_Client[6].busy,
                  ERROR => #Mod_TCP_Setup.Mod_Client[6].error,
                  STATUS => #Mod_TCP_Setup.Mod_Client[6].status,
                  ENO => #_w1);
   IF #_w1 AND #Mod_TCP_Setup.Mod_Client[6].error THEN
       #Mod_TCP_Setup.Mod_Client[6].statusSave := #Mod_TCP_Setup.Mod_Client[6].status;
   END_IF;
END_REGION

REGION Network 21: Write Master-6 Coil Data
   RUNG wire#powerrail
      Contact( "AlwaysTRUE" )
      wire#w1
      Contact( #Mod_TCP_Setup.Mod_Client[6].request )
      Contact( #Mod_TCP_Setup.Mod_Client[6].busy )
      Move(in := 1, out1 => #PStep_No.MASTER_STEP_NO.Master_Step_No[6])
   END_RUNG
   RUNG wire#w1
      { S7_Templates := "SrcType := USInt" } EQ_Contact(in1 := #PStep_No.MASTER_STEP_NO.Master_Step_No[6], in2 := 1)
      Contact( #Mod_TCP_Setup.Mod_Client[6].done )
      wire#w2
      R_Coil( #Mod_TCP_Setup.Mod_Client[6].request )
   END_RUNG
   RUNG wire#w2
      Move(in := 0, out1 => #PStep_No.MASTER_STEP_NO.Master_Step_No[6])
   END_RUNG
   RUNG wire#w1
      Contact( #LPG_Fill_Data.FILL_SEQ_IN.Reset_Seq )
      R_Coil( #Mod_TCP_Setup.Mod_Client[6].request )
   END_RUNG
   // the same network as SCL:
   IF "AlwaysTRUE" AND #Mod_TCP_Setup.Mod_Client[6].request AND #Mod_TCP_Setup.Mod_Client[6].busy THEN
       #PStep_No.MASTER_STEP_NO.Master_Step_No[6] := 1;
   END_IF;
   #_w1 := "AlwaysTRUE" AND (#PStep_No.MASTER_STEP_NO.Master_Step_No[6] = 1) AND #Mod_TCP_Setup.Mod_Client[6].done;
   IF #_w1 THEN
       #Mod_TCP_Setup.Mod_Client[6].request := FALSE;
       #PStep_No.MASTER_STEP_NO.Master_Step_No[6] := 0;
   END_IF;
   IF "AlwaysTRUE" AND #LPG_Fill_Data.FILL_SEQ_IN.Reset_Seq THEN
       #Mod_TCP_Setup.Mod_Client[6].request := FALSE;
   END_IF;
END_REGION

REGION Network 22: Modbus Busy
   RUNG wire#powerrail
      Contact( "AlwaysTRUE" )
      wire#w1
      Contact( #Mod_TCP_Setup.Mod_Client[1].busy )
      wire#w2
      Coil( #Modbus_Busy )
   END_RUNG
   RUNG wire#w1
      Contact( #Mod_TCP_Setup.Mod_Client[2].busy )
   END_RUNG wire#w2
   RUNG wire#w1
      Contact( #Mod_TCP_Setup.Mod_Client[3].busy )
   END_RUNG wire#w2
   RUNG wire#w1
      Contact( #Mod_TCP_Setup.Mod_Client[4].busy )
   END_RUNG wire#w2
   RUNG wire#w1
      Contact( #Mod_TCP_Setup.Mod_Client[5].busy )
   END_RUNG wire#w2
   RUNG wire#w1
      Contact( #Mod_TCP_Setup.Mod_Client[6].busy )
   END_RUNG wire#w2
   // the same network as SCL:
   #Modbus_Busy := "AlwaysTRUE" AND (#Mod_TCP_Setup.Mod_Client[1].busy OR #Mod_TCP_Setup.Mod_Client[2].busy OR #Mod_TCP_Setup.Mod_Client[3].busy OR #Mod_TCP_Setup.Mod_Client[4].busy OR #Mod_TCP_Setup.Mod_Client[5].busy OR #Mod_TCP_Setup.Mod_Client[6].busy);
END_REGION

REGION Network 23
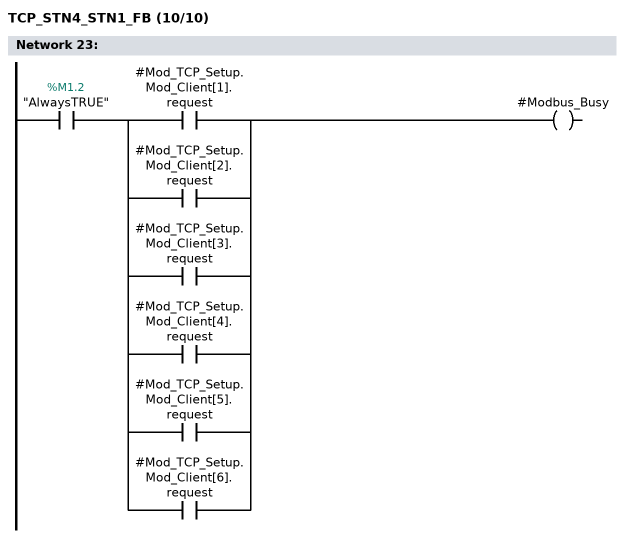
   RUNG wire#powerrail
      Contact( "AlwaysTRUE" )
      wire#w1
      Contact( #Mod_TCP_Setup.Mod_Client[1].request )
      wire#w2
      Coil( #Modbus_Busy )
   END_RUNG
   RUNG wire#w1
      Contact( #Mod_TCP_Setup.Mod_Client[2].request )
   END_RUNG wire#w2
   RUNG wire#w1
      Contact( #Mod_TCP_Setup.Mod_Client[3].request )
   END_RUNG wire#w2
   RUNG wire#w1
      Contact( #Mod_TCP_Setup.Mod_Client[4].request )
   END_RUNG wire#w2
   RUNG wire#w1
      Contact( #Mod_TCP_Setup.Mod_Client[5].request )
   END_RUNG wire#w2
   RUNG wire#w1
      Contact( #Mod_TCP_Setup.Mod_Client[6].request )
   END_RUNG wire#w2
   // the same network as SCL:
   #Modbus_Busy := "AlwaysTRUE" AND (#Mod_TCP_Setup.Mod_Client[1].request OR #Mod_TCP_Setup.Mod_Client[2].request OR #Mod_TCP_Setup.Mod_Client[3].request OR #Mod_TCP_Setup.Mod_Client[4].request OR #Mod_TCP_Setup.Mod_Client[5].request OR #Mod_TCP_Setup.Mod_Client[6].request);
END_REGION
END_FUNCTION_BLOCK

